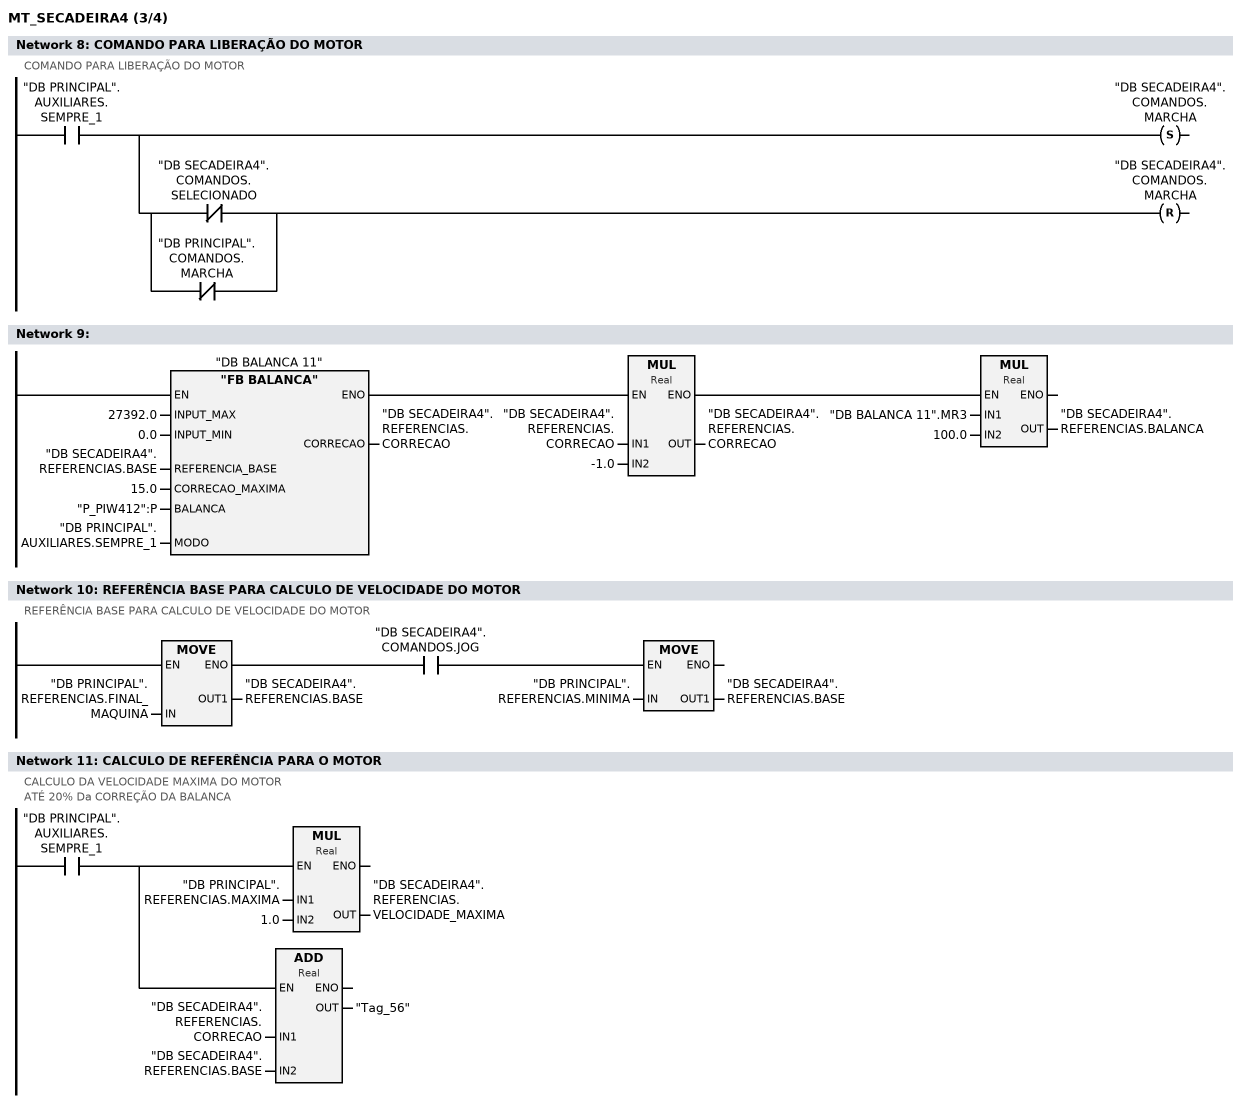
   RUNG wire#powerrail
      Contact( "DB PRINCIPAL".AUXILIARES.SEMPRE_1 )
      wire#w1
      S_Coil( "DB SECADEIRA4".COMANDOS.MARCHA )
   END_RUNG
   RUNG wire#w1
      I_Contact( "DB SECADEIRA4".COMANDOS.SELECIONADO )
      wire#w2
      R_Coil( "DB SECADEIRA4".COMANDOS.MARCHA )
   END_RUNG
   RUNG wire#w1
      I_Contact( "DB PRINCIPAL".COMANDOS.MARCHA )
   END_RUNG wire#w2
   // the same network as SCL:
   IF "DB PRINCIPAL".AUXILIARES.SEMPRE_1 THEN "DB SECADEIRA4".COMANDOS.MARCHA := TRUE; END_IF;
   IF "DB PRINCIPAL".AUXILIARES.SEMPRE_1 AND (NOT "DB SECADEIRA4".COMANDOS.SELECIONADO OR NOT "DB PRINCIPAL".COMANDOS.MARCHA) THEN
       "DB SECADEIRA4".COMANDOS.MARCHA := FALSE;
   END_IF;
END_REGION

REGION Network 9
   RUNG wire#powerrail
      "DB BALANCA 11"(INPUT_MAX := 27392.0, INPUT_MIN := 0.0, REFERENCIA_BASE := "DB SECADEIRA4".REFERENCIAS.BASE, CORRECAO_MAXIMA := 15.0, BALANCA := "P_PIW412":P, MODO := "DB PRINCIPAL".AUXILIARES.SEMPRE_1, CORRECAO => "DB SECADEIRA4".REFERENCIAS.CORRECAO)
      { S7_Templates := "SrcType := Real"; S7_GenerateENO := "TRUE" } Mul(in1 := "DB SECADEIRA4".REFERENCIAS.CORRECAO, in2 := -1.0, out => "DB SECADEIRA4".REFERENCIAS.CORRECAO)
      { S7_Templates := "SrcType := Real"; S7_GenerateENO := "TRUE" } Mul(in1 := "DB BALANCA 11".MR3, in2 := 100.0, out => "DB SECADEIRA4".REFERENCIAS.BALANCA)
   END_RUNG
   // the same network as SCL:
   // ENO of a box is taken as its EN; it also drops when the box reports an error
   "DB BALANCA 11"(INPUT_MAX := 27392.0,   // "FB BALANCA"
                   INPUT_MIN := 0.0,
                   REFERENCIA_BASE := "DB SECADEIRA4".REFERENCIAS.BASE,
                   CORRECAO_MAXIMA := 15.0,
                   BALANCA := "P_PIW412":P,
                   MODO := "DB PRINCIPAL".AUXILIARES.SEMPRE_1,
                   CORRECAO => "DB SECADEIRA4".REFERENCIAS.CORRECAO,
                   ENO => #_w1);
   IF #_w1 THEN
       "DB SECADEIRA4".REFERENCIAS.CORRECAO := "DB SECADEIRA4".REFERENCIAS.CORRECAO * (-1.0);
       "DB SECADEIRA4".REFERENCIAS.BALANCA := "DB BALANCA 11".MR3 * 100.0;
   END_IF;
END_REGION

REGION Network 10: REFERÊNCIA BASE PARA CALCULO DE VELOCIDADE DO MOTOR
   // REFERÊNCIA BASE PARA CALCULO DE VELOCIDADE DO MOTOR
   RUNG wire#powerrail
      { S7_GenerateENO := "TRUE" } Move(in := "DB PRINCIPAL".REFERENCIAS.FINAL_MAQUINA, out1 => "DB SECADEIRA4".REFERENCIAS.BASE)
      Contact( "DB SECADEIRA4".COMANDOS.JOG )
      { S7_GenerateENO := "TRUE" } Move(in := "DB PRINCIPAL".REFERENCIAS.MINIMA, out1 => "DB SECADEIRA4".REFERENCIAS.BASE)
   END_RUNG
   // the same network as SCL:
   // ENO of a box is taken as its EN; it also drops when the box reports an error
   "DB SECADEIRA4".REFERENCIAS.BASE := "DB PRINCIPAL".REFERENCIAS.FINAL_MAQUINA;
   IF "DB SECADEIRA4".COMANDOS.JOG THEN
       "DB SECADEIRA4".REFERENCIAS.BASE := "DB PRINCIPAL".REFERENCIAS.MINIMA;
   END_IF;
END_REGION

REGION Network 11: CALCULO DE REFERÊNCIA PARA O MOTOR
   // CALCULO DA VELOCIDADE MAXIMA DO MOTOR
   // ATÉ 20% Da CORREÇÃO DA BALANCA
   RUNG wire#powerrail
      Contact( "DB PRINCIPAL".AUXILIARES.SEMPRE_1 )
      wire#w1
      { S7_Templates := "SrcType := Real"; S7_GenerateENO := "TRUE" } Mul(in1 := "DB PRINCIPAL".REFERENCIAS.MAXIMA, in2 := 1.0, out => "DB SECADEIRA4".REFERENCIAS.VELOCIDADE_MAXIMA)
   END_RUNG
   RUNG wire#w1
      { S7_Templates := "SrcType := Real"; S7_GenerateENO := "TRUE" } Add(in1 := "DB SECADEIRA4".REFERENCIAS.CORRECAO, in2 := "DB SECADEIRA4".REFERENCIAS.BASE, out => "Tag_56")
   END_RUNG
   // the same network as SCL:
   IF "DB PRINCIPAL".AUXILIARES.SEMPRE_1 THEN
       "DB SECADEIRA4".REFERENCIAS.VELOCIDADE_MAXIMA := "DB PRINCIPAL".REFERENCIAS.MAXIMA * 1.0;
       "Tag_56" := "DB SECADEIRA4".REFERENCIAS.CORRECAO + "DB SECADEIRA4".REFERENCIAS.BASE;
   END_IF;
END_REGION

REGION Network 12: ACC/DEC DA REFERÊNCIA DO MOTOR
   // ACC/DEC DA REFERÊNCIA DO MOTOR
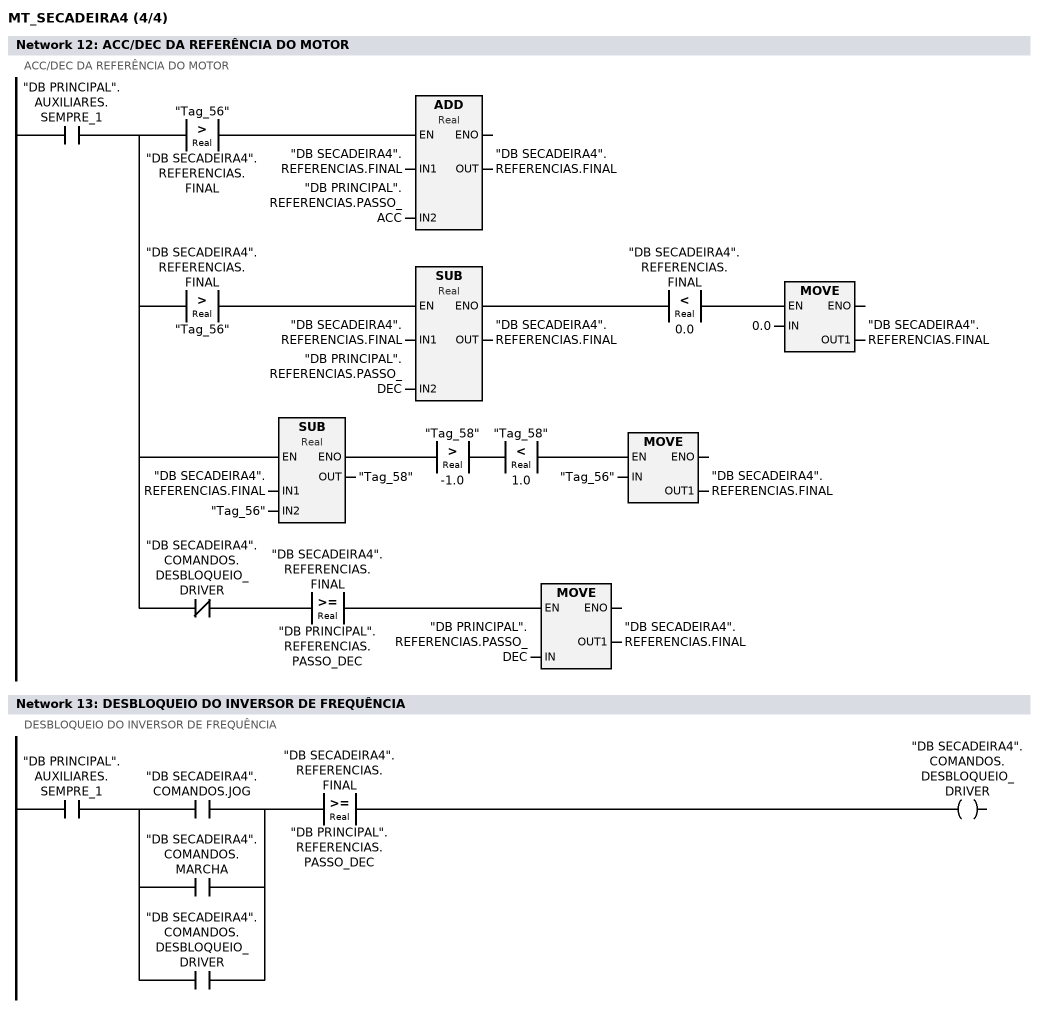
   RUNG wire#powerrail
      Contact( "DB PRINCIPAL".AUXILIARES.SEMPRE_1 )
      wire#w1
      { S7_Templates := "SrcType := Real" } GT_Contact(in1 := "Tag_56", in2 := "DB SECADEIRA4".REFERENCIAS.FINAL)
      { S7_Templates := "SrcType := Real"; S7_GenerateENO := "TRUE" } Add(in1 := "DB SECADEIRA4".REFERENCIAS.FINAL, in2 := "DB PRINCIPAL".REFERENCIAS.PASSO_ACC, out => "DB SECADEIRA4".REFERENCIAS.FINAL)
   END_RUNG
   RUNG wire#w1
      { S7_Templates := "SrcType := Real" } GT_Contact(in1 := "DB SECADEIRA4".REFERENCIAS.FINAL, in2 := "Tag_56")
      { S7_Templates := "SrcType := Real"; S7_GenerateENO := "TRUE" } Sub(in1 := "DB SECADEIRA4".REFERENCIAS.FINAL, in2 := "DB PRINCIPAL".REFERENCIAS.PASSO_DEC, out => "DB SECADEIRA4".REFERENCIAS.FINAL)
      { S7_Templates := "SrcType := Real" } LT_Contact(in1 := "DB SECADEIRA4".REFERENCIAS.FINAL, in2 := 0.0)
      { S7_GenerateENO := "TRUE" } Move(in := 0.0, out1 => "DB SECADEIRA4".REFERENCIAS.FINAL)
   END_RUNG
   RUNG wire#w1
      { S7_Templates := "SrcType := Real"; S7_GenerateENO := "TRUE" } Sub(in1 := "DB SECADEIRA4".REFERENCIAS.FINAL, in2 := "Tag_56", out => "Tag_58")
      { S7_Templates := "SrcType := Real" } GT_Contact(in1 := "Tag_58", in2 := -1.0)
      { S7_Templates := "SrcType := Real" } LT_Contact(in1 := "Tag_58", in2 := 1.0)
      { S7_GenerateENO := "TRUE" } Move(in := "Tag_56", out1 => "DB SECADEIRA4".REFERENCIAS.FINAL)
   END_RUNG
   RUNG wire#w1
      I_Contact( "DB SECADEIRA4".COMANDOS.DESBLOQUEIO_DRIVER )
      { S7_Templates := "SrcType := Real" } GE_Contact(in1 := "DB SECADEIRA4".REFERENCIAS.FINAL, in2 := "DB PRINCIPAL".REFERENCIAS.PASSO_DEC)
      { S7_GenerateENO := "TRUE" } Move(in := "DB PRINCIPAL".REFERENCIAS.PASSO_DEC, out1 => "DB SECADEIRA4".REFERENCIAS.FINAL)
   END_RUNG
   // the same network as SCL:
   // ENO of a box is taken as its EN; it also drops when the box reports an error
   IF "DB PRINCIPAL".AUXILIARES.SEMPRE_1 AND ("Tag_56" > "DB SECADEIRA4".REFERENCIAS.FINAL) THEN
       "DB SECADEIRA4".REFERENCIAS.FINAL := "DB SECADEIRA4".REFERENCIAS.FINAL + "DB PRINCIPAL".REFERENCIAS.PASSO_ACC;
   END_IF;
   #_w1 := "DB PRINCIPAL".AUXILIARES.SEMPRE_1 AND ("DB SECADEIRA4".REFERENCIAS.FINAL > "Tag_56");
   IF #_w1 THEN
       "DB SECADEIRA4".REFERENCIAS.FINAL := "DB SECADEIRA4".REFERENCIAS.FINAL - "DB PRINCIPAL".REFERENCIAS.PASSO_DEC;
   END_IF;
   IF #_w1 AND ("DB SECADEIRA4".REFERENCIAS.FINAL < 0.0) THEN
       "DB SECADEIRA4".REFERENCIAS.FINAL := 0.0;
   END_IF;
   IF "DB PRINCIPAL".AUXILIARES.SEMPRE_1 THEN
       "Tag_58" := "DB SECADEIRA4".REFERENCIAS.FINAL - "Tag_56";
   END_IF;
   IF "DB PRINCIPAL".AUXILIARES.SEMPRE_1 AND ("Tag_58" > (-1.0)) AND ("Tag_58" < 1.0) THEN
       "DB SECADEIRA4".REFERENCIAS.FINAL := "Tag_56";
   END_IF;
   IF "DB PRINCIPAL".AUXILIARES.SEMPRE_1 AND NOT "DB SECADEIRA4".COMANDOS.DESBLOQUEIO_DRIVER AND ("DB SECADEIRA4".REFERENCIAS.FINAL >= "DB PRINCIPAL".REFERENCIAS.PASSO_DEC) THEN
       "DB SECADEIRA4".REFERENCIAS.FINAL := "DB PRINCIPAL".REFERENCIAS.PASSO_DEC;
   END_IF;
END_REGION

REGION Network 13: DESBLOQUEIO DO INVERSOR DE FREQUÊNCIA
   // DESBLOQUEIO DO INVERSOR DE FREQUÊNCIA
   RUNG wire#powerrail
      Contact( "DB PRINCIPAL".AUXILIARES.SEMPRE_1 )
      wire#w1
      Contact( "DB SECADEIRA4".COMANDOS.JOG )
      wire#w2
      { S7_Templates := "SrcType := Real" } GE_Contact(in1 := "DB SECADEIRA4".REFERENCIAS.FINAL, in2 := "DB PRINCIPAL".REFERENCIAS.PASSO_DEC)
      Coil( "DB SECADEIRA4".COMANDOS.DESBLOQUEIO_DRIVER )
   END_RUNG
   RUNG wire#w1
      Contact( "DB SECADEIRA4".COMANDOS.MARCHA )
   END_RUNG wire#w2
   RUNG wire#w1
      Contact( "DB SECADEIRA4".COMANDOS.DESBLOQUEIO_DRIVER )
   END_RUNG wire#w2
   // the same network as SCL:
   "DB SECADEIRA4".COMANDOS.DESBLOQUEIO_DRIVER := "DB PRINCIPAL".AUXILIARES.SEMPRE_1 AND ("DB SECADEIRA4".COMANDOS.JOG OR "DB SECADEIRA4".COMANDOS.MARCHA OR "DB SECADEIRA4".COMANDOS.DESBLOQUEIO_DRIVER) AND ("DB SECADEIRA4".REFERENCIAS.FINAL >= "DB PRINCIPAL".REFERENCIAS.PASSO_DEC);
END_REGION

REGION Network 14 (STL): STATUS / CONTROLE - INVERSOR DE FREQUÊNCIA
   // DANFOSS FC300 PROFIBUS - TEX24626INV001
   // STATUS DO INVERSOR DE FREQUÊNCIA
         L     "Tag_42":P;
         T     "Tag_1";
         AN    "Tag_59";
         =     "DB SECADEIRA4".COMANDOS.STATUS_DRIVER;

   // CONTROLE DO INVERSOR DE FREQUÊNCIA
         L     1150;
         T     "Tag_1";
         A     "DB SECADEIRA4".COMANDOS.DESBLOQUEIO_DRIVER;
         =     "Tag_60";
         A     "T2";
         AN    "DB SECADEIRA4".COMANDOS.STATUS_DRIVER;
         =     "Tag_61";
         L     "Tag_1";
         T     "Tag_43":P;

   // REFERÊNCIA PARA O INVERSOR DE FREQUÊNCIA
         L     "DB SECADEIRA4".REFERENCIAS.FINAL;
         L     16384.0;
         *R;

         L     "DB SECADEIRA4".REFERENCIAS.VELOCIDADE_MAXIMA;
         /R;
         RND;
         T     "Tag_62";
         L     "Tag_62";
         T     "Tag_44":P;
END_REGION

REGION Network 15 (STL): INVERSOR RESERVA
         A     "DB PRINCIPAL".AUXILIARES.SEMPRE_1;
         =     %L24.0;
         A     %L24.0;
         A(;
         L     "DB PRINCIPAL".AUXILIARES1.INVERSOR_RESERVA1;
         L     15;
         ==I;
         );
         =     %L24.1;
         A     %L24.1;
         JNB   M00d;
         L     "DB SECADEIRA4".REFERENCIAS.FINAL;
         L     3.456;
         *R;
         T     #AUX_R;
         RND;
         T     "P_QW100":P;
   M00d: NOP   0;
         A     %L24.1;
         A     "I130";
         S     "DB PRINCIPAL".ALARME.INV_RESERVA1;
         A     %L24.1;
         A     "DB SECADEIRA4".COMANDOS.DESBLOQUEIO_DRIVER;
         S     "Q134";
         A     %L24.1;
         AN    "DB SECADEIRA4".COMANDOS.DESBLOQUEIO_DRIVER;
         R     "Q134";
         A     %L24.0;
         A(;
         L     "DB PRINCIPAL".AUXILIARES1.INVERSOR_RESERVA2;
         L     15;
         ==I;
         );
         =     %L24.1;
         A     %L24.1;
         JNB   M00e;
         L     "DB SECADEIRA4".REFERENCIAS.FINAL;
         L     3.456;
         *R;
         T     #AUX_R;
         RND;
         T     "P_QW102":P;
   M00e: NOP   0;
         A     %L24.1;
         A     "I132";
         S     "DB PRINCIPAL".ALARME.INV_RESERVA2;
         A     %L24.1;
         A     "DB SECADEIRA4".COMANDOS.DESBLOQUEIO_DRIVER;
         S     "Q135";
         A     %L24.1;
         AN    "DB SECADEIRA4".COMANDOS.DESBLOQUEIO_DRIVER;
         R     "Q135";
END_REGION
END_FUNCTION

FUNCTION "MT_PUXADOR_JOTA_SAIDA" : Void   // FC25, LAD
TITLE = MÓDULO DE CONTROLE DO PUXADOR DO JOTA DA SAIDA
{ S7_Optimized_Access := 'FALSE' }
AUTHOR : THALLES
FAMILY : TRAÇÃO
NAME : LINHA1
VERSION : 0.1
// DATA BLOCK DE CONTROLE // DB25
// Automation Pack Automação Indl. e Com. Ltda.
// Cliente: Texima S/A Ind. de Máquinas
// Cliente Final: Cia. Fiação e Tecidos Santo Antonio.
// Máquina: LINHA 1 DENIN - O.S.: 24.626
   VAR_TEMP
      AUX_R : Real;
   END_VAR
   VAR_TEMP   // added for the SCL form of the ladder/FBD networks
      _w1 : Bool;
   END_VAR
BEGIN

REGION Network 1: ALARMES
   // RESET DOS ALARMES
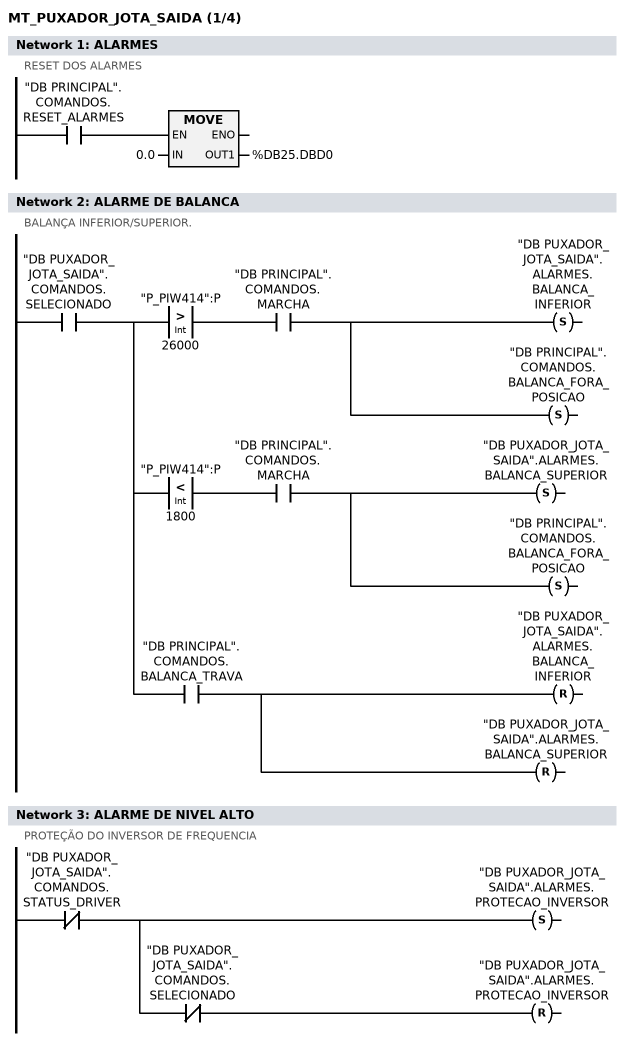
   RUNG wire#powerrail
      Contact( "DB PRINCIPAL".COMANDOS.RESET_ALARMES )
      { S7_GenerateENO := "TRUE" } Move(in := 0.0, out1 => %DB25.DBD0)
   END_RUNG
   // the same network as SCL:
   IF "DB PRINCIPAL".COMANDOS.RESET_ALARMES THEN %DB25.DBD0 := 0.0; END_IF;
END_REGION

REGION Network 2: ALARME DE BALANCA
   // BALANÇA INFERIOR/SUPERIOR.
   RUNG wire#powerrail
      Contact( "DB PUXADOR_JOTA_SAIDA".COMANDOS.SELECIONADO )
      wire#w1
      { S7_Templates := "SrcType := Int" } GT_Contact(in1 := "P_PIW414":P, in2 := 26000)
      Contact( "DB PRINCIPAL".COMANDOS.MARCHA )
      wire#w2
      S_Coil( "DB PUXADOR_JOTA_SAIDA".ALARMES.BALANCA_INFERIOR )
   END_RUNG
   RUNG wire#w2
      S_Coil( "DB PRINCIPAL".COMANDOS.BALANCA_FORA_POSICAO )
   END_RUNG
   RUNG wire#w1
      { S7_Templates := "SrcType := Int" } LT_Contact(in1 := "P_PIW414":P, in2 := 1800)
      Contact( "DB PRINCIPAL".COMANDOS.MARCHA )
      wire#w3
      S_Coil( "DB PUXADOR_JOTA_SAIDA".ALARMES.BALANCA_SUPERIOR )
   END_RUNG
   RUNG wire#w3
      S_Coil( "DB PRINCIPAL".COMANDOS.BALANCA_FORA_POSICAO )
   END_RUNG
   RUNG wire#w1
      Contact( "DB PRINCIPAL".COMANDOS.BALANCA_TRAVA )
      wire#w4
      R_Coil( "DB PUXADOR_JOTA_SAIDA".ALARMES.BALANCA_INFERIOR )
   END_RUNG
   RUNG wire#w4
      R_Coil( "DB PUXADOR_JOTA_SAIDA".ALARMES.BALANCA_SUPERIOR )
   END_RUNG
   // the same network as SCL:
   IF "DB PUXADOR_JOTA_SAIDA".COMANDOS.SELECIONADO AND ("P_PIW414":P > 26000) AND "DB PRINCIPAL".COMANDOS.MARCHA THEN
       "DB PUXADOR_JOTA_SAIDA".ALARMES.BALANCA_INFERIOR := TRUE;
       "DB PRINCIPAL".COMANDOS.BALANCA_FORA_POSICAO := TRUE;
   END_IF;
   IF "DB PUXADOR_JOTA_SAIDA".COMANDOS.SELECIONADO AND ("P_PIW414":P < 1800) AND "DB PRINCIPAL".COMANDOS.MARCHA THEN
       "DB PUXADOR_JOTA_SAIDA".ALARMES.BALANCA_SUPERIOR := TRUE;
       "DB PRINCIPAL".COMANDOS.BALANCA_FORA_POSICAO := TRUE;
   END_IF;
   IF "DB PUXADOR_JOTA_SAIDA".COMANDOS.SELECIONADO AND "DB PRINCIPAL".COMANDOS.BALANCA_TRAVA THEN
       "DB PUXADOR_JOTA_SAIDA".ALARMES.BALANCA_INFERIOR := FALSE;
       "DB PUXADOR_JOTA_SAIDA".ALARMES.BALANCA_SUPERIOR := FALSE;
   END_IF;
END_REGION

REGION Network 3: ALARME DE NIVEL ALTO
   // PROTEÇÃO DO INVERSOR DE FREQUENCIA
   RUNG wire#powerrail
      I_Contact( "DB PUXADOR_JOTA_SAIDA".COMANDOS.STATUS_DRIVER )
      wire#w1
      S_Coil( "DB PUXADOR_JOTA_SAIDA".ALARMES.PROTECAO_INVERSOR )
   END_RUNG
   RUNG wire#w1
      I_Contact( "DB PUXADOR_JOTA_SAIDA".COMANDOS.SELECIONADO )
      R_Coil( "DB PUXADOR_JOTA_SAIDA".ALARMES.PROTECAO_INVERSOR )
   END_RUNG
   // the same network as SCL:
   #_w1 := NOT "DB PUXADOR_JOTA_SAIDA".COMANDOS.STATUS_DRIVER;
   IF #_w1 THEN "DB PUXADOR_JOTA_SAIDA".ALARMES.PROTECAO_INVERSOR := TRUE; END_IF;
   IF #_w1 AND NOT "DB PUXADOR_JOTA_SAIDA".COMANDOS.SELECIONADO THEN
       "DB PUXADOR_JOTA_SAIDA".ALARMES.PROTECAO_INVERSOR := FALSE;
   END_IF;
END_REGION

REGION Network 4: ALARMES
   // ATIVAÇÃO DO BIT DE ALARME DE NIVEL ALTO
   // ATIVAÇÃO DO BIT DE ALARME DE NIVEL BAIXO
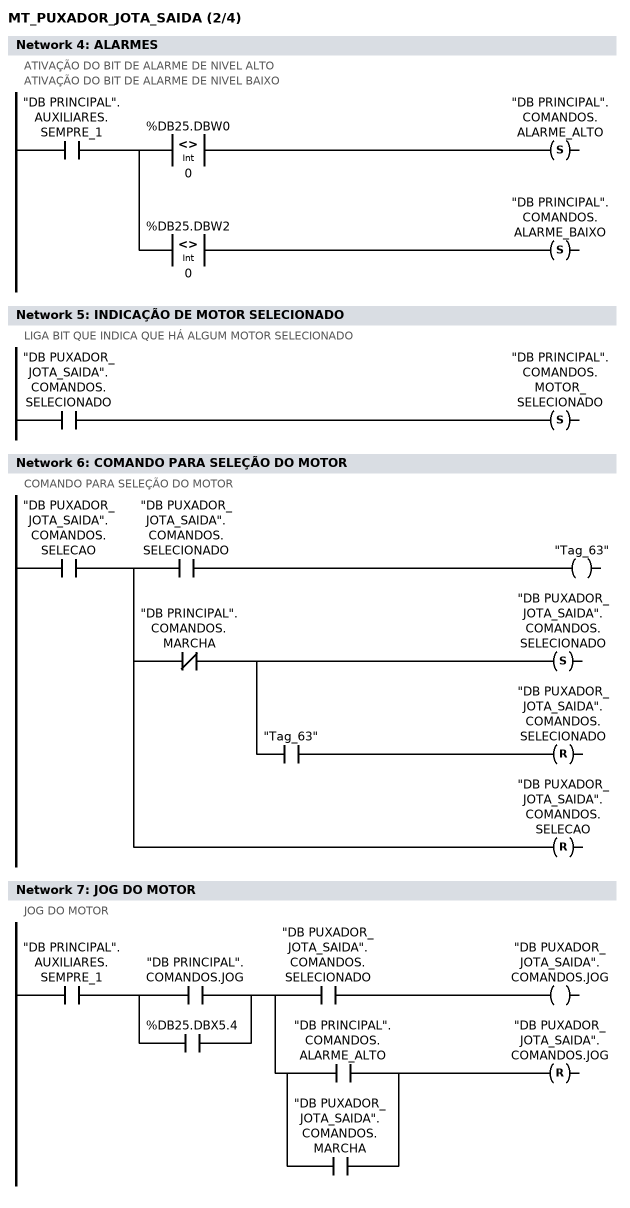
   RUNG wire#powerrail
      Contact( "DB PRINCIPAL".AUXILIARES.SEMPRE_1 )
      wire#w1
      { S7_Templates := "SrcType := Int" } NE_Contact(in1 := %DB25.DBW0, in2 := 0)
      S_Coil( "DB PRINCIPAL".COMANDOS.ALARME_ALTO )
   END_RUNG
   RUNG wire#w1
      { S7_Templates := "SrcType := Int" } NE_Contact(in1 := %DB25.DBW2, in2 := 0)
      S_Coil( "DB PRINCIPAL".COMANDOS.ALARME_BAIXO )
   END_RUNG
   // the same network as SCL:
   IF "DB PRINCIPAL".AUXILIARES.SEMPRE_1 AND (%DB25.DBW0 <> 0) THEN
       "DB PRINCIPAL".COMANDOS.ALARME_ALTO := TRUE;
   END_IF;
   IF "DB PRINCIPAL".AUXILIARES.SEMPRE_1 AND (%DB25.DBW2 <> 0) THEN
       "DB PRINCIPAL".COMANDOS.ALARME_BAIXO := TRUE;
   END_IF;
END_REGION

REGION Network 5: INDICAÇÃO DE MOTOR SELECIONADO
   // LIGA BIT QUE INDICA QUE HÁ ALGUM MOTOR SELECIONADO
   RUNG wire#powerrail
      Contact( "DB PUXADOR_JOTA_SAIDA".COMANDOS.SELECIONADO )
      S_Coil( "DB PRINCIPAL".COMANDOS.MOTOR_SELECIONADO )
   END_RUNG
   // the same network as SCL:
   IF "DB PUXADOR_JOTA_SAIDA".COMANDOS.SELECIONADO THEN
       "DB PRINCIPAL".COMANDOS.MOTOR_SELECIONADO := TRUE;
   END_IF;
END_REGION

REGION Network 6: COMANDO PARA SELEÇÃO DO MOTOR
   // COMANDO PARA SELEÇÃO DO MOTOR
   RUNG wire#powerrail
      Contact( "DB PUXADOR_JOTA_SAIDA".COMANDOS.SELECAO )
      wire#w1
      Contact( "DB PUXADOR_JOTA_SAIDA".COMANDOS.SELECIONADO )
      Coil( "Tag_63" )
   END_RUNG
   RUNG wire#w1
      I_Contact( "DB PRINCIPAL".COMANDOS.MARCHA )
      wire#w2
      S_Coil( "DB PUXADOR_JOTA_SAIDA".COMANDOS.SELECIONADO )
   END_RUNG
   RUNG wire#w2
      Contact( "Tag_63" )
      R_Coil( "DB PUXADOR_JOTA_SAIDA".COMANDOS.SELECIONADO )
   END_RUNG
   RUNG wire#w1
      R_Coil( "DB PUXADOR_JOTA_SAIDA".COMANDOS.SELECAO )
   END_RUNG
   // the same network as SCL:
   "Tag_63" := "DB PUXADOR_JOTA_SAIDA".COMANDOS.SELECAO AND "DB PUXADOR_JOTA_SAIDA".COMANDOS.SELECIONADO;
   #_w1 := "DB PUXADOR_JOTA_SAIDA".COMANDOS.SELECAO AND NOT "DB PRINCIPAL".COMANDOS.MARCHA;
   IF #_w1 THEN "DB PUXADOR_JOTA_SAIDA".COMANDOS.SELECIONADO := TRUE; END_IF;
   IF #_w1 AND "Tag_63" THEN "DB PUXADOR_JOTA_SAIDA".COMANDOS.SELECIONADO := FALSE; END_IF;
   IF "DB PUXADOR_JOTA_SAIDA".COMANDOS.SELECAO THEN
       "DB PUXADOR_JOTA_SAIDA".COMANDOS.SELECAO := FALSE;
   END_IF;
END_REGION

REGION Network 7: JOG DO MOTOR
   // JOG DO MOTOR
   RUNG wire#powerrail
      Contact( "DB PRINCIPAL".AUXILIARES.SEMPRE_1 )
      wire#w1
      Contact( "DB PRINCIPAL".COMANDOS.JOG )
      wire#w2
      Contact( "DB PUXADOR_JOTA_SAIDA".COMANDOS.SELECIONADO )
      Coil( "DB PUXADOR_JOTA_SAIDA".COMANDOS.JOG )
   END_RUNG
   RUNG wire#w1
      Contact( %DB25.DBX5.4 )
   END_RUNG wire#w2
   RUNG wire#w2
      Contact( "DB PRINCIPAL".COMANDOS.ALARME_ALTO )
      wire#w3
      R_Coil( "DB PUXADOR_JOTA_SAIDA".COMANDOS.JOG )
   END_RUNG
   RUNG wire#w2
      Contact( "DB PUXADOR_JOTA_SAIDA".COMANDOS.MARCHA )
   END_RUNG wire#w3
   // the same network as SCL:
   #_w1 := "DB PRINCIPAL".AUXILIARES.SEMPRE_1 AND ("DB PRINCIPAL".COMANDOS.JOG OR %DB25.DBX5.4);
   "DB PUXADOR_JOTA_SAIDA".COMANDOS.JOG := #_w1 AND "DB PUXADOR_JOTA_SAIDA".COMANDOS.SELECIONADO;
   IF #_w1 AND ("DB PRINCIPAL".COMANDOS.ALARME_ALTO OR "DB PUXADOR_JOTA_SAIDA".COMANDOS.MARCHA) THEN
       "DB PUXADOR_JOTA_SAIDA".COMANDOS.JOG := FALSE;
   END_IF;
END_REGION

REGION Network 8: COMANDO PARA LIBERAÇÃO DO MOTOR
   // COMANDO PARA LIBERAÇÃO DO MOTOR
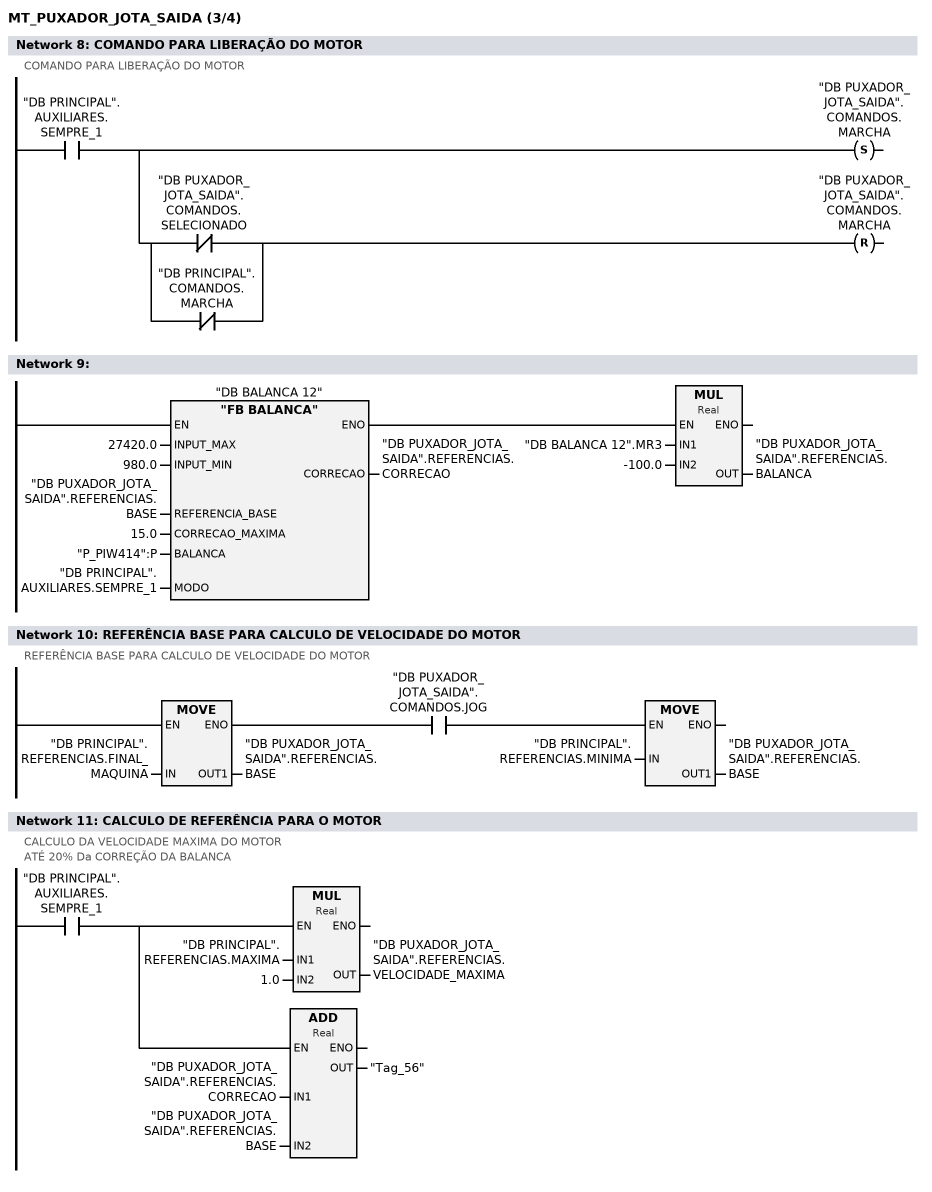
   RUNG wire#powerrail
      Contact( "DB PRINCIPAL".AUXILIARES.SEMPRE_1 )
      wire#w1
      S_Coil( "DB PUXADOR_JOTA_SAIDA".COMANDOS.MARCHA )
   END_RUNG
   RUNG wire#w1
      I_Contact( "DB PUXADOR_JOTA_SAIDA".COMANDOS.SELECIONADO )
      wire#w2
      R_Coil( "DB PUXADOR_JOTA_SAIDA".COMANDOS.MARCHA )
   END_RUNG
   RUNG wire#w1
      I_Contact( "DB PRINCIPAL".COMANDOS.MARCHA )
   END_RUNG wire#w2
   // the same network as SCL:
   IF "DB PRINCIPAL".AUXILIARES.SEMPRE_1 THEN "DB PUXADOR_JOTA_SAIDA".COMANDOS.MARCHA := TRUE; END_IF;
   IF "DB PRINCIPAL".AUXILIARES.SEMPRE_1 AND (NOT "DB PUXADOR_JOTA_SAIDA".COMANDOS.SELECIONADO OR NOT "DB PRINCIPAL".COMANDOS.MARCHA) THEN
       "DB PUXADOR_JOTA_SAIDA".COMANDOS.MARCHA := FALSE;
   END_IF;
END_REGION

REGION Network 9
   RUNG wire#powerrail
      "DB BALANCA 12"(INPUT_MAX := 27420.0, INPUT_MIN := 980.0, REFERENCIA_BASE := "DB PUXADOR_JOTA_SAIDA".REFERENCIAS.BASE, CORRECAO_MAXIMA := 15.0, BALANCA := "P_PIW414":P, MODO := "DB PRINCIPAL".AUXILIARES.SEMPRE_1, CORRECAO => "DB PUXADOR_JOTA_SAIDA".REFERENCIAS.CORRECAO)
      { S7_Templates := "SrcType := Real"; S7_GenerateENO := "TRUE" } Mul(in1 := "DB BALANCA 12".MR3, in2 := -100.0, out => "DB PUXADOR_JOTA_SAIDA".REFERENCIAS.BALANCA)
   END_RUNG
   // the same network as SCL:
   "DB BALANCA 12"(INPUT_MAX := 27420.0,   // "FB BALANCA"
                   INPUT_MIN := 980.0,
                   REFERENCIA_BASE := "DB PUXADOR_JOTA_SAIDA".REFERENCIAS.BASE,
                   CORRECAO_MAXIMA := 15.0,
                   BALANCA := "P_PIW414":P,
                   MODO := "DB PRINCIPAL".AUXILIARES.SEMPRE_1,
                   CORRECAO => "DB PUXADOR_JOTA_SAIDA".REFERENCIAS.CORRECAO,
                   ENO => #_w1);
   IF #_w1 THEN "DB PUXADOR_JOTA_SAIDA".REFERENCIAS.BALANCA := "DB BALANCA 12".MR3 * (-100.0); END_IF;
END_REGION

REGION Network 10: REFERÊNCIA BASE PARA CALCULO DE VELOCIDADE DO MOTOR
   // REFERÊNCIA BASE PARA CALCULO DE VELOCIDADE DO MOTOR
   RUNG wire#powerrail
      { S7_GenerateENO := "TRUE" } Move(in := "DB PRINCIPAL".REFERENCIAS.FINAL_MAQUINA, out1 => "DB PUXADOR_JOTA_SAIDA".REFERENCIAS.BASE)
      Contact( "DB PUXADOR_JOTA_SAIDA".COMANDOS.JOG )
      { S7_GenerateENO := "TRUE" } Move(in := "DB PRINCIPAL".REFERENCIAS.MINIMA, out1 => "DB PUXADOR_JOTA_SAIDA".REFERENCIAS.BASE)
   END_RUNG
   // the same network as SCL:
   // ENO of a box is taken as its EN; it also drops when the box reports an error
   "DB PUXADOR_JOTA_SAIDA".REFERENCIAS.BASE := "DB PRINCIPAL".REFERENCIAS.FINAL_MAQUINA;
   IF "DB PUXADOR_JOTA_SAIDA".COMANDOS.JOG THEN
       "DB PUXADOR_JOTA_SAIDA".REFERENCIAS.BASE := "DB PRINCIPAL".REFERENCIAS.MINIMA;
   END_IF;
END_REGION

REGION Network 11: CALCULO DE REFERÊNCIA PARA O MOTOR
   // CALCULO DA VELOCIDADE MAXIMA DO MOTOR
   // ATÉ 20% Da CORREÇÃO DA BALANCA
   RUNG wire#powerrail
      Contact( "DB PRINCIPAL".AUXILIARES.SEMPRE_1 )
      wire#w1
      { S7_Templates := "SrcType := Real"; S7_GenerateENO := "TRUE" } Mul(in1 := "DB PRINCIPAL".REFERENCIAS.MAXIMA, in2 := 1.0, out => "DB PUXADOR_JOTA_SAIDA".REFERENCIAS.VELOCIDADE_MAXIMA)
   END_RUNG
   RUNG wire#w1
      { S7_Templates := "SrcType := Real"; S7_GenerateENO := "TRUE" } Add(in1 := "DB PUXADOR_JOTA_SAIDA".REFERENCIAS.CORRECAO, in2 := "DB PUXADOR_JOTA_SAIDA".REFERENCIAS.BASE, out => "Tag_56")
   END_RUNG
   // the same network as SCL:
   IF "DB PRINCIPAL".AUXILIARES.SEMPRE_1 THEN
       "DB PUXADOR_JOTA_SAIDA".REFERENCIAS.VELOCIDADE_MAXIMA := "DB PRINCIPAL".REFERENCIAS.MAXIMA * 1.0;
       "Tag_56" := "DB PUXADOR_JOTA_SAIDA".REFERENCIAS.CORRECAO + "DB PUXADOR_JOTA_SAIDA".REFERENCIAS.BASE;
   END_IF;
END_REGION

REGION Network 12: ACC/DEC DA REFERÊNCIA DO MOTOR
   // ACC/DEC DA REFERÊNCIA DO MOTOR
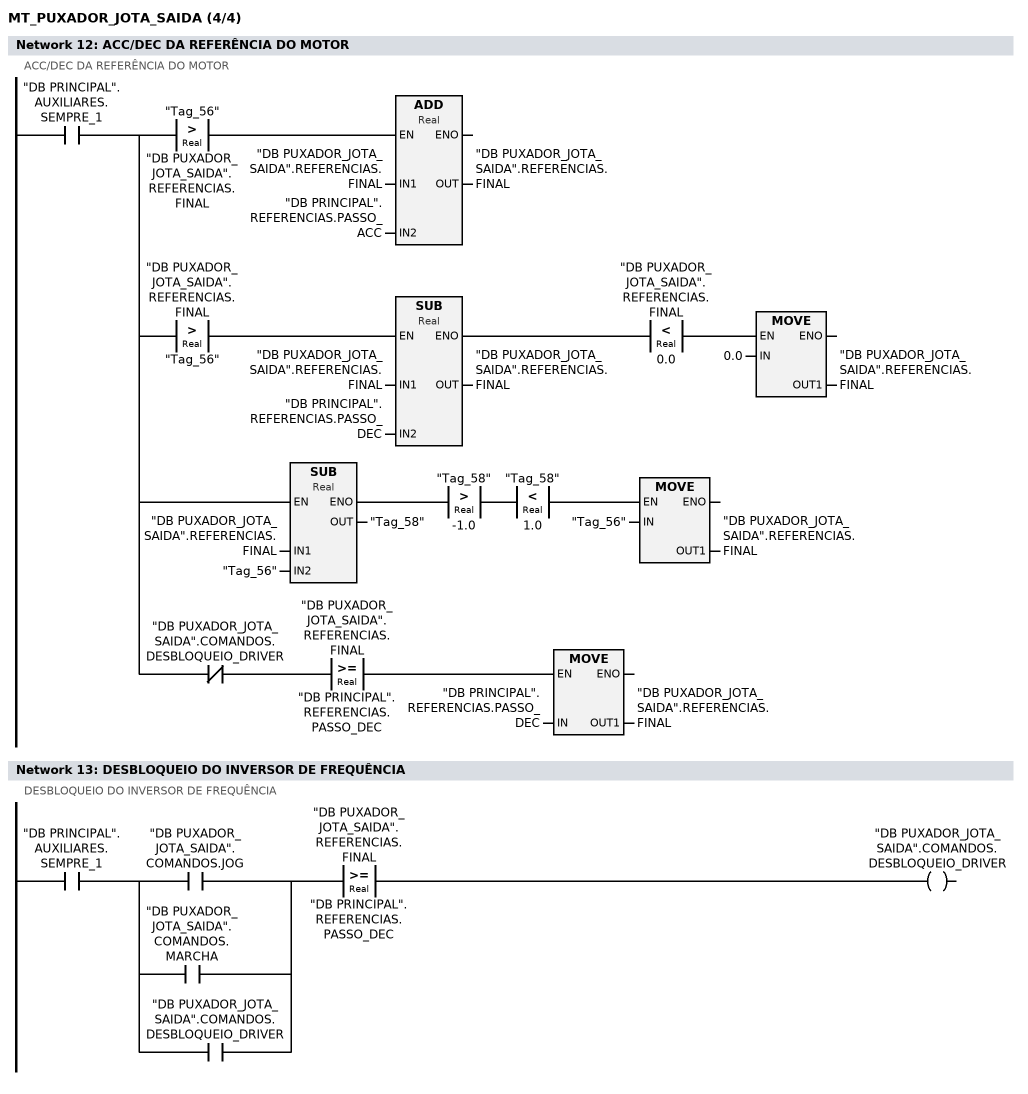
   RUNG wire#powerrail
      Contact( "DB PRINCIPAL".AUXILIARES.SEMPRE_1 )
      wire#w1
      { S7_Templates := "SrcType := Real" } GT_Contact(in1 := "Tag_56", in2 := "DB PUXADOR_JOTA_SAIDA".REFERENCIAS.FINAL)
      { S7_Templates := "SrcType := Real"; S7_GenerateENO := "TRUE" } Add(in1 := "DB PUXADOR_JOTA_SAIDA".REFERENCIAS.FINAL, in2 := "DB PRINCIPAL".REFERENCIAS.PASSO_ACC, out => "DB PUXADOR_JOTA_SAIDA".REFERENCIAS.FINAL)
   END_RUNG
   RUNG wire#w1
      { S7_Templates := "SrcType := Real" } GT_Contact(in1 := "DB PUXADOR_JOTA_SAIDA".REFERENCIAS.FINAL, in2 := "Tag_56")
      { S7_Templates := "SrcType := Real"; S7_GenerateENO := "TRUE" } Sub(in1 := "DB PUXADOR_JOTA_SAIDA".REFERENCIAS.FINAL, in2 := "DB PRINCIPAL".REFERENCIAS.PASSO_DEC, out => "DB PUXADOR_JOTA_SAIDA".REFERENCIAS.FINAL)
      { S7_Templates := "SrcType := Real" } LT_Contact(in1 := "DB PUXADOR_JOTA_SAIDA".REFERENCIAS.FINAL, in2 := 0.0)
      { S7_GenerateENO := "TRUE" } Move(in := 0.0, out1 => "DB PUXADOR_JOTA_SAIDA".REFERENCIAS.FINAL)
   END_RUNG
   RUNG wire#w1
      { S7_Templates := "SrcType := Real"; S7_GenerateENO := "TRUE" } Sub(in1 := "DB PUXADOR_JOTA_SAIDA".REFERENCIAS.FINAL, in2 := "Tag_56", out => "Tag_58")
      { S7_Templates := "SrcType := Real" } GT_Contact(in1 := "Tag_58", in2 := -1.0)
      { S7_Templates := "SrcType := Real" } LT_Contact(in1 := "Tag_58", in2 := 1.0)
      { S7_GenerateENO := "TRUE" } Move(in := "Tag_56", out1 => "DB PUXADOR_JOTA_SAIDA".REFERENCIAS.FINAL)
   END_RUNG
   RUNG wire#w1
      I_Contact( "DB PUXADOR_JOTA_SAIDA".COMANDOS.DESBLOQUEIO_DRIVER )
      { S7_Templates := "SrcType := Real" } GE_Contact(in1 := "DB PUXADOR_JOTA_SAIDA".REFERENCIAS.FINAL, in2 := "DB PRINCIPAL".REFERENCIAS.PASSO_DEC)
      { S7_GenerateENO := "TRUE" } Move(in := "DB PRINCIPAL".REFERENCIAS.PASSO_DEC, out1 => "DB PUXADOR_JOTA_SAIDA".REFERENCIAS.FINAL)
   END_RUNG
   // the same network as SCL:
   // ENO of a box is taken as its EN; it also drops when the box reports an error
   IF "DB PRINCIPAL".AUXILIARES.SEMPRE_1 AND ("Tag_56" > "DB PUXADOR_JOTA_SAIDA".REFERENCIAS.FINAL) THEN
       "DB PUXADOR_JOTA_SAIDA".REFERENCIAS.FINAL := "DB PUXADOR_JOTA_SAIDA".REFERENCIAS.FINAL + "DB PRINCIPAL".REFERENCIAS.PASSO_ACC;
   END_IF;
   #_w1 := "DB PRINCIPAL".AUXILIARES.SEMPRE_1 AND ("DB PUXADOR_JOTA_SAIDA".REFERENCIAS.FINAL > "Tag_56");
   IF #_w1 THEN
       "DB PUXADOR_JOTA_SAIDA".REFERENCIAS.FINAL := "DB PUXADOR_JOTA_SAIDA".REFERENCIAS.FINAL - "DB PRINCIPAL".REFERENCIAS.PASSO_DEC;
   END_IF;
   IF #_w1 AND ("DB PUXADOR_JOTA_SAIDA".REFERENCIAS.FINAL < 0.0) THEN
       "DB PUXADOR_JOTA_SAIDA".REFERENCIAS.FINAL := 0.0;
   END_IF;
   IF "DB PRINCIPAL".AUXILIARES.SEMPRE_1 THEN
       "Tag_58" := "DB PUXADOR_JOTA_SAIDA".REFERENCIAS.FINAL - "Tag_56";
   END_IF;
   IF "DB PRINCIPAL".AUXILIARES.SEMPRE_1 AND ("Tag_58" > (-1.0)) AND ("Tag_58" < 1.0) THEN
       "DB PUXADOR_JOTA_SAIDA".REFERENCIAS.FINAL := "Tag_56";
   END_IF;
   IF "DB PRINCIPAL".AUXILIARES.SEMPRE_1 AND NOT "DB PUXADOR_JOTA_SAIDA".COMANDOS.DESBLOQUEIO_DRIVER AND ("DB PUXADOR_JOTA_SAIDA".REFERENCIAS.FINAL >= "DB PRINCIPAL".REFERENCIAS.PASSO_DEC) THEN
       "DB PUXADOR_JOTA_SAIDA".REFERENCIAS.FINAL := "DB PRINCIPAL".REFERENCIAS.PASSO_DEC;
   END_IF;
END_REGION

REGION Network 13: DESBLOQUEIO DO INVERSOR DE FREQUÊNCIA
   // DESBLOQUEIO DO INVERSOR DE FREQUÊNCIA
   RUNG wire#powerrail
      Contact( "DB PRINCIPAL".AUXILIARES.SEMPRE_1 )
      wire#w1
      Contact( "DB PUXADOR_JOTA_SAIDA".COMANDOS.JOG )
      wire#w2
      { S7_Templates := "SrcType := Real" } GE_Contact(in1 := "DB PUXADOR_JOTA_SAIDA".REFERENCIAS.FINAL, in2 := "DB PRINCIPAL".REFERENCIAS.PASSO_DEC)
      Coil( "DB PUXADOR_JOTA_SAIDA".COMANDOS.DESBLOQUEIO_DRIVER )
   END_RUNG
   RUNG wire#w1
      Contact( "DB PUXADOR_JOTA_SAIDA".COMANDOS.MARCHA )
   END_RUNG wire#w2
   RUNG wire#w1
      Contact( "DB PUXADOR_JOTA_SAIDA".COMANDOS.DESBLOQUEIO_DRIVER )
   END_RUNG wire#w2
   // the same network as SCL:
   "DB PUXADOR_JOTA_SAIDA".COMANDOS.DESBLOQUEIO_DRIVER := "DB PRINCIPAL".AUXILIARES.SEMPRE_1 AND ("DB PUXADOR_JOTA_SAIDA".COMANDOS.JOG OR "DB PUXADOR_JOTA_SAIDA".COMANDOS.MARCHA OR "DB PUXADOR_JOTA_SAIDA".COMANDOS.DESBLOQUEIO_DRIVER) AND ("DB PUXADOR_JOTA_SAIDA".REFERENCIAS.FINAL >= "DB PRINCIPAL".REFERENCIAS.PASSO_DEC);
END_REGION

REGION Network 14 (STL): STATUS / CONTROLE - INVERSOR DE FREQUÊNCIA
   // DANFOSS FC300 PROFIBUS - TEX24626INV001
   // STATUS DO INVERSOR DE FREQUÊNCIA
         L     "Tag_45":P;
         T     "Tag_1";
         AN    "Tag_59";
         =     "DB PUXADOR_JOTA_SAIDA".COMANDOS.STATUS_DRIVER;

   // CONTROLE DO INVERSOR DE FREQUÊNCIA
         L     1150;
         T     "Tag_1";
         A     "DB PUXADOR_JOTA_SAIDA".COMANDOS.DESBLOQUEIO_DRIVER;
         =     "Tag_60";
         A     "T2";
         AN    "DB PUXADOR_JOTA_SAIDA".COMANDOS.STATUS_DRIVER;
         =     "Tag_61";
         L     "Tag_1";
         T     "Tag_46":P;

   // REFERÊNCIA PARA O INVERSOR DE FREQUÊNCIA
         L     "DB PUXADOR_JOTA_SAIDA".REFERENCIAS.FINAL;
         L     16384.0;
         *R;

         L     "DB PUXADOR_JOTA_SAIDA".REFERENCIAS.VELOCIDADE_MAXIMA;
         /R;
         RND;
         T     "Tag_62";
         L     "Tag_62";
         T     "Tag_47":P;
END_REGION

REGION Network 15 (STL): INVERSOR RESERVA
         A     "DB PRINCIPAL".AUXILIARES.SEMPRE_1;
         =     %L24.0;
         A     %L24.0;
         A(;
         L     "DB PRINCIPAL".AUXILIARES1.INVERSOR_RESERVA1;
         L     16;
         ==I;
         );
         =     %L24.1;
         A     %L24.1;
         JNB   M00c;
         L     "DB PUXADOR_JOTA_SAIDA".REFERENCIAS.FINAL;
         L     3.456;
         *R;
         T     #AUX_R;
         RND;
         T     "P_QW100":P;
   M00c: NOP   0;
         A     %L24.1;
         A     "I130";
         S     "DB PRINCIPAL".ALARME.INV_RESERVA1;
         A     %L24.1;
         A     "DB PUXADOR_JOTA_SAIDA".COMANDOS.DESBLOQUEIO_DRIVER;
         S     "Q134";
         A     %L24.1;
         AN    "DB PUXADOR_JOTA_SAIDA".COMANDOS.DESBLOQUEIO_DRIVER;
         R     "Q134";
         A     %L24.0;
         A(;
         L     "DB PRINCIPAL".AUXILIARES1.INVERSOR_RESERVA2;
         L     16;
         ==I;
         );
         =     %L24.1;
         A     %L24.1;
         JNB   M00d;
         L     "DB PUXADOR_JOTA_SAIDA".REFERENCIAS.FINAL;
         L     3.456;
         *R;
         T     #AUX_R;
         RND;
         T     "P_QW102":P;
   M00d: NOP   0;
         A     %L24.1;
         A     "I132";
         S     "DB PRINCIPAL".ALARME.INV_RESERVA2;
         A     %L24.1;
         A     "DB PUXADOR_JOTA_SAIDA".COMANDOS.DESBLOQUEIO_DRIVER;
         S     "Q135";
         A     %L24.1;
         AN    "DB PUXADOR_JOTA_SAIDA".COMANDOS.DESBLOQUEIO_DRIVER;
         R     "Q135";
END_REGION
END_FUNCTION

FUNCTION "MT_ENROLADOR_GIGANTE" : Void   // FC26, LAD
TITLE = MÓDULO DE CONTROLE DO ENROLADOR GIGANTE
{ S7_Optimized_Access := 'FALSE' }
AUTHOR : THALLES
FAMILY : TRAÇÃO
NAME : LINHA1
VERSION : 0.1
// DATA BLOCK DE CONTROLE // DB26
// Automation Pack Automação Indl. e Com. Ltda.
// Cliente: Texima S/A Ind. de Máquinas
// Cliente Final: Cia. Fiação e Tecidos Santo Antonio.
// Máquina: LINHA 1 DENIN - O.S.: 24.626
   VAR_TEMP
      AUX_R : Real;
   END_VAR
   VAR_TEMP   // added for the SCL form of the ladder/FBD networks
      _w1 : Bool;
      _w2 : Bool;
      _w3 : Bool;
      _w4 : Bool;
      _w5 : Bool;
      _w6 : Bool;
   END_VAR
BEGIN

REGION Network 1: ALARMES
   // RESET DOS ALARMES
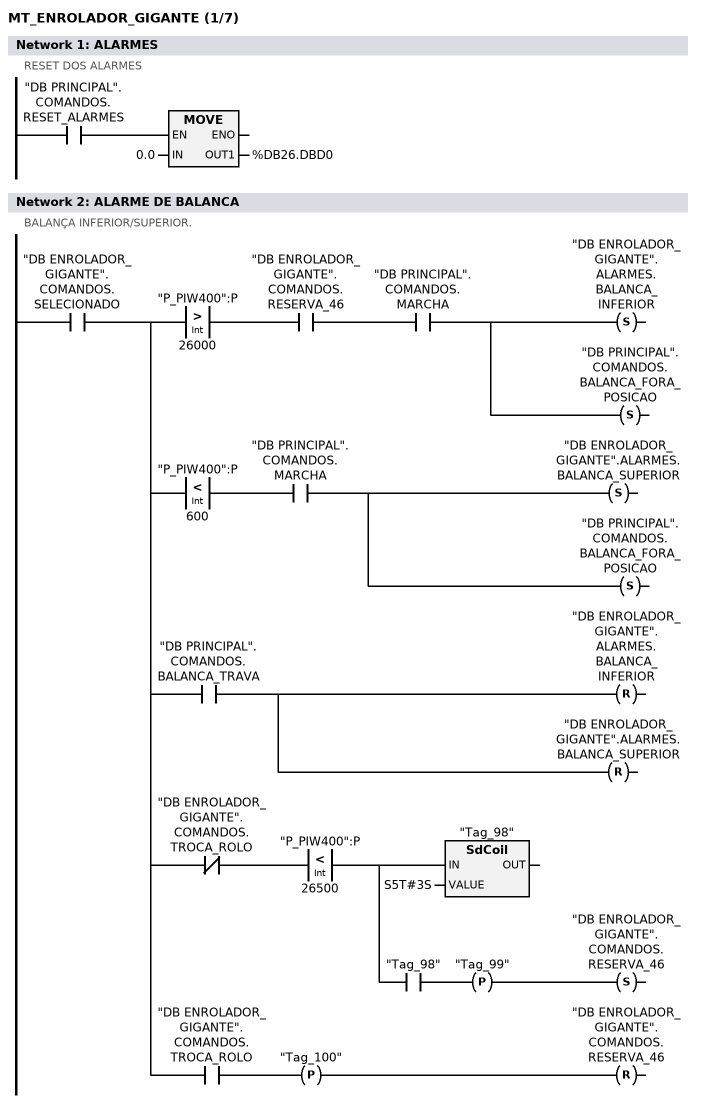
   RUNG wire#powerrail
      Contact( "DB PRINCIPAL".COMANDOS.RESET_ALARMES )
      { S7_GenerateENO := "TRUE" } Move(in := 0.0, out1 => %DB26.DBD0)
   END_RUNG
   // the same network as SCL:
   IF "DB PRINCIPAL".COMANDOS.RESET_ALARMES THEN %DB26.DBD0 := 0.0; END_IF;
END_REGION

REGION Network 2: ALARME DE BALANCA
   // BALANÇA INFERIOR/SUPERIOR.
   // no SCL statement known for SdCoil: written as a call
   IF "DB ENROLADOR_GIGANTE".COMANDOS.SELECIONADO AND ("P_PIW400":P > 26000) AND "DB ENROLADOR_GIGANTE".COMANDOS.RESERVA_46 AND "DB PRINCIPAL".COMANDOS.MARCHA THEN
       "DB ENROLADOR_GIGANTE".ALARMES.BALANCA_INFERIOR := TRUE;
       "DB PRINCIPAL".COMANDOS.BALANCA_FORA_POSICAO := TRUE;
   END_IF;
   IF "DB ENROLADOR_GIGANTE".COMANDOS.SELECIONADO AND ("P_PIW400":P < 600) AND "DB PRINCIPAL".COMANDOS.MARCHA THEN
       "DB ENROLADOR_GIGANTE".ALARMES.BALANCA_SUPERIOR := TRUE;
       "DB PRINCIPAL".COMANDOS.BALANCA_FORA_POSICAO := TRUE;
   END_IF;
   IF "DB ENROLADOR_GIGANTE".COMANDOS.SELECIONADO AND "DB PRINCIPAL".COMANDOS.BALANCA_TRAVA THEN
       "DB ENROLADOR_GIGANTE".ALARMES.BALANCA_INFERIOR := FALSE;
       "DB ENROLADOR_GIGANTE".ALARMES.BALANCA_SUPERIOR := FALSE;
   END_IF;
   #_w1 := "DB ENROLADOR_GIGANTE".COMANDOS.SELECIONADO AND NOT "DB ENROLADOR_GIGANTE".COMANDOS.TROCA_ROLO AND ("P_PIW400":P < 26500);
   #_w2 := "DB ENROLADOR_GIGANTE".COMANDOS.SELECIONADO;
   SdCoil(in := #_w1, value := S5T#3S, operand := "Tag_98");
   #_w3 := #_w1 AND "Tag_98";
   #_w4 := #_w3 AND NOT "Tag_99";   // rising edge
   "Tag_99" := #_w3;
   IF #_w4 THEN "DB ENROLADOR_GIGANTE".COMANDOS.RESERVA_46 := TRUE; END_IF;
   #_w5 := #_w2 AND "DB ENROLADOR_GIGANTE".COMANDOS.TROCA_ROLO;
   #_w6 := #_w5 AND NOT "Tag_100";   // rising edge
   "Tag_100" := #_w5;
   IF #_w6 THEN "DB ENROLADOR_GIGANTE".COMANDOS.RESERVA_46 := FALSE; END_IF;
END_REGION

REGION Network 3: ALARME DE NIVEL ALTO
   // PROTEÇÃO DO INVERSOR DE FREQUENCIA
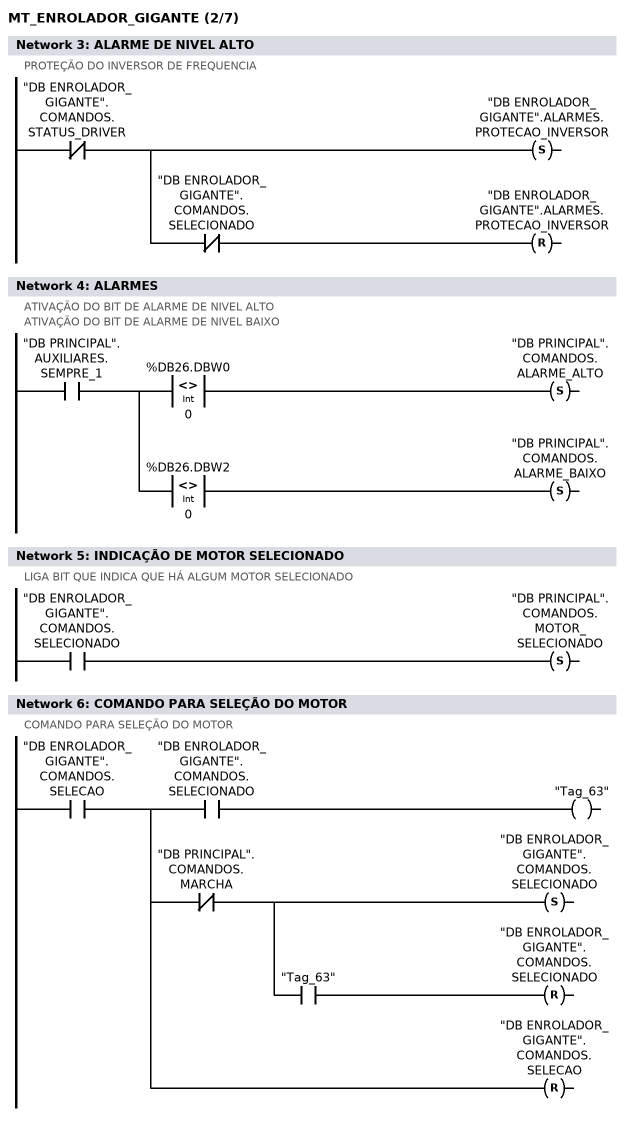
   RUNG wire#powerrail
      I_Contact( "DB ENROLADOR_GIGANTE".COMANDOS.STATUS_DRIVER )
      wire#w1
      S_Coil( "DB ENROLADOR_GIGANTE".ALARMES.PROTECAO_INVERSOR )
   END_RUNG
   RUNG wire#w1
      I_Contact( "DB ENROLADOR_GIGANTE".COMANDOS.SELECIONADO )
      R_Coil( "DB ENROLADOR_GIGANTE".ALARMES.PROTECAO_INVERSOR )
   END_RUNG
   // the same network as SCL:
   #_w1 := NOT "DB ENROLADOR_GIGANTE".COMANDOS.STATUS_DRIVER;
   IF #_w1 THEN "DB ENROLADOR_GIGANTE".ALARMES.PROTECAO_INVERSOR := TRUE; END_IF;
   IF #_w1 AND NOT "DB ENROLADOR_GIGANTE".COMANDOS.SELECIONADO THEN
       "DB ENROLADOR_GIGANTE".ALARMES.PROTECAO_INVERSOR := FALSE;
   END_IF;
END_REGION

REGION Network 4: ALARMES
   // ATIVAÇÃO DO BIT DE ALARME DE NIVEL ALTO
   // ATIVAÇÃO DO BIT DE ALARME DE NIVEL BAIXO
   RUNG wire#powerrail
      Contact( "DB PRINCIPAL".AUXILIARES.SEMPRE_1 )
      wire#w1
      { S7_Templates := "SrcType := Int" } NE_Contact(in1 := %DB26.DBW0, in2 := 0)
      S_Coil( "DB PRINCIPAL".COMANDOS.ALARME_ALTO )
   END_RUNG
   RUNG wire#w1
      { S7_Templates := "SrcType := Int" } NE_Contact(in1 := %DB26.DBW2, in2 := 0)
      S_Coil( "DB PRINCIPAL".COMANDOS.ALARME_BAIXO )
   END_RUNG
   // the same network as SCL:
   IF "DB PRINCIPAL".AUXILIARES.SEMPRE_1 AND (%DB26.DBW0 <> 0) THEN
       "DB PRINCIPAL".COMANDOS.ALARME_ALTO := TRUE;
   END_IF;
   IF "DB PRINCIPAL".AUXILIARES.SEMPRE_1 AND (%DB26.DBW2 <> 0) THEN
       "DB PRINCIPAL".COMANDOS.ALARME_BAIXO := TRUE;
   END_IF;
END_REGION

REGION Network 5: INDICAÇÃO DE MOTOR SELECIONADO
   // LIGA BIT QUE INDICA QUE HÁ ALGUM MOTOR SELECIONADO
   RUNG wire#powerrail
      Contact( "DB ENROLADOR_GIGANTE".COMANDOS.SELECIONADO )
      S_Coil( "DB PRINCIPAL".COMANDOS.MOTOR_SELECIONADO )
   END_RUNG
   // the same network as SCL:
   IF "DB ENROLADOR_GIGANTE".COMANDOS.SELECIONADO THEN
       "DB PRINCIPAL".COMANDOS.MOTOR_SELECIONADO := TRUE;
   END_IF;
END_REGION

REGION Network 6: COMANDO PARA SELEÇÃO DO MOTOR
   // COMANDO PARA SELEÇÃO DO MOTOR
   RUNG wire#powerrail
      Contact( "DB ENROLADOR_GIGANTE".COMANDOS.SELECAO )
      wire#w1
      Contact( "DB ENROLADOR_GIGANTE".COMANDOS.SELECIONADO )
      Coil( "Tag_63" )
   END_RUNG
   RUNG wire#w1
      I_Contact( "DB PRINCIPAL".COMANDOS.MARCHA )
      wire#w2
      S_Coil( "DB ENROLADOR_GIGANTE".COMANDOS.SELECIONADO )
   END_RUNG
   RUNG wire#w2
      Contact( "Tag_63" )
      R_Coil( "DB ENROLADOR_GIGANTE".COMANDOS.SELECIONADO )
   END_RUNG
   RUNG wire#w1
      R_Coil( "DB ENROLADOR_GIGANTE".COMANDOS.SELECAO )
   END_RUNG
   // the same network as SCL:
   "Tag_63" := "DB ENROLADOR_GIGANTE".COMANDOS.SELECAO AND "DB ENROLADOR_GIGANTE".COMANDOS.SELECIONADO;
   #_w1 := "DB ENROLADOR_GIGANTE".COMANDOS.SELECAO AND NOT "DB PRINCIPAL".COMANDOS.MARCHA;
   IF #_w1 THEN "DB ENROLADOR_GIGANTE".COMANDOS.SELECIONADO := TRUE; END_IF;
   IF #_w1 AND "Tag_63" THEN "DB ENROLADOR_GIGANTE".COMANDOS.SELECIONADO := FALSE; END_IF;
   IF "DB ENROLADOR_GIGANTE".COMANDOS.SELECAO THEN "DB ENROLADOR_GIGANTE".COMANDOS.SELECAO := FALSE; END_IF;
END_REGION

REGION Network 7: JOG DO MOTOR
   // JOG DO MOTOR
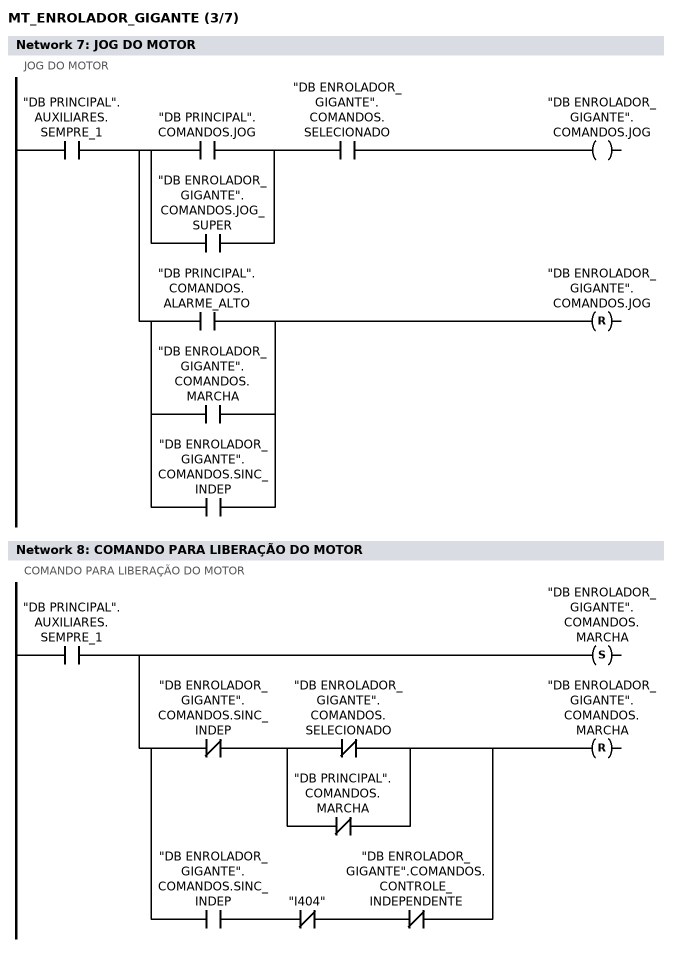
   RUNG wire#powerrail
      Contact( "DB PRINCIPAL".AUXILIARES.SEMPRE_1 )
      wire#w1
      Contact( "DB PRINCIPAL".COMANDOS.JOG )
      wire#w2
      Contact( "DB ENROLADOR_GIGANTE".COMANDOS.SELECIONADO )
      Coil( "DB ENROLADOR_GIGANTE".COMANDOS.JOG )
   END_RUNG
   RUNG wire#w1
      Contact( "DB ENROLADOR_GIGANTE".COMANDOS.JOG_SUPER )
   END_RUNG wire#w2
   RUNG wire#w1
      Contact( "DB PRINCIPAL".COMANDOS.ALARME_ALTO )
      wire#w3
      R_Coil( "DB ENROLADOR_GIGANTE".COMANDOS.JOG )
   END_RUNG
   RUNG wire#w1
      Contact( "DB ENROLADOR_GIGANTE".COMANDOS.MARCHA )
   END_RUNG wire#w3
   RUNG wire#w1
      Contact( "DB ENROLADOR_GIGANTE".COMANDOS.SINC_INDEP )
   END_RUNG wire#w3
   // the same network as SCL:
   "DB ENROLADOR_GIGANTE".COMANDOS.JOG := "DB PRINCIPAL".AUXILIARES.SEMPRE_1 AND ("DB PRINCIPAL".COMANDOS.JOG OR "DB ENROLADOR_GIGANTE".COMANDOS.JOG_SUPER) AND "DB ENROLADOR_GIGANTE".COMANDOS.SELECIONADO;
   IF "DB PRINCIPAL".AUXILIARES.SEMPRE_1 AND ("DB PRINCIPAL".COMANDOS.ALARME_ALTO OR "DB ENROLADOR_GIGANTE".COMANDOS.MARCHA OR "DB ENROLADOR_GIGANTE".COMANDOS.SINC_INDEP) THEN
       "DB ENROLADOR_GIGANTE".COMANDOS.JOG := FALSE;
   END_IF;
END_REGION

REGION Network 8: COMANDO PARA LIBERAÇÃO DO MOTOR
   // COMANDO PARA LIBERAÇÃO DO MOTOR
   RUNG wire#powerrail
      Contact( "DB PRINCIPAL".AUXILIARES.SEMPRE_1 )
      wire#w1
      S_Coil( "DB ENROLADOR_GIGANTE".COMANDOS.MARCHA )
   END_RUNG
   RUNG wire#w1
      I_Contact( "DB ENROLADOR_GIGANTE".COMANDOS.SINC_INDEP )
      wire#w2
      I_Contact( "DB ENROLADOR_GIGANTE".COMANDOS.SELECIONADO )
      wire#w3
      R_Coil( "DB ENROLADOR_GIGANTE".COMANDOS.MARCHA )
   END_RUNG
   RUNG wire#w2
      I_Contact( "DB PRINCIPAL".COMANDOS.MARCHA )
   END_RUNG wire#w3
   RUNG wire#w1
      Contact( "DB ENROLADOR_GIGANTE".COMANDOS.SINC_INDEP )
      I_Contact( "I404" )
      I_Contact( "DB ENROLADOR_GIGANTE".COMANDOS.CONTROLE_INDEPENDENTE )
   END_RUNG wire#w3
   // the same network as SCL:
   IF "DB PRINCIPAL".AUXILIARES.SEMPRE_1 THEN "DB ENROLADOR_GIGANTE".COMANDOS.MARCHA := TRUE; END_IF;
   IF "DB PRINCIPAL".AUXILIARES.SEMPRE_1 AND ((NOT "DB ENROLADOR_GIGANTE".COMANDOS.SINC_INDEP AND (NOT "DB ENROLADOR_GIGANTE".COMANDOS.SELECIONADO OR NOT "DB PRINCIPAL".COMANDOS.MARCHA)) OR ("DB ENROLADOR_GIGANTE".COMANDOS.SINC_INDEP AND NOT "I404" AND NOT "DB ENROLADOR_GIGANTE".COMANDOS.CONTROLE_INDEPENDENTE)) THEN
       "DB ENROLADOR_GIGANTE".COMANDOS.MARCHA := FALSE;
   END_IF;
END_REGION

REGION Network 9: MODO TROCA ROLO
   // LÓGICA QUE CONTROLA O MODO TROCA ROLO.
   // O MODO TROCA ROLO É RESETADO QUANDO A MAQUINA PARA
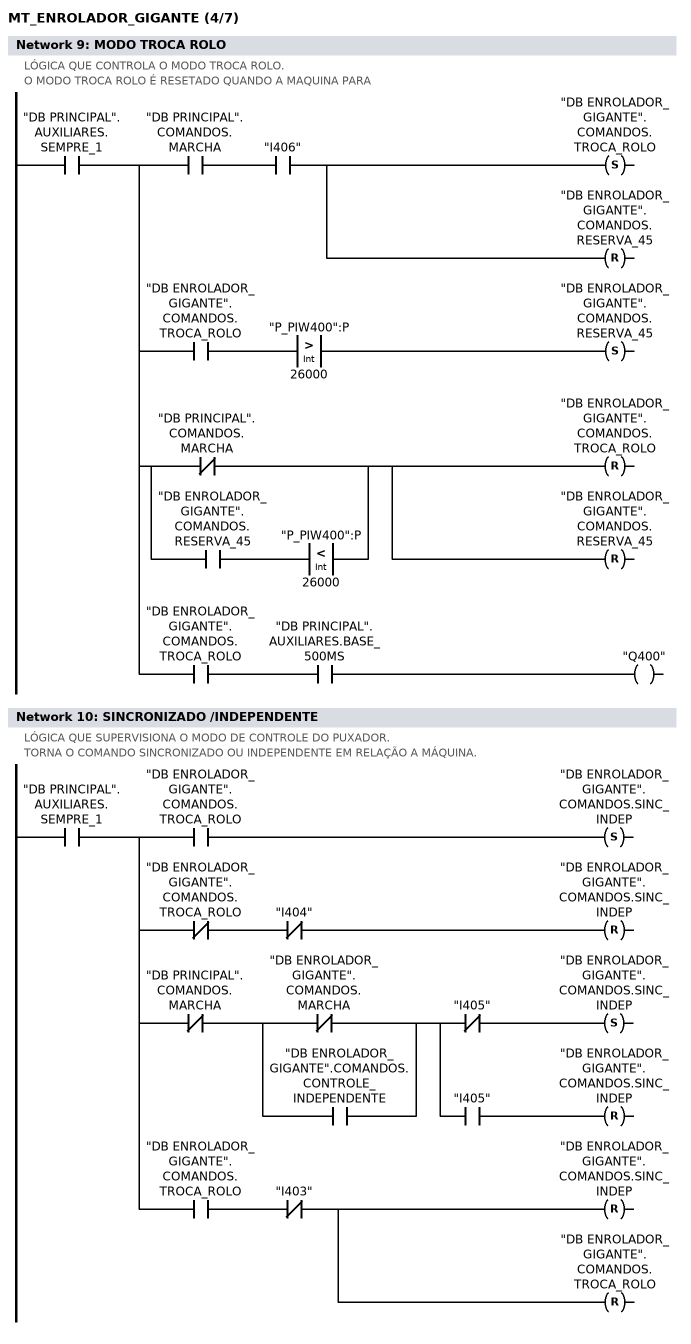
   IF "DB PRINCIPAL".AUXILIARES.SEMPRE_1 AND "DB PRINCIPAL".COMANDOS.MARCHA AND "I406" THEN
       "DB ENROLADOR_GIGANTE".COMANDOS.TROCA_ROLO := TRUE;
       "DB ENROLADOR_GIGANTE".COMANDOS.RESERVA_45 := FALSE;
   END_IF;
   IF "DB PRINCIPAL".AUXILIARES.SEMPRE_1 AND "DB ENROLADOR_GIGANTE".COMANDOS.TROCA_ROLO AND ("P_PIW400":P > 26000) THEN
       "DB ENROLADOR_GIGANTE".COMANDOS.RESERVA_45 := TRUE;
   END_IF;
   IF "DB PRINCIPAL".AUXILIARES.SEMPRE_1 AND (("DB ENROLADOR_GIGANTE".COMANDOS.RESERVA_45 AND ("P_PIW400":P < 26000)) OR NOT "DB PRINCIPAL".COMANDOS.MARCHA) THEN
       "DB ENROLADOR_GIGANTE".COMANDOS.TROCA_ROLO := FALSE;
       "DB ENROLADOR_GIGANTE".COMANDOS.RESERVA_45 := FALSE;
   END_IF;
   "Q400" := "DB PRINCIPAL".AUXILIARES.SEMPRE_1 AND "DB ENROLADOR_GIGANTE".COMANDOS.TROCA_ROLO AND "DB PRINCIPAL".AUXILIARES.BASE_500MS;
END_REGION

REGION Network 10: SINCRONIZADO /INDEPENDENTE
   // LÓGICA QUE SUPERVISIONA O MODO DE CONTROLE DO PUXADOR.
   // TORNA O COMANDO SINCRONIZADO OU INDEPENDENTE EM RELAÇÃO A MÁQUINA.
   RUNG wire#powerrail
      Contact( "DB PRINCIPAL".AUXILIARES.SEMPRE_1 )
      wire#w1
      Contact( "DB ENROLADOR_GIGANTE".COMANDOS.TROCA_ROLO )
      S_Coil( "DB ENROLADOR_GIGANTE".COMANDOS.SINC_INDEP )
   END_RUNG
   RUNG wire#w1
      I_Contact( "DB ENROLADOR_GIGANTE".COMANDOS.TROCA_ROLO )
      I_Contact( "I404" )
      R_Coil( "DB ENROLADOR_GIGANTE".COMANDOS.SINC_INDEP )
   END_RUNG
   RUNG wire#w1
      I_Contact( "DB PRINCIPAL".COMANDOS.MARCHA )
      wire#w2
      I_Contact( "DB ENROLADOR_GIGANTE".COMANDOS.MARCHA )
      wire#w3
      I_Contact( "I405" )
      S_Coil( "DB ENROLADOR_GIGANTE".COMANDOS.SINC_INDEP )
   END_RUNG
   RUNG wire#w2
      Contact( "DB ENROLADOR_GIGANTE".COMANDOS.CONTROLE_INDEPENDENTE )
   END_RUNG wire#w3
   RUNG wire#w3
      Contact( "I405" )
      R_Coil( "DB ENROLADOR_GIGANTE".COMANDOS.SINC_INDEP )
   END_RUNG
   RUNG wire#w1
      Contact( "DB ENROLADOR_GIGANTE".COMANDOS.TROCA_ROLO )
      I_Contact( "I403" )
      wire#w4
      R_Coil( "DB ENROLADOR_GIGANTE".COMANDOS.SINC_INDEP )
   END_RUNG
   RUNG wire#w4
      R_Coil( "DB ENROLADOR_GIGANTE".COMANDOS.TROCA_ROLO )
   END_RUNG
   // the same network as SCL:
   IF "DB PRINCIPAL".AUXILIARES.SEMPRE_1 AND "DB ENROLADOR_GIGANTE".COMANDOS.TROCA_ROLO THEN
       "DB ENROLADOR_GIGANTE".COMANDOS.SINC_INDEP := TRUE;
   END_IF;
   IF "DB PRINCIPAL".AUXILIARES.SEMPRE_1 AND NOT "DB ENROLADOR_GIGANTE".COMANDOS.TROCA_ROLO AND NOT "I404" THEN
       "DB ENROLADOR_GIGANTE".COMANDOS.SINC_INDEP := FALSE;
   END_IF;
   #_w1 := "DB PRINCIPAL".AUXILIARES.SEMPRE_1 AND NOT "DB PRINCIPAL".COMANDOS.MARCHA AND (NOT "DB ENROLADOR_GIGANTE".COMANDOS.MARCHA OR "DB ENROLADOR_GIGANTE".COMANDOS.CONTROLE_INDEPENDENTE);
   IF #_w1 AND NOT "I405" THEN "DB ENROLADOR_GIGANTE".COMANDOS.SINC_INDEP := TRUE; END_IF;
   IF #_w1 AND "I405" THEN "DB ENROLADOR_GIGANTE".COMANDOS.SINC_INDEP := FALSE; END_IF;
   IF "DB PRINCIPAL".AUXILIARES.SEMPRE_1 AND "DB ENROLADOR_GIGANTE".COMANDOS.TROCA_ROLO AND NOT "I403" THEN
       "DB ENROLADOR_GIGANTE".COMANDOS.SINC_INDEP := FALSE;
       "DB ENROLADOR_GIGANTE".COMANDOS.TROCA_ROLO := FALSE;
   END_IF;
END_REGION

REGION Network 11: COMANDO INDEPENDENTE
   // LÓGICA DE LIGA / DESLIGA O ENROLADOR GIGANTE EM MODO INDEPENDENTE.
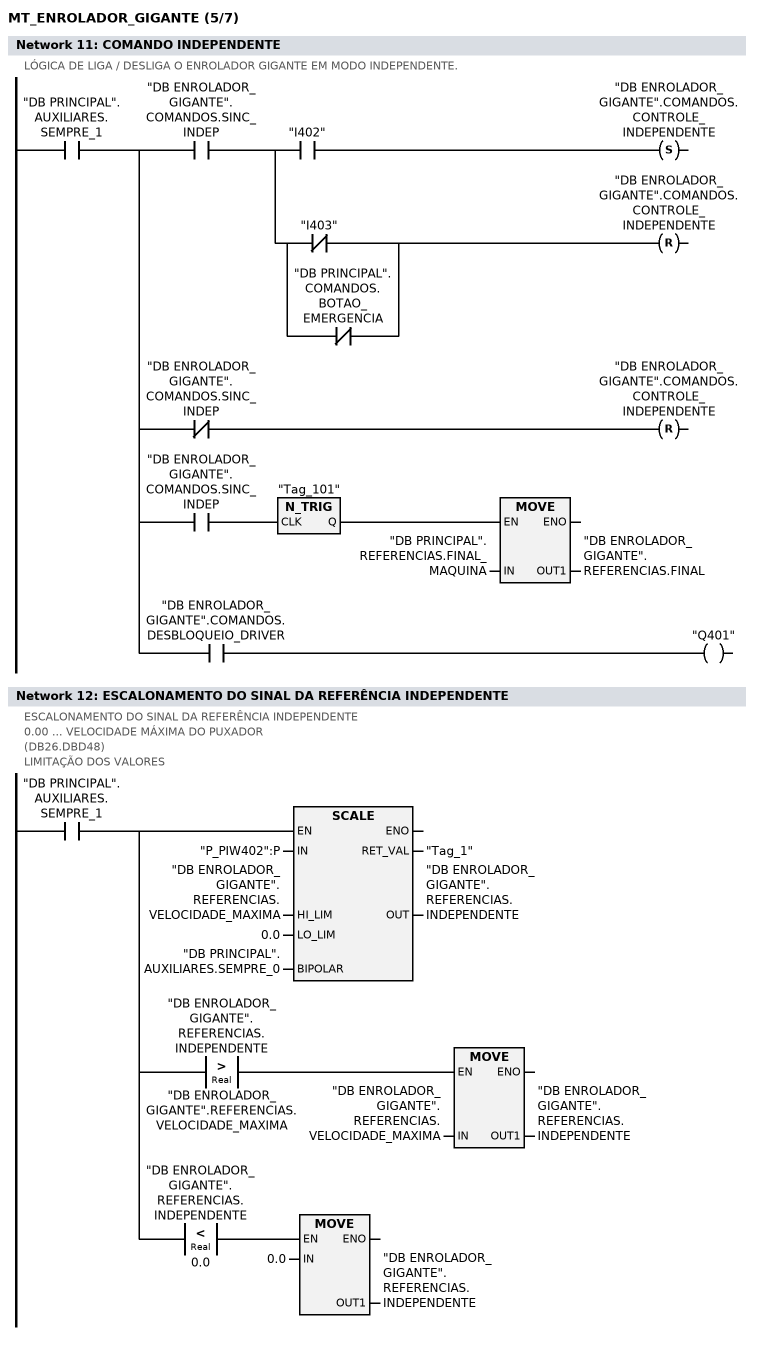
   RUNG wire#powerrail
      Contact( "DB PRINCIPAL".AUXILIARES.SEMPRE_1 )
      wire#w1
      Contact( "DB ENROLADOR_GIGANTE".COMANDOS.SINC_INDEP )
      wire#w2
      Contact( "I402" )
      S_Coil( "DB ENROLADOR_GIGANTE".COMANDOS.CONTROLE_INDEPENDENTE )
   END_RUNG
   RUNG wire#w2
      I_Contact( "I403" )
      wire#w3
      R_Coil( "DB ENROLADOR_GIGANTE".COMANDOS.CONTROLE_INDEPENDENTE )
   END_RUNG
   RUNG wire#w2
      I_Contact( "DB PRINCIPAL".COMANDOS.BOTAO_EMERGENCIA )
   END_RUNG wire#w3
   RUNG wire#w1
      I_Contact( "DB ENROLADOR_GIGANTE".COMANDOS.SINC_INDEP )
      R_Coil( "DB ENROLADOR_GIGANTE".COMANDOS.CONTROLE_INDEPENDENTE )
   END_RUNG
   RUNG wire#w1
      Contact( "DB ENROLADOR_GIGANTE".COMANDOS.SINC_INDEP )
      N_Trig( "Tag_101" )
      { S7_GenerateENO := "TRUE" } Move(in := "DB PRINCIPAL".REFERENCIAS.FINAL_MAQUINA, out1 => "DB ENROLADOR_GIGANTE".REFERENCIAS.FINAL)
   END_RUNG
   RUNG wire#w1
      Contact( "DB ENROLADOR_GIGANTE".COMANDOS.DESBLOQUEIO_DRIVER )
      Coil( "Q401" )
   END_RUNG
   // the same network as SCL:
   #_w1 := "DB PRINCIPAL".AUXILIARES.SEMPRE_1 AND "DB ENROLADOR_GIGANTE".COMANDOS.SINC_INDEP;
   IF #_w1 AND "I402" THEN "DB ENROLADOR_GIGANTE".COMANDOS.CONTROLE_INDEPENDENTE := TRUE; END_IF;
   IF #_w1 AND (NOT "I403" OR NOT "DB PRINCIPAL".COMANDOS.BOTAO_EMERGENCIA) THEN
       "DB ENROLADOR_GIGANTE".COMANDOS.CONTROLE_INDEPENDENTE := FALSE;
   END_IF;
   IF "DB PRINCIPAL".AUXILIARES.SEMPRE_1 AND NOT "DB ENROLADOR_GIGANTE".COMANDOS.SINC_INDEP THEN
       "DB ENROLADOR_GIGANTE".COMANDOS.CONTROLE_INDEPENDENTE := FALSE;
   END_IF;
   #_w2 := "DB PRINCIPAL".AUXILIARES.SEMPRE_1 AND "DB ENROLADOR_GIGANTE".COMANDOS.SINC_INDEP;
   #_w3 := NOT #_w2 AND "Tag_101";   // falling edge
   "Tag_101" := #_w2;
   IF #_w3 THEN "DB ENROLADOR_GIGANTE".REFERENCIAS.FINAL := "DB PRINCIPAL".REFERENCIAS.FINAL_MAQUINA; END_IF;
   "Q401" := "DB PRINCIPAL".AUXILIARES.SEMPRE_1 AND "DB ENROLADOR_GIGANTE".COMANDOS.DESBLOQUEIO_DRIVER;
END_REGION

REGION Network 12: ESCALONAMENTO DO SINAL DA REFERÊNCIA INDEPENDENTE
   // ESCALONAMENTO DO SINAL DA REFERÊNCIA INDEPENDENTE
   // 0.00 ... VELOCIDADE MÁXIMA DO PUXADOR 
   // (DB26.DBD48)
   // LIMITAÇÃO DOS VALORES
   #_w1 := "DB PRINCIPAL".AUXILIARES.SEMPRE_1;
   IF #_w1 THEN
       "Tag_1" := SCALE(IN := "P_PIW402":P,
                        HI_LIM := "DB ENROLADOR_GIGANTE".REFERENCIAS.VELOCIDADE_MAXIMA,
                        LO_LIM := 0.0,
                        BIPOLAR := "DB PRINCIPAL".AUXILIARES.SEMPRE_0,
                        OUT => "DB ENROLADOR_GIGANTE".REFERENCIAS.INDEPENDENTE);
   END_IF;
   IF #_w1 AND ("DB ENROLADOR_GIGANTE".REFERENCIAS.INDEPENDENTE > "DB ENROLADOR_GIGANTE".REFERENCIAS.VELOCIDADE_MAXIMA) THEN
       "DB ENROLADOR_GIGANTE".REFERENCIAS.INDEPENDENTE := "DB ENROLADOR_GIGANTE".REFERENCIAS.VELOCIDADE_MAXIMA;
   END_IF;
   IF #_w1 AND ("DB ENROLADOR_GIGANTE".REFERENCIAS.INDEPENDENTE < 0.0) THEN
       "DB ENROLADOR_GIGANTE".REFERENCIAS.INDEPENDENTE := 0.0;
   END_IF;
END_REGION

REGION Network 13
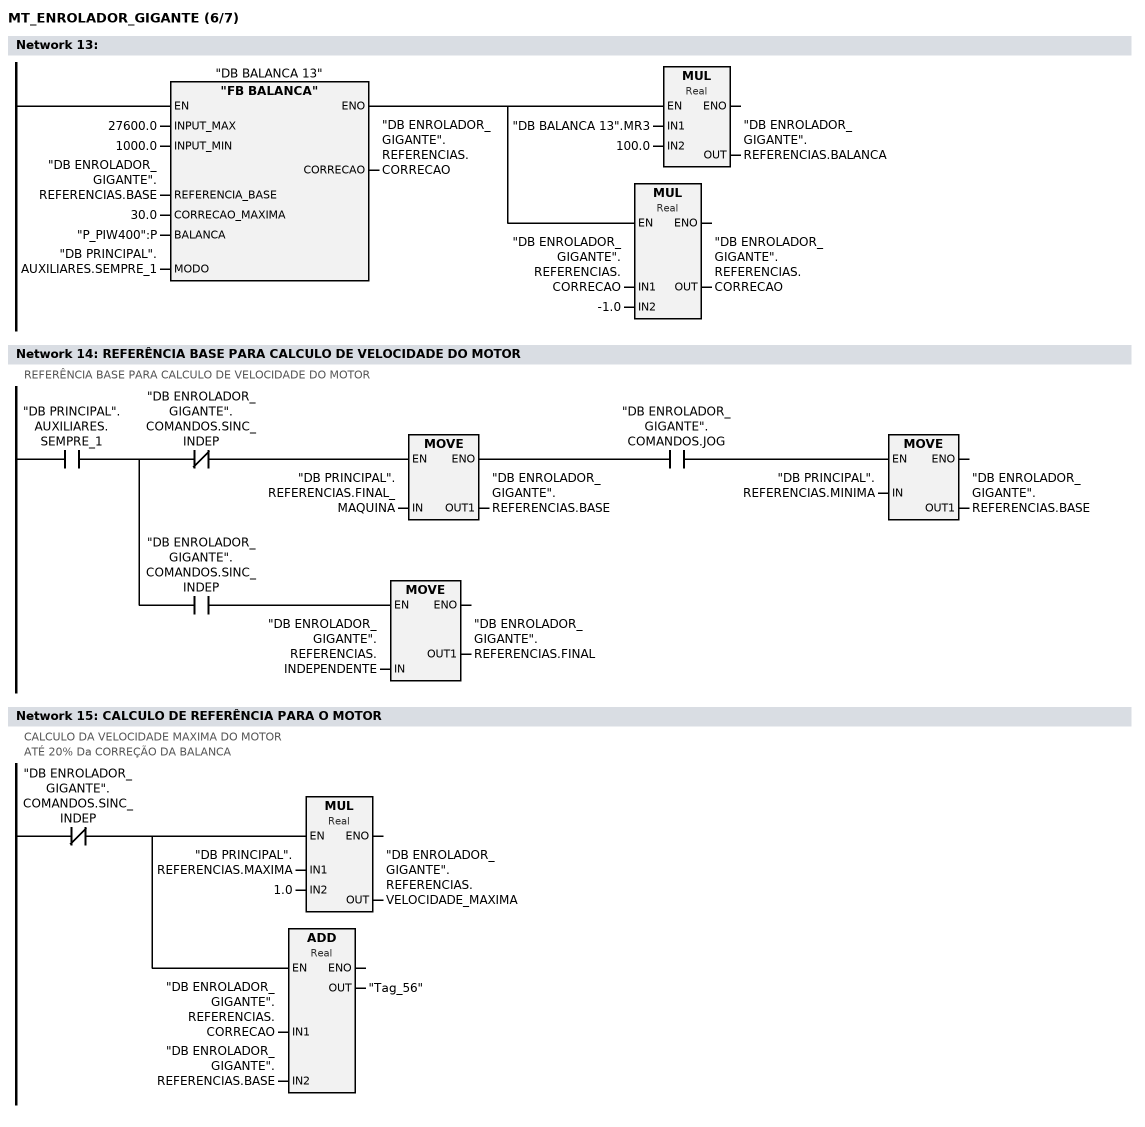
   RUNG wire#powerrail
      "DB BALANCA 13"(INPUT_MAX := 27600.0, INPUT_MIN := 1000.0, REFERENCIA_BASE := "DB ENROLADOR_GIGANTE".REFERENCIAS.BASE, CORRECAO_MAXIMA := 30.0, BALANCA := "P_PIW400":P, MODO := "DB PRINCIPAL".AUXILIARES.SEMPRE_1, CORRECAO => "DB ENROLADOR_GIGANTE".REFERENCIAS.CORRECAO)
      wire#w1
      { S7_Templates := "SrcType := Real"; S7_GenerateENO := "TRUE" } Mul(in1 := "DB BALANCA 13".MR3, in2 := 100.0, out => "DB ENROLADOR_GIGANTE".REFERENCIAS.BALANCA)
   END_RUNG
   RUNG wire#w1
      { S7_Templates := "SrcType := Real"; S7_GenerateENO := "TRUE" } Mul(in1 := "DB ENROLADOR_GIGANTE".REFERENCIAS.CORRECAO, in2 := -1.0, out => "DB ENROLADOR_GIGANTE".REFERENCIAS.CORRECAO)
   END_RUNG
   // the same network as SCL:
   "DB BALANCA 13"(INPUT_MAX := 27600.0,   // "FB BALANCA"
                   INPUT_MIN := 1000.0,
                   REFERENCIA_BASE := "DB ENROLADOR_GIGANTE".REFERENCIAS.BASE,
                   CORRECAO_MAXIMA := 30.0,
                   BALANCA := "P_PIW400":P,
                   MODO := "DB PRINCIPAL".AUXILIARES.SEMPRE_1,
                   CORRECAO => "DB ENROLADOR_GIGANTE".REFERENCIAS.CORRECAO,
                   ENO => #_w1);
   IF #_w1 THEN
       "DB ENROLADOR_GIGANTE".REFERENCIAS.BALANCA := "DB BALANCA 13".MR3 * 100.0;
       "DB ENROLADOR_GIGANTE".REFERENCIAS.CORRECAO := "DB ENROLADOR_GIGANTE".REFERENCIAS.CORRECAO * (-1.0);
   END_IF;
END_REGION

REGION Network 14: REFERÊNCIA BASE PARA CALCULO DE VELOCIDADE DO MOTOR
   // REFERÊNCIA BASE PARA CALCULO DE VELOCIDADE DO MOTOR
   RUNG wire#powerrail
      Contact( "DB PRINCIPAL".AUXILIARES.SEMPRE_1 )
      wire#w1
      I_Contact( "DB ENROLADOR_GIGANTE".COMANDOS.SINC_INDEP )
      { S7_GenerateENO := "TRUE" } Move(in := "DB PRINCIPAL".REFERENCIAS.FINAL_MAQUINA, out1 => "DB ENROLADOR_GIGANTE".REFERENCIAS.BASE)
      Contact( "DB ENROLADOR_GIGANTE".COMANDOS.JOG )
      { S7_GenerateENO := "TRUE" } Move(in := "DB PRINCIPAL".REFERENCIAS.MINIMA, out1 => "DB ENROLADOR_GIGANTE".REFERENCIAS.BASE)
   END_RUNG
   RUNG wire#w1
      Contact( "DB ENROLADOR_GIGANTE".COMANDOS.SINC_INDEP )
      { S7_GenerateENO := "TRUE" } Move(in := "DB ENROLADOR_GIGANTE".REFERENCIAS.INDEPENDENTE, out1 => "DB ENROLADOR_GIGANTE".REFERENCIAS.FINAL)
   END_RUNG
   // the same network as SCL:
   // ENO of a box is taken as its EN; it also drops when the box reports an error
   #_w1 := "DB PRINCIPAL".AUXILIARES.SEMPRE_1 AND NOT "DB ENROLADOR_GIGANTE".COMANDOS.SINC_INDEP;
   IF #_w1 THEN "DB ENROLADOR_GIGANTE".REFERENCIAS.BASE := "DB PRINCIPAL".REFERENCIAS.FINAL_MAQUINA; END_IF;
   IF #_w1 AND "DB ENROLADOR_GIGANTE".COMANDOS.JOG THEN
       "DB ENROLADOR_GIGANTE".REFERENCIAS.BASE := "DB PRINCIPAL".REFERENCIAS.MINIMA;
   END_IF;
   IF "DB PRINCIPAL".AUXILIARES.SEMPRE_1 AND "DB ENROLADOR_GIGANTE".COMANDOS.SINC_INDEP THEN
       "DB ENROLADOR_GIGANTE".REFERENCIAS.FINAL := "DB ENROLADOR_GIGANTE".REFERENCIAS.INDEPENDENTE;
   END_IF;
END_REGION

REGION Network 15: CALCULO DE REFERÊNCIA PARA O MOTOR
   // CALCULO DA VELOCIDADE MAXIMA DO MOTOR
   // ATÉ 20% Da CORREÇÃO DA BALANCA
   RUNG wire#powerrail
      I_Contact( "DB ENROLADOR_GIGANTE".COMANDOS.SINC_INDEP )
      wire#w1
      { S7_Templates := "SrcType := Real"; S7_GenerateENO := "TRUE" } Mul(in1 := "DB PRINCIPAL".REFERENCIAS.MAXIMA, in2 := 1.0, out => "DB ENROLADOR_GIGANTE".REFERENCIAS.VELOCIDADE_MAXIMA)
   END_RUNG
   RUNG wire#w1
      { S7_Templates := "SrcType := Real"; S7_GenerateENO := "TRUE" } Add(in1 := "DB ENROLADOR_GIGANTE".REFERENCIAS.CORRECAO, in2 := "DB ENROLADOR_GIGANTE".REFERENCIAS.BASE, out => "Tag_56")
   END_RUNG
   // the same network as SCL:
   IF NOT "DB ENROLADOR_GIGANTE".COMANDOS.SINC_INDEP THEN
       "DB ENROLADOR_GIGANTE".REFERENCIAS.VELOCIDADE_MAXIMA := "DB PRINCIPAL".REFERENCIAS.MAXIMA * 1.0;
       "Tag_56" := "DB ENROLADOR_GIGANTE".REFERENCIAS.CORRECAO + "DB ENROLADOR_GIGANTE".REFERENCIAS.BASE;
   END_IF;
END_REGION

REGION Network 16: ACC/DEC DA REFERÊNCIA DO MOTOR
   // ACC/DEC DA REFERÊNCIA DO MOTOR
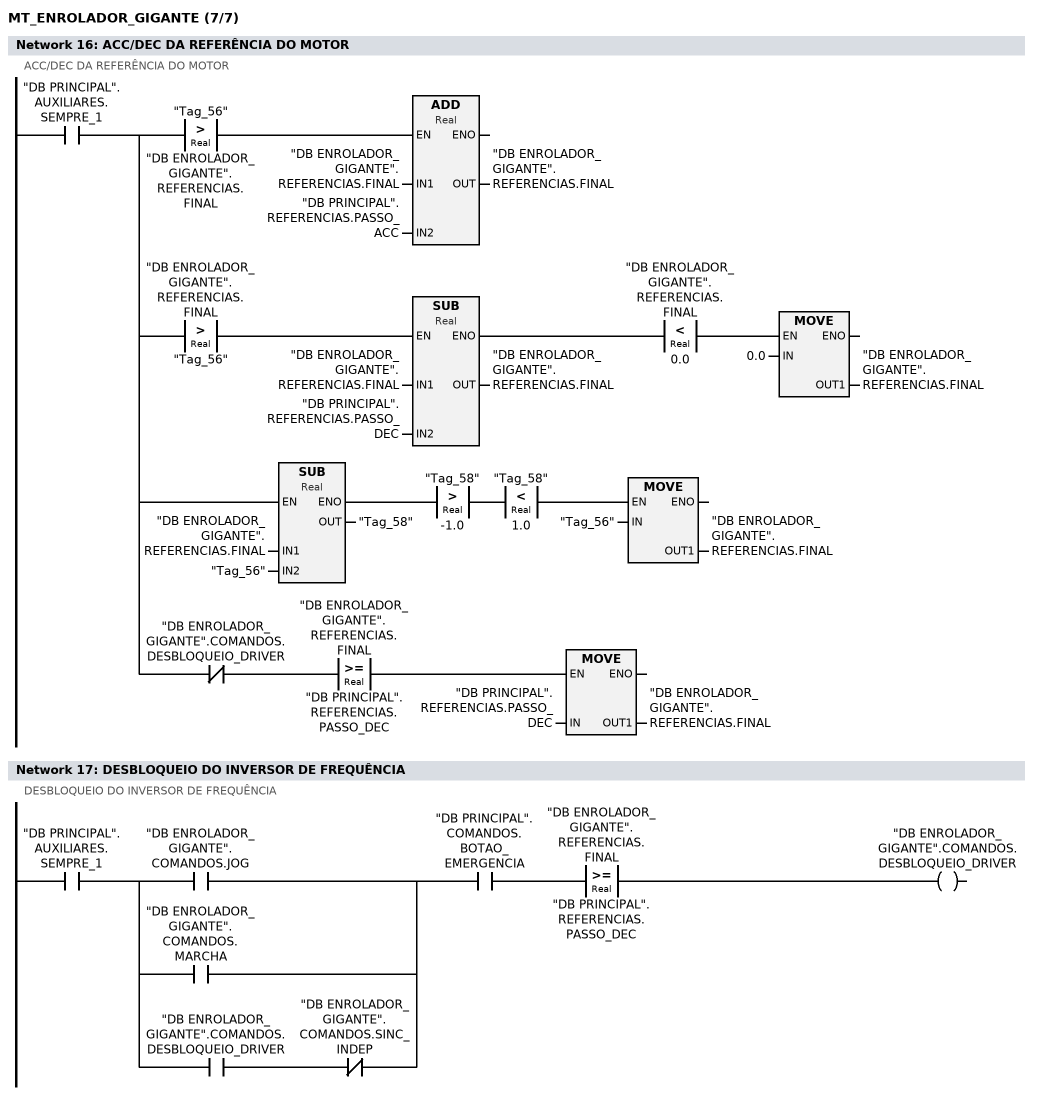
   RUNG wire#powerrail
      Contact( "DB PRINCIPAL".AUXILIARES.SEMPRE_1 )
      wire#w1
      { S7_Templates := "SrcType := Real" } GT_Contact(in1 := "Tag_56", in2 := "DB ENROLADOR_GIGANTE".REFERENCIAS.FINAL)
      { S7_Templates := "SrcType := Real"; S7_GenerateENO := "TRUE" } Add(in1 := "DB ENROLADOR_GIGANTE".REFERENCIAS.FINAL, in2 := "DB PRINCIPAL".REFERENCIAS.PASSO_ACC, out => "DB ENROLADOR_GIGANTE".REFERENCIAS.FINAL)
   END_RUNG
   RUNG wire#w1
      { S7_Templates := "SrcType := Real" } GT_Contact(in1 := "DB ENROLADOR_GIGANTE".REFERENCIAS.FINAL, in2 := "Tag_56")
      { S7_Templates := "SrcType := Real"; S7_GenerateENO := "TRUE" } Sub(in1 := "DB ENROLADOR_GIGANTE".REFERENCIAS.FINAL, in2 := "DB PRINCIPAL".REFERENCIAS.PASSO_DEC, out => "DB ENROLADOR_GIGANTE".REFERENCIAS.FINAL)
      { S7_Templates := "SrcType := Real" } LT_Contact(in1 := "DB ENROLADOR_GIGANTE".REFERENCIAS.FINAL, in2 := 0.0)
      { S7_GenerateENO := "TRUE" } Move(in := 0.0, out1 => "DB ENROLADOR_GIGANTE".REFERENCIAS.FINAL)
   END_RUNG
   RUNG wire#w1
      { S7_Templates := "SrcType := Real"; S7_GenerateENO := "TRUE" } Sub(in1 := "DB ENROLADOR_GIGANTE".REFERENCIAS.FINAL, in2 := "Tag_56", out => "Tag_58")
      { S7_Templates := "SrcType := Real" } GT_Contact(in1 := "Tag_58", in2 := -1.0)
      { S7_Templates := "SrcType := Real" } LT_Contact(in1 := "Tag_58", in2 := 1.0)
      { S7_GenerateENO := "TRUE" } Move(in := "Tag_56", out1 => "DB ENROLADOR_GIGANTE".REFERENCIAS.FINAL)
   END_RUNG
   RUNG wire#w1
      I_Contact( "DB ENROLADOR_GIGANTE".COMANDOS.DESBLOQUEIO_DRIVER )
      { S7_Templates := "SrcType := Real" } GE_Contact(in1 := "DB ENROLADOR_GIGANTE".REFERENCIAS.FINAL, in2 := "DB PRINCIPAL".REFERENCIAS.PASSO_DEC)
      { S7_GenerateENO := "TRUE" } Move(in := "DB PRINCIPAL".REFERENCIAS.PASSO_DEC, out1 => "DB ENROLADOR_GIGANTE".REFERENCIAS.FINAL)
   END_RUNG
   // the same network as SCL:
   // ENO of a box is taken as its EN; it also drops when the box reports an error
   IF "DB PRINCIPAL".AUXILIARES.SEMPRE_1 AND ("Tag_56" > "DB ENROLADOR_GIGANTE".REFERENCIAS.FINAL) THEN
       "DB ENROLADOR_GIGANTE".REFERENCIAS.FINAL := "DB ENROLADOR_GIGANTE".REFERENCIAS.FINAL + "DB PRINCIPAL".REFERENCIAS.PASSO_ACC;
   END_IF;
   #_w1 := "DB PRINCIPAL".AUXILIARES.SEMPRE_1 AND ("DB ENROLADOR_GIGANTE".REFERENCIAS.FINAL > "Tag_56");
   IF #_w1 THEN
       "DB ENROLADOR_GIGANTE".REFERENCIAS.FINAL := "DB ENROLADOR_GIGANTE".REFERENCIAS.FINAL - "DB PRINCIPAL".REFERENCIAS.PASSO_DEC;
   END_IF;
   IF #_w1 AND ("DB ENROLADOR_GIGANTE".REFERENCIAS.FINAL < 0.0) THEN
       "DB ENROLADOR_GIGANTE".REFERENCIAS.FINAL := 0.0;
   END_IF;
   IF "DB PRINCIPAL".AUXILIARES.SEMPRE_1 THEN
       "Tag_58" := "DB ENROLADOR_GIGANTE".REFERENCIAS.FINAL - "Tag_56";
   END_IF;
   IF "DB PRINCIPAL".AUXILIARES.SEMPRE_1 AND ("Tag_58" > (-1.0)) AND ("Tag_58" < 1.0) THEN
       "DB ENROLADOR_GIGANTE".REFERENCIAS.FINAL := "Tag_56";
   END_IF;
   IF "DB PRINCIPAL".AUXILIARES.SEMPRE_1 AND NOT "DB ENROLADOR_GIGANTE".COMANDOS.DESBLOQUEIO_DRIVER AND ("DB ENROLADOR_GIGANTE".REFERENCIAS.FINAL >= "DB PRINCIPAL".REFERENCIAS.PASSO_DEC) THEN
       "DB ENROLADOR_GIGANTE".REFERENCIAS.FINAL := "DB PRINCIPAL".REFERENCIAS.PASSO_DEC;
   END_IF;
END_REGION

REGION Network 17: DESBLOQUEIO DO INVERSOR DE FREQUÊNCIA
   // DESBLOQUEIO DO INVERSOR DE FREQUÊNCIA
   RUNG wire#powerrail
      Contact( "DB PRINCIPAL".AUXILIARES.SEMPRE_1 )
      wire#w1
      Contact( "DB ENROLADOR_GIGANTE".COMANDOS.JOG )
      wire#w2
      Contact( "DB PRINCIPAL".COMANDOS.BOTAO_EMERGENCIA )
      { S7_Templates := "SrcType := Real" } GE_Contact(in1 := "DB ENROLADOR_GIGANTE".REFERENCIAS.FINAL, in2 := "DB PRINCIPAL".REFERENCIAS.PASSO_DEC)
      Coil( "DB ENROLADOR_GIGANTE".COMANDOS.DESBLOQUEIO_DRIVER )
   END_RUNG
   RUNG wire#w1
      Contact( "DB ENROLADOR_GIGANTE".COMANDOS.MARCHA )
   END_RUNG wire#w2
   RUNG wire#w1
      Contact( "DB ENROLADOR_GIGANTE".COMANDOS.DESBLOQUEIO_DRIVER )
      I_Contact( "DB ENROLADOR_GIGANTE".COMANDOS.SINC_INDEP )
   END_RUNG wire#w2
   // the same network as SCL:
   "DB ENROLADOR_GIGANTE".COMANDOS.DESBLOQUEIO_DRIVER := "DB PRINCIPAL".AUXILIARES.SEMPRE_1 AND ("DB ENROLADOR_GIGANTE".COMANDOS.JOG OR "DB ENROLADOR_GIGANTE".COMANDOS.MARCHA OR ("DB ENROLADOR_GIGANTE".COMANDOS.DESBLOQUEIO_DRIVER AND NOT "DB ENROLADOR_GIGANTE".COMANDOS.SINC_INDEP)) AND "DB PRINCIPAL".COMANDOS.BOTAO_EMERGENCIA AND ("DB ENROLADOR_GIGANTE".REFERENCIAS.FINAL >= "DB PRINCIPAL".REFERENCIAS.PASSO_DEC);
END_REGION

REGION Network 18 (STL): STATUS / CONTROLE - INVERSOR DE FREQUÊNCIA
   // DANFOSS FC300 PROFIBUS - TEX24626INV001
   // STATUS DO INVERSOR DE FREQUÊNCIA
         L     "Tag_48":P;
         T     "Tag_1";
         AN    "Tag_59";
         =     "DB ENROLADOR_GIGANTE".COMANDOS.STATUS_DRIVER;

   // CONTROLE DO INVERSOR DE FREQUÊNCIA
         L     1150;
         T     "Tag_1";
         A     "DB ENROLADOR_GIGANTE".COMANDOS.DESBLOQUEIO_DRIVER;
         =     "Tag_60";
         A     "T2";
         AN    "DB ENROLADOR_GIGANTE".COMANDOS.STATUS_DRIVER;
         =     "Tag_61";
         L     "Tag_1";
         T     "Tag_49":P;

   // REFERÊNCIA PARA O INVERSOR DE FREQUÊNCIA
         L     "DB ENROLADOR_GIGANTE".REFERENCIAS.FINAL;
         L     16384.0;
         *R;

         L     "DB ENROLADOR_GIGANTE".REFERENCIAS.VELOCIDADE_MAXIMA;
         /R;
         RND;
         T     "Tag_62";
         L     "Tag_62";
         T     "Tag_50":P;
END_REGION

REGION Network 19 (STL): INVERSOR RESERVA
         A     "DB PRINCIPAL".AUXILIARES.SEMPRE_1;
         =     %L24.0;
         A     %L24.0;
         A(;
         L     "DB PRINCIPAL".AUXILIARES1.INVERSOR_RESERVA1;
         L     17;
         ==I;
         );
         =     %L24.1;
         A     %L24.1;
         JNB   M002;
         L     "DB ENROLADOR_GIGANTE".REFERENCIAS.FINAL;
         L     3.456;
         *R;
         T     #AUX_R;
         RND;
         T     "P_QW100":P;
   M002: NOP   0;
         A     %L24.1;
         A     "I130";
         S     "DB PRINCIPAL".ALARME.INV_RESERVA1;
         A     %L24.1;
         A     "DB ENROLADOR_GIGANTE".COMANDOS.DESBLOQUEIO_DRIVER;
         S     "Q134";
         A     %L24.1;
         AN    "DB ENROLADOR_GIGANTE".COMANDOS.DESBLOQUEIO_DRIVER;
         R     "Q134";
         A     %L24.0;
         A(;
         L     "DB PRINCIPAL".AUXILIARES1.INVERSOR_RESERVA2;
         L     17;
         ==I;
         );
         =     %L24.1;
         A     %L24.1;
         JNB   M001;
         L     "DB ENROLADOR_GIGANTE".REFERENCIAS.FINAL;
         L     3.456;
         *R;
         T     #AUX_R;
         RND;
         T     "P_QW102":P;
   M001: NOP   0;
         A     %L24.1;
         A     "I132";
         S     "DB PRINCIPAL".ALARME.INV_RESERVA2;
         A     %L24.1;
         A     "DB ENROLADOR_GIGANTE".COMANDOS.DESBLOQUEIO_DRIVER;
         S     "Q135";
         A     %L24.1;
         AN    "DB ENROLADOR_GIGANTE".COMANDOS.DESBLOQUEIO_DRIVER;
         R     "Q135";
END_REGION
END_FUNCTION

FUNCTION "INTEGRAÇÃO LINHA" : Void   // FC100, LAD
TITLE = MÓDULO DE CONTROLE DA INTERLIGAÇÃO DA LINHA COM A SANFORIZADEIRA
{ S7_Optimized_Access := 'FALSE' }
AUTHOR : ANDERSON
FAMILY : OS:24626
NAME : SANFOR
VERSION : 0.1
// DATA BLOCK DE CONTROLE // DB100
// Automation Pack Automação Indl. e Com. Ltda.
// Cliente: Texima S/A Ind. de Máquinas
// Cliente Final: Cia. Fiação e Tecidos Santo Antonio.
// Máquina: Sanforizadeira da Linha Integrada 1 - O.S.: 24.626
BEGIN

REGION Network 1 (STL): VARIÁVEIS TRANSMITIDAS COMUNS AS MÁQUINAS
   // ALOCAÇÃO DAS VARIÁVEIS QUE SERAM TRANSMITIDAS NA DB DE TRANSMIÇÃO
         A     "DB PRINCIPAL".COMANDOS.BOTAO_LIGA;
         =     "DB VALORES TRANSMITIDOS".VARIAVEIS_COMPARTILHADAS.DIGITAIS.LIGA_MAQUINA;
         A     "DB PRINCIPAL".COMANDOS.BOTAO_DESLIGA;
         =     "DB VALORES TRANSMITIDOS".VARIAVEIS_COMPARTILHADAS.DIGITAIS.DESLIGA_MAQUINA;
         A     "DB PRINCIPAL".COMANDOS.BOTAO_EMERGENCIA;
         =     "DB VALORES TRANSMITIDOS".VARIAVEIS_COMPARTILHADAS.DIGITAIS.EMERGENCIA_GERAL;
         A     "DB PRINCIPAL".COMANDOS.BOTAO_JOG;
         =     "DB VALORES TRANSMITIDOS".VARIAVEIS_COMPARTILHADAS.DIGITAIS.JOG_GERAL;
         A     "I306";
         =     "DB VALORES TRANSMITIDOS".VARIAVEIS_COMPARTILHADAS.DIGITAIS.TRAVA_BALANCA;
         A     "I307";
         =     "DB VALORES TRANSMITIDOS".VARIAVEIS_COMPARTILHADAS.DIGITAIS.DESTRAVA_ALARME;
         A     "I323";
         =     "DB VALORES TRANSMITIDOS".VARIAVEIS_COMPARTILHADAS.DIGITAIS.PRESSOSTATO_MAQUINA;
         A     "DB PRINCIPAL".COMANDOS.ALARME_ALTO;
         =     "DB VALORES TRANSMITIDOS".VARIAVEIS_COMPARTILHADAS.DIGITAIS.ALARME_ALTO;
         A     "DB PRINCIPAL".COMANDOS.ALARME_BAIXO;
         =     "DB VALORES TRANSMITIDOS".VARIAVEIS_COMPARTILHADAS.DIGITAIS.ALARME_BAIXO;
         A     "DB PRINCIPAL".COMANDOS.BALANCA_FORA_POSICAO;
         =     "DB VALORES TRANSMITIDOS".VARIAVEIS_COMPARTILHADAS.DIGITAIS.BALANCA_FORA_POSICAO;
         A     "DB PRINCIPAL".COMANDOS.MARCHA;
         =     "DB VALORES TRANSMITIDOS".VARIAVEIS_COMPARTILHADAS.DIGITAIS.MARCHA;
         A     "DB PRINCIPAL".COMANDOS.AUX_MARCHA;
         =     "DB VALORES TRANSMITIDOS".VARIAVEIS_COMPARTILHADAS.DIGITAIS.AUX_MARCHA;
         A     "DB PRINCIPAL".COMANDOS.MOTOR_SELECIONADO;
         =     "DB VALORES TRANSMITIDOS".VARIAVEIS_COMPARTILHADAS.DIGITAIS.MOTOR_SELECIONADO;
END_REGION

REGION Network 2 (STL): VARIAVEIS TRANSMITIDAS DA LINHA PARA A SANFOR
   // ALOCAÇÃO DAS VARIÁVEIS QUE SERAM TRANSMITIDAS NA DB DE TRANSMIÇÃO
         L     "DB PRINCIPAL".REFERENCIAS.BASE;
         T     "DB VALORES TRANSMITIDOS".VARIAVEIS_LINHA.ANALOGICAS.REFERENCIA_BASE_LINHA;
         L     "P_PIW400":P;
         T     "DB VALORES TRANSMITIDOS".VARIAVEIS_LINHA.ANALOGICAS.POSICAO_REAL_BALANCA;
END_REGION
END_FUNCTION

ORGANIZATION_BLOCK "PRINCIPAL"   // OB1, LAD
TITLE = MÓDULO PRINCIPAL
{ S7_Optimized_Access := 'FALSE' }
AUTHOR : THALLES
FAMILY : MÁQUINA
NAME : LINHA1
VERSION : 0.1
// DATA BLOCK DE CONTROLE // DB1
// Automation Pack Automação Indl. e Com. Ltda.
// Cliente: Texima S/A Ind. de Máquinas
// Cliente Final: Cia. Fiação e Tecidos Santo Antonio.
// Máquina: LINHA 1 DENIN - O.S.: 24.626
   VAR_TEMP
      OB1_EV_CLASS : Byte;   // Bits 0-3 = 1 (Coming event), Bits 4-7 = 1 (Event class 1)
      OB1_SCAN_1 : Byte;   // 1 (Cold restart scan 1 of OB 1), 3 (Scan 2-n of OB 1)
      OB1_PRIORITY : Byte;   // Priority of OB Execution
      OB1_OB_NUMBR : Byte;   // 1 (Organization block 1, OB1)
      OB1_RESERVED_1 : Byte;   // Reserved for system
      OB1_RESERVED_2 : Byte;   // Reserved for system
      OB1_PREV_CYCLE : Int;   // Cycle time of previous OB1 scan (milliseconds)
      OB1_MIN_CYCLE : Int;   // Minimum cycle time of OB1 (milliseconds)
      OB1_MAX_CYCLE : Int;   // Maximum cycle time of OB1 (milliseconds)
      OB1_DATE_TIME : Date_And_Time;   // Date and time OB1 started
      AUX_R : Real;
   END_VAR
   VAR_TEMP   // added for the SCL form of the ladder/FBD networks
      _w1 : Bool;
      _s5time1 : S5Time;
      _w2 : Bool;
      _w3 : Bool;
      _w4 : Bool;
   END_VAR
BEGIN

REGION Network 1: CHAMA LOGICA DE LEITURA DOS VALORES DA INTEGRAÇÃO DA REDE
   // CONEXÃO MERGE PROFINET ENTRE AS CPU'S LINHA E SANFORIZADEIRA ONDE A 
   // SANFORIZADEIRA CONTROLA A COMUNICAÇÃO E A LINHA CONTROLA AS VARIAVEIS (EXEMPLO 
   // VELOCIDADE DO CONJUNTO)
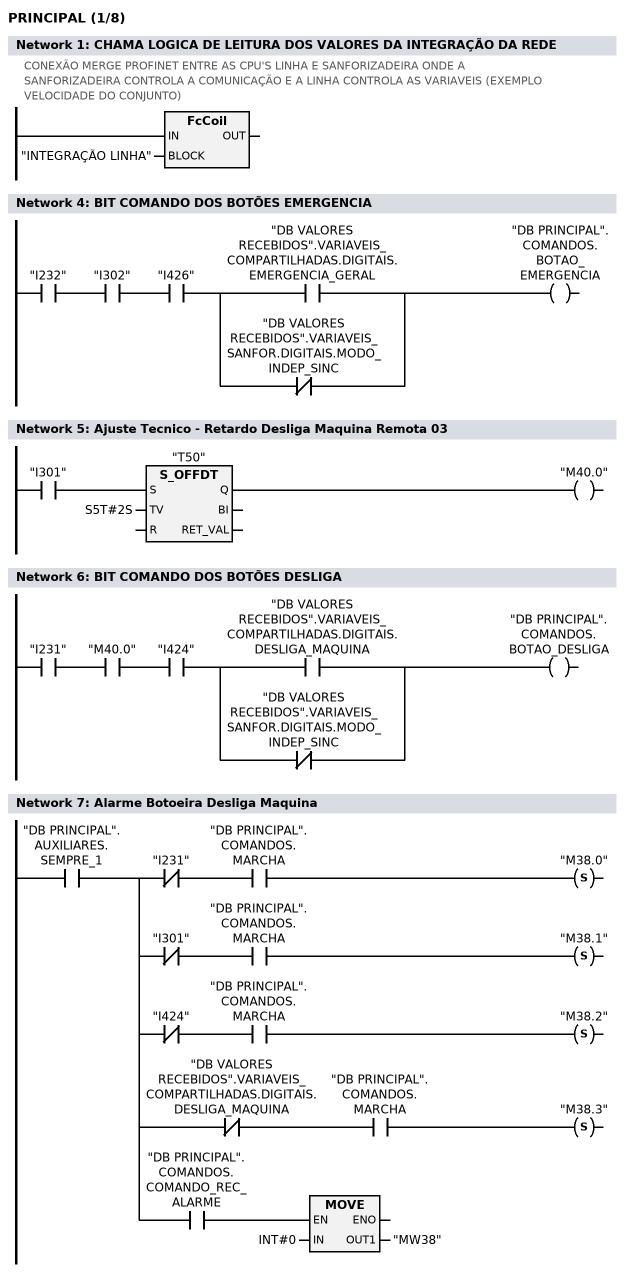
   // no SCL statement known for FcCoil: written as a call
   FcCoil(block := "INTEGRAÇÃO LINHA", in := TRUE);
END_REGION

REGION Network 2 (STL): BIT´S DE USO GERAL
   // BIT SEMPRE DESLIGADO
   // BIT SEMPRE LIGADO
         CLR;
         =     "DB PRINCIPAL".AUXILIARES.SEMPRE_0;
         SET;
         =     "DB PRINCIPAL".AUXILIARES.SEMPRE_1;
         NOP   0;
END_REGION

REGION Network 3 (STL): BIT´S DE USO GERAL
   // MUDA DE ESTADO A CADA SCAN
   // MUDA DE ESTADO À CADA  50ms - PERIODO 100MS
   // MUDA DE ESTADO A CADA 250ms - PERIODO 500MS
   // MUDA DE ESTADO A CADA 500ms - PERIODO 1S
         AN    "DB PRINCIPAL".AUXILIARES.BASE_1_SCAN;
         =     "DB PRINCIPAL".AUXILIARES.BASE_1_SCAN;
         A     "Tag_102";
         =     "DB PRINCIPAL".AUXILIARES.BASE_100MS;
         A     "Tag_103";
         =     "DB PRINCIPAL".AUXILIARES.BASE_500MS;
         A     "Tag_104";
         =     "DB PRINCIPAL".AUXILIARES.BASE_1S;
         NOP   0;
END_REGION

REGION Network 4: BIT COMANDO DOS BOTÕES EMERGENCIA
   RUNG wire#powerrail
      Contact( "I232" )
      Contact( "I302" )
      Contact( "I426" )
      wire#w1
      Contact( "DB VALORES RECEBIDOS".VARIAVEIS_COMPARTILHADAS.DIGITAIS.EMERGENCIA_GERAL )
      wire#w2
      Coil( "DB PRINCIPAL".COMANDOS.BOTAO_EMERGENCIA )
   END_RUNG
   RUNG wire#w1
      I_Contact( "DB VALORES RECEBIDOS".VARIAVEIS_SANFOR.DIGITAIS.MODO_INDEP_SINC )
   END_RUNG wire#w2
   // the same network as SCL:
   "DB PRINCIPAL".COMANDOS.BOTAO_EMERGENCIA := "I232" AND "I302" AND "I426" AND ("DB VALORES RECEBIDOS".VARIAVEIS_COMPARTILHADAS.DIGITAIS.EMERGENCIA_GERAL OR NOT "DB VALORES RECEBIDOS".VARIAVEIS_SANFOR.DIGITAIS.MODO_INDEP_SINC);
END_REGION

REGION Network 5: Ajuste Tecnico - Retardo Desliga Maquina Remota 03
   RUNG wire#powerrail
      Contact( "I301" )
      S_OFFDT(T_NO := "T50", TV := S5T#2S, R :=, BI =>, RET_VAL =>)
      Coil( "M40.0" )
   END_RUNG
   // the same network as SCL:
   #_s5time1 := S_OFFDT(T_NO := "T50", TV := S5T#2S, S := "I301", Q => #_w1);
   "M40.0" := #_w1;
END_REGION

REGION Network 6: BIT COMANDO DOS BOTÕES DESLIGA
   RUNG wire#powerrail
      Contact( "I231" )
      Contact( "M40.0" )
      Contact( "I424" )
      wire#w1
      Contact( "DB VALORES RECEBIDOS".VARIAVEIS_COMPARTILHADAS.DIGITAIS.DESLIGA_MAQUINA )
      wire#w2
      Coil( "DB PRINCIPAL".COMANDOS.BOTAO_DESLIGA )
   END_RUNG
   RUNG wire#w1
      I_Contact( "DB VALORES RECEBIDOS".VARIAVEIS_SANFOR.DIGITAIS.MODO_INDEP_SINC )
   END_RUNG wire#w2
   // the same network as SCL:
   "DB PRINCIPAL".COMANDOS.BOTAO_DESLIGA := "I231" AND "M40.0" AND "I424" AND ("DB VALORES RECEBIDOS".VARIAVEIS_COMPARTILHADAS.DIGITAIS.DESLIGA_MAQUINA OR NOT "DB VALORES RECEBIDOS".VARIAVEIS_SANFOR.DIGITAIS.MODO_INDEP_SINC);
END_REGION

REGION Network 7: Alarme Botoeira Desliga Maquina
   RUNG wire#powerrail
      Contact( "DB PRINCIPAL".AUXILIARES.SEMPRE_1 )
      wire#w1
      I_Contact( "I231" )
      Contact( "DB PRINCIPAL".COMANDOS.MARCHA )
      S_Coil( "M38.0" )
   END_RUNG
   RUNG wire#w1
      I_Contact( "I301" )
      Contact( "DB PRINCIPAL".COMANDOS.MARCHA )
      S_Coil( "M38.1" )
   END_RUNG
   RUNG wire#w1
      I_Contact( "I424" )
      Contact( "DB PRINCIPAL".COMANDOS.MARCHA )
      S_Coil( "M38.2" )
   END_RUNG
   RUNG wire#w1
      I_Contact( "DB VALORES RECEBIDOS".VARIAVEIS_COMPARTILHADAS.DIGITAIS.DESLIGA_MAQUINA )
      Contact( "DB PRINCIPAL".COMANDOS.MARCHA )
      S_Coil( "M38.3" )
   END_RUNG
   RUNG wire#w1
      Contact( "DB PRINCIPAL".COMANDOS.COMANDO_REC_ALARME )
      { S7_GenerateENO := "TRUE" } Move(in := INT#0, out1 => "MW38")
   END_RUNG
   // the same network as SCL:
   IF "DB PRINCIPAL".AUXILIARES.SEMPRE_1 AND NOT "I231" AND "DB PRINCIPAL".COMANDOS.MARCHA THEN
       "M38.0" := TRUE;
   END_IF;
   IF "DB PRINCIPAL".AUXILIARES.SEMPRE_1 AND NOT "I301" AND "DB PRINCIPAL".COMANDOS.MARCHA THEN
       "M38.1" := TRUE;
   END_IF;
   IF "DB PRINCIPAL".AUXILIARES.SEMPRE_1 AND NOT "I424" AND "DB PRINCIPAL".COMANDOS.MARCHA THEN
       "M38.2" := TRUE;
   END_IF;
   IF "DB PRINCIPAL".AUXILIARES.SEMPRE_1 AND NOT "DB VALORES RECEBIDOS".VARIAVEIS_COMPARTILHADAS.DIGITAIS.DESLIGA_MAQUINA AND "DB PRINCIPAL".COMANDOS.MARCHA THEN
       "M38.3" := TRUE;
   END_IF;
   IF "DB PRINCIPAL".AUXILIARES.SEMPRE_1 AND "DB PRINCIPAL".COMANDOS.COMANDO_REC_ALARME THEN
       "MW38" := INT#0;
   END_IF;
END_REGION

REGION Network 8: BIT COMANDO DOS BOTÕES JOG
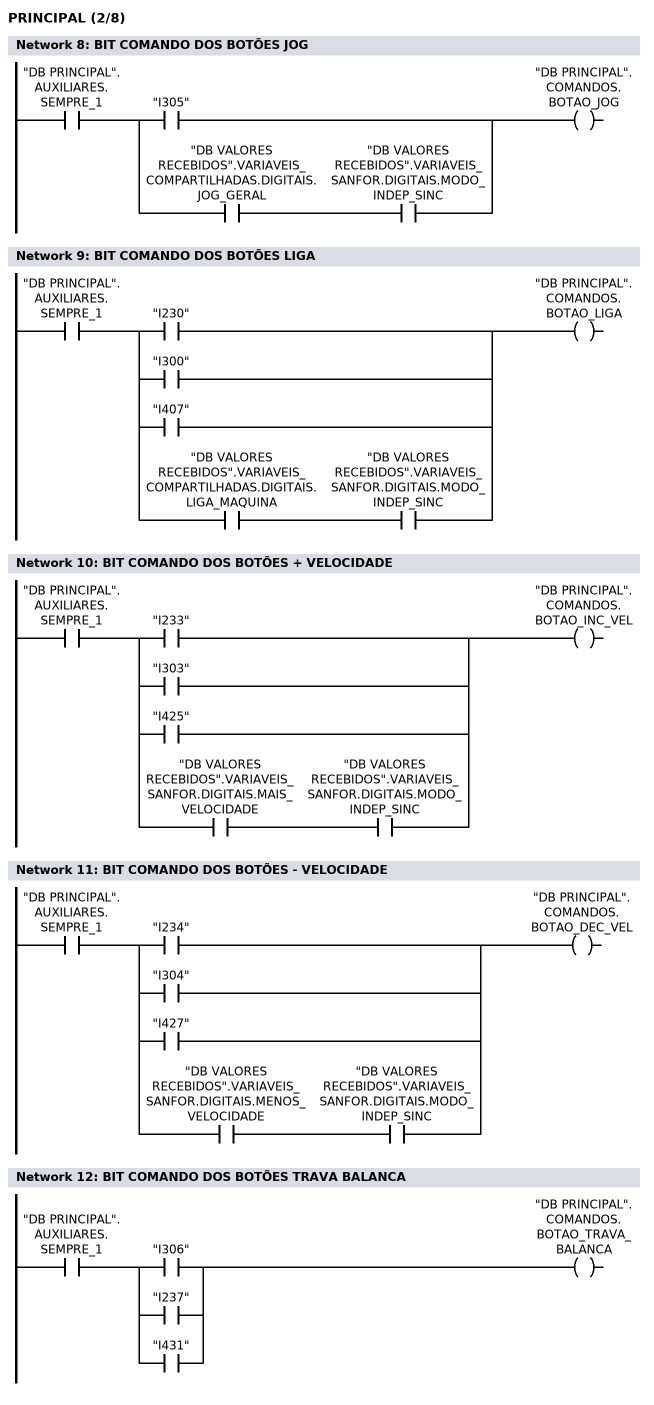
   RUNG wire#powerrail
      Contact( "DB PRINCIPAL".AUXILIARES.SEMPRE_1 )
      wire#w1
      Contact( "I305" )
      wire#w2
      Coil( "DB PRINCIPAL".COMANDOS.BOTAO_JOG )
   END_RUNG
   RUNG wire#w1
      Contact( "DB VALORES RECEBIDOS".VARIAVEIS_COMPARTILHADAS.DIGITAIS.JOG_GERAL )
      Contact( "DB VALORES RECEBIDOS".VARIAVEIS_SANFOR.DIGITAIS.MODO_INDEP_SINC )
   END_RUNG wire#w2
   // the same network as SCL:
   "DB PRINCIPAL".COMANDOS.BOTAO_JOG := "DB PRINCIPAL".AUXILIARES.SEMPRE_1 AND ("I305" OR ("DB VALORES RECEBIDOS".VARIAVEIS_COMPARTILHADAS.DIGITAIS.JOG_GERAL AND "DB VALORES RECEBIDOS".VARIAVEIS_SANFOR.DIGITAIS.MODO_INDEP_SINC));
END_REGION

REGION Network 9: BIT COMANDO DOS BOTÕES LIGA
   RUNG wire#powerrail
      Contact( "DB PRINCIPAL".AUXILIARES.SEMPRE_1 )
      wire#w1
      Contact( "I230" )
      wire#w2
      Coil( "DB PRINCIPAL".COMANDOS.BOTAO_LIGA )
   END_RUNG
   RUNG wire#w1
      Contact( "I300" )
   END_RUNG wire#w2
   RUNG wire#w1
      Contact( "I407" )
   END_RUNG wire#w2
   RUNG wire#w1
      Contact( "DB VALORES RECEBIDOS".VARIAVEIS_COMPARTILHADAS.DIGITAIS.LIGA_MAQUINA )
      Contact( "DB VALORES RECEBIDOS".VARIAVEIS_SANFOR.DIGITAIS.MODO_INDEP_SINC )
   END_RUNG wire#w2
   // the same network as SCL:
   "DB PRINCIPAL".COMANDOS.BOTAO_LIGA := "DB PRINCIPAL".AUXILIARES.SEMPRE_1 AND ("I230" OR "I300" OR "I407" OR ("DB VALORES RECEBIDOS".VARIAVEIS_COMPARTILHADAS.DIGITAIS.LIGA_MAQUINA AND "DB VALORES RECEBIDOS".VARIAVEIS_SANFOR.DIGITAIS.MODO_INDEP_SINC));
END_REGION

REGION Network 10: BIT COMANDO DOS BOTÕES + VELOCIDADE
   RUNG wire#powerrail
      Contact( "DB PRINCIPAL".AUXILIARES.SEMPRE_1 )
      wire#w1
      Contact( "I233" )
      wire#w2
      Coil( "DB PRINCIPAL".COMANDOS.BOTAO_INC_VEL )
   END_RUNG
   RUNG wire#w1
      Contact( "I303" )
   END_RUNG wire#w2
   RUNG wire#w1
      Contact( "I425" )
   END_RUNG wire#w2
   RUNG wire#w1
      Contact( "DB VALORES RECEBIDOS".VARIAVEIS_SANFOR.DIGITAIS.MAIS_VELOCIDADE )
      Contact( "DB VALORES RECEBIDOS".VARIAVEIS_SANFOR.DIGITAIS.MODO_INDEP_SINC )
   END_RUNG wire#w2
   // the same network as SCL:
   "DB PRINCIPAL".COMANDOS.BOTAO_INC_VEL := "DB PRINCIPAL".AUXILIARES.SEMPRE_1 AND ("I233" OR "I303" OR "I425" OR ("DB VALORES RECEBIDOS".VARIAVEIS_SANFOR.DIGITAIS.MAIS_VELOCIDADE AND "DB VALORES RECEBIDOS".VARIAVEIS_SANFOR.DIGITAIS.MODO_INDEP_SINC));
END_REGION

REGION Network 11: BIT COMANDO DOS BOTÕES - VELOCIDADE
   RUNG wire#powerrail
      Contact( "DB PRINCIPAL".AUXILIARES.SEMPRE_1 )
      wire#w1
      Contact( "I234" )
      wire#w2
      Coil( "DB PRINCIPAL".COMANDOS.BOTAO_DEC_VEL )
   END_RUNG
   RUNG wire#w1
      Contact( "I304" )
   END_RUNG wire#w2
   RUNG wire#w1
      Contact( "I427" )
   END_RUNG wire#w2
   RUNG wire#w1
      Contact( "DB VALORES RECEBIDOS".VARIAVEIS_SANFOR.DIGITAIS.MENOS_VELOCIDADE )
      Contact( "DB VALORES RECEBIDOS".VARIAVEIS_SANFOR.DIGITAIS.MODO_INDEP_SINC )
   END_RUNG wire#w2
   // the same network as SCL:
   "DB PRINCIPAL".COMANDOS.BOTAO_DEC_VEL := "DB PRINCIPAL".AUXILIARES.SEMPRE_1 AND ("I234" OR "I304" OR "I427" OR ("DB VALORES RECEBIDOS".VARIAVEIS_SANFOR.DIGITAIS.MENOS_VELOCIDADE AND "DB VALORES RECEBIDOS".VARIAVEIS_SANFOR.DIGITAIS.MODO_INDEP_SINC));
END_REGION

REGION Network 12: BIT COMANDO DOS BOTÕES TRAVA BALANCA
   RUNG wire#powerrail
      Contact( "DB PRINCIPAL".AUXILIARES.SEMPRE_1 )
      wire#w1
      Contact( "I306" )
      wire#w2
      Coil( "DB PRINCIPAL".COMANDOS.BOTAO_TRAVA_BALANCA )
   END_RUNG
   RUNG wire#w1
      Contact( "I237" )
   END_RUNG wire#w2
   RUNG wire#w1
      Contact( "I431" )
   END_RUNG wire#w2
   // the same network as SCL:
   "DB PRINCIPAL".COMANDOS.BOTAO_TRAVA_BALANCA := "DB PRINCIPAL".AUXILIARES.SEMPRE_1 AND ("I306" OR "I237" OR "I431");
END_REGION

REGION Network 13: BIT COMANDO DOS BOTÕES SIRENE
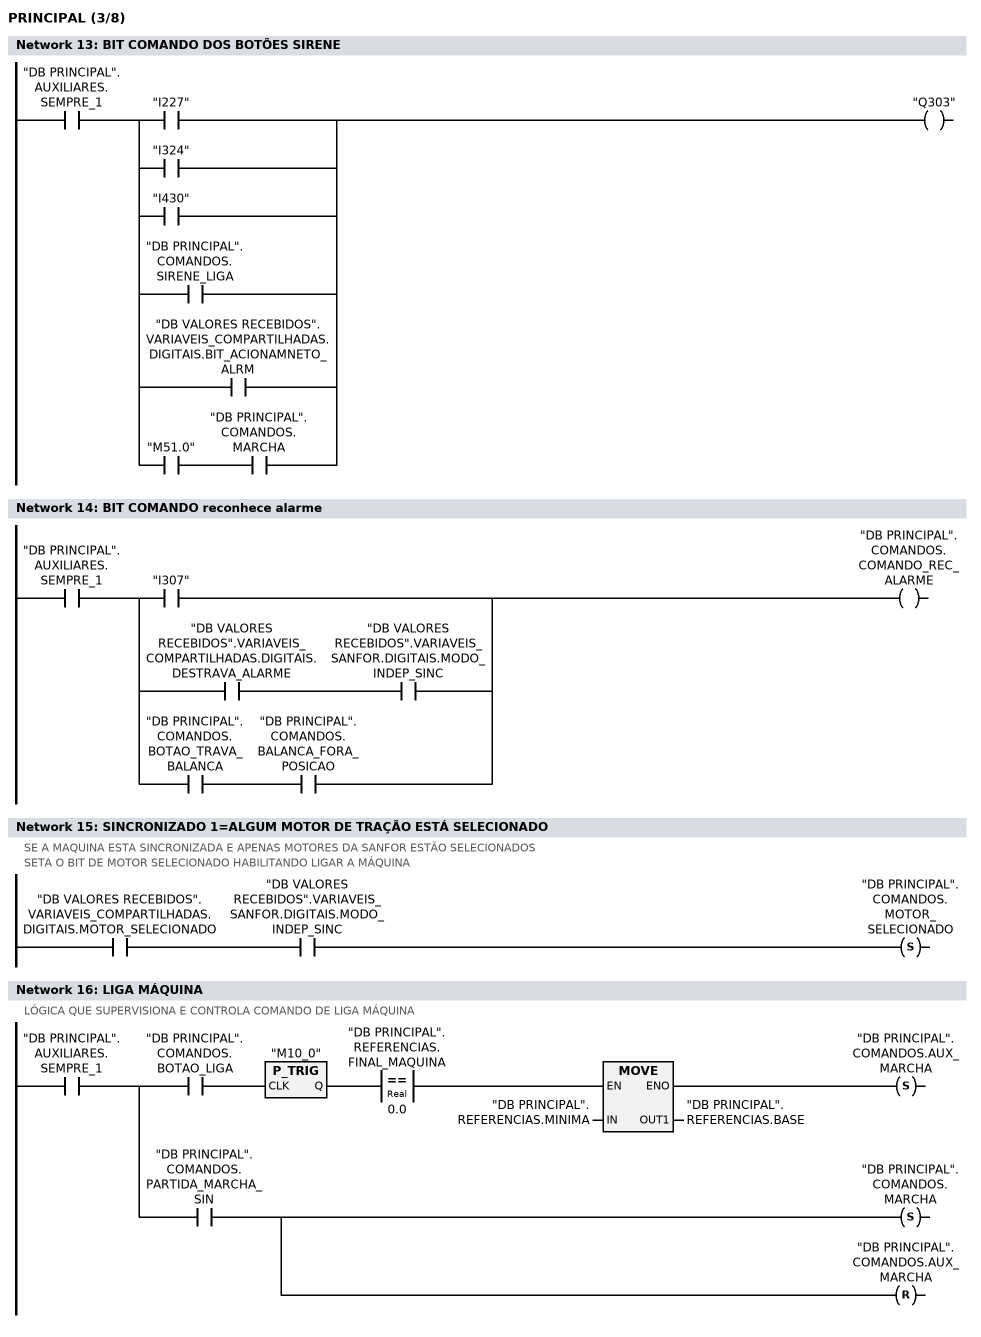
   RUNG wire#powerrail
      Contact( "DB PRINCIPAL".AUXILIARES.SEMPRE_1 )
      wire#w1
      Contact( "I227" )
      wire#w2
      Coil( "Q303" )
   END_RUNG
   RUNG wire#w1
      Contact( "I324" )
   END_RUNG wire#w2
   RUNG wire#w1
      Contact( "I430" )
   END_RUNG wire#w2
   RUNG wire#w1
      Contact( "DB PRINCIPAL".COMANDOS.SIRENE_LIGA )
   END_RUNG wire#w2
   RUNG wire#w1
      Contact( "DB VALORES RECEBIDOS".VARIAVEIS_COMPARTILHADAS.DIGITAIS.BIT_ACIONAMNETO_ALRM )
   END_RUNG wire#w2
   RUNG wire#w1
      Contact( "M51.0" )
      Contact( "DB PRINCIPAL".COMANDOS.MARCHA )
   END_RUNG wire#w2
   // the same network as SCL:
   "Q303" := "DB PRINCIPAL".AUXILIARES.SEMPRE_1 AND ("I227" OR "I324" OR "I430" OR "DB PRINCIPAL".COMANDOS.SIRENE_LIGA OR "DB VALORES RECEBIDOS".VARIAVEIS_COMPARTILHADAS.DIGITAIS.BIT_ACIONAMNETO_ALRM OR ("M51.0" AND "DB PRINCIPAL".COMANDOS.MARCHA));
END_REGION

REGION Network 14: BIT COMANDO reconhece alarme
   RUNG wire#powerrail
      Contact( "DB PRINCIPAL".AUXILIARES.SEMPRE_1 )
      wire#w1
      Contact( "I307" )
      wire#w2
      Coil( "DB PRINCIPAL".COMANDOS.COMANDO_REC_ALARME )
   END_RUNG
   RUNG wire#w1
      Contact( "DB VALORES RECEBIDOS".VARIAVEIS_COMPARTILHADAS.DIGITAIS.DESTRAVA_ALARME )
      Contact( "DB VALORES RECEBIDOS".VARIAVEIS_SANFOR.DIGITAIS.MODO_INDEP_SINC )
   END_RUNG wire#w2
   RUNG wire#w1
      Contact( "DB PRINCIPAL".COMANDOS.BOTAO_TRAVA_BALANCA )
      Contact( "DB PRINCIPAL".COMANDOS.BALANCA_FORA_POSICAO )
   END_RUNG wire#w2
   // the same network as SCL:
   "DB PRINCIPAL".COMANDOS.COMANDO_REC_ALARME := "DB PRINCIPAL".AUXILIARES.SEMPRE_1 AND ("I307" OR ("DB VALORES RECEBIDOS".VARIAVEIS_COMPARTILHADAS.DIGITAIS.DESTRAVA_ALARME AND "DB VALORES RECEBIDOS".VARIAVEIS_SANFOR.DIGITAIS.MODO_INDEP_SINC) OR ("DB PRINCIPAL".COMANDOS.BOTAO_TRAVA_BALANCA AND "DB PRINCIPAL".COMANDOS.BALANCA_FORA_POSICAO));
END_REGION

REGION Network 15: SINCRONIZADO 1=ALGUM MOTOR DE TRAÇÃO ESTÁ SELECIONADO
   // SE A MAQUINA ESTA SINCRONIZADA E APENAS MOTORES DA SANFOR ESTÃO SELECIONADOS 
   // SETA O BIT DE MOTOR SELECIONADO HABILITANDO LIGAR A MÁQUINA
   RUNG wire#powerrail
      Contact( "DB VALORES RECEBIDOS".VARIAVEIS_COMPARTILHADAS.DIGITAIS.MOTOR_SELECIONADO )
      Contact( "DB VALORES RECEBIDOS".VARIAVEIS_SANFOR.DIGITAIS.MODO_INDEP_SINC )
      S_Coil( "DB PRINCIPAL".COMANDOS.MOTOR_SELECIONADO )
   END_RUNG
   // the same network as SCL:
   IF "DB VALORES RECEBIDOS".VARIAVEIS_COMPARTILHADAS.DIGITAIS.MOTOR_SELECIONADO AND "DB VALORES RECEBIDOS".VARIAVEIS_SANFOR.DIGITAIS.MODO_INDEP_SINC THEN
       "DB PRINCIPAL".COMANDOS.MOTOR_SELECIONADO := TRUE;
   END_IF;
END_REGION

REGION Network 16: LIGA MÁQUINA
   // LÓGICA QUE SUPERVISIONA E CONTROLA COMANDO DE LIGA MÁQUINA
   RUNG wire#powerrail
      Contact( "DB PRINCIPAL".AUXILIARES.SEMPRE_1 )
      wire#w1
      Contact( "DB PRINCIPAL".COMANDOS.BOTAO_LIGA )
      P_Trig( "M10_0" )
      { S7_Templates := "SrcType := Real" } EQ_Contact(in1 := "DB PRINCIPAL".REFERENCIAS.FINAL_MAQUINA, in2 := 0.0)
      { S7_GenerateENO := "TRUE" } Move(in := "DB PRINCIPAL".REFERENCIAS.MINIMA, out1 => "DB PRINCIPAL".REFERENCIAS.BASE)
      S_Coil( "DB PRINCIPAL".COMANDOS.AUX_MARCHA )
   END_RUNG
   RUNG wire#w1
      Contact( "DB PRINCIPAL".COMANDOS.PARTIDA_MARCHA_SIN )
      wire#w2
      S_Coil( "DB PRINCIPAL".COMANDOS.MARCHA )
   END_RUNG
   RUNG wire#w2
      R_Coil( "DB PRINCIPAL".COMANDOS.AUX_MARCHA )
   END_RUNG
   // the same network as SCL:
   // ENO of a box is taken as its EN; it also drops when the box reports an error
   #_w1 := "DB PRINCIPAL".AUXILIARES.SEMPRE_1 AND "DB PRINCIPAL".COMANDOS.BOTAO_LIGA;
   #_w2 := #_w1 AND NOT "M10_0";   // rising edge
   "M10_0" := #_w1;
   IF #_w2 AND ("DB PRINCIPAL".REFERENCIAS.FINAL_MAQUINA = 0.0) THEN
       "DB PRINCIPAL".REFERENCIAS.BASE := "DB PRINCIPAL".REFERENCIAS.MINIMA;
       "DB PRINCIPAL".COMANDOS.AUX_MARCHA := TRUE;
   END_IF;
   IF "DB PRINCIPAL".AUXILIARES.SEMPRE_1 AND "DB PRINCIPAL".COMANDOS.PARTIDA_MARCHA_SIN THEN
       "DB PRINCIPAL".COMANDOS.MARCHA := TRUE;
       "DB PRINCIPAL".COMANDOS.AUX_MARCHA := FALSE;
   END_IF;
END_REGION

REGION Network 17
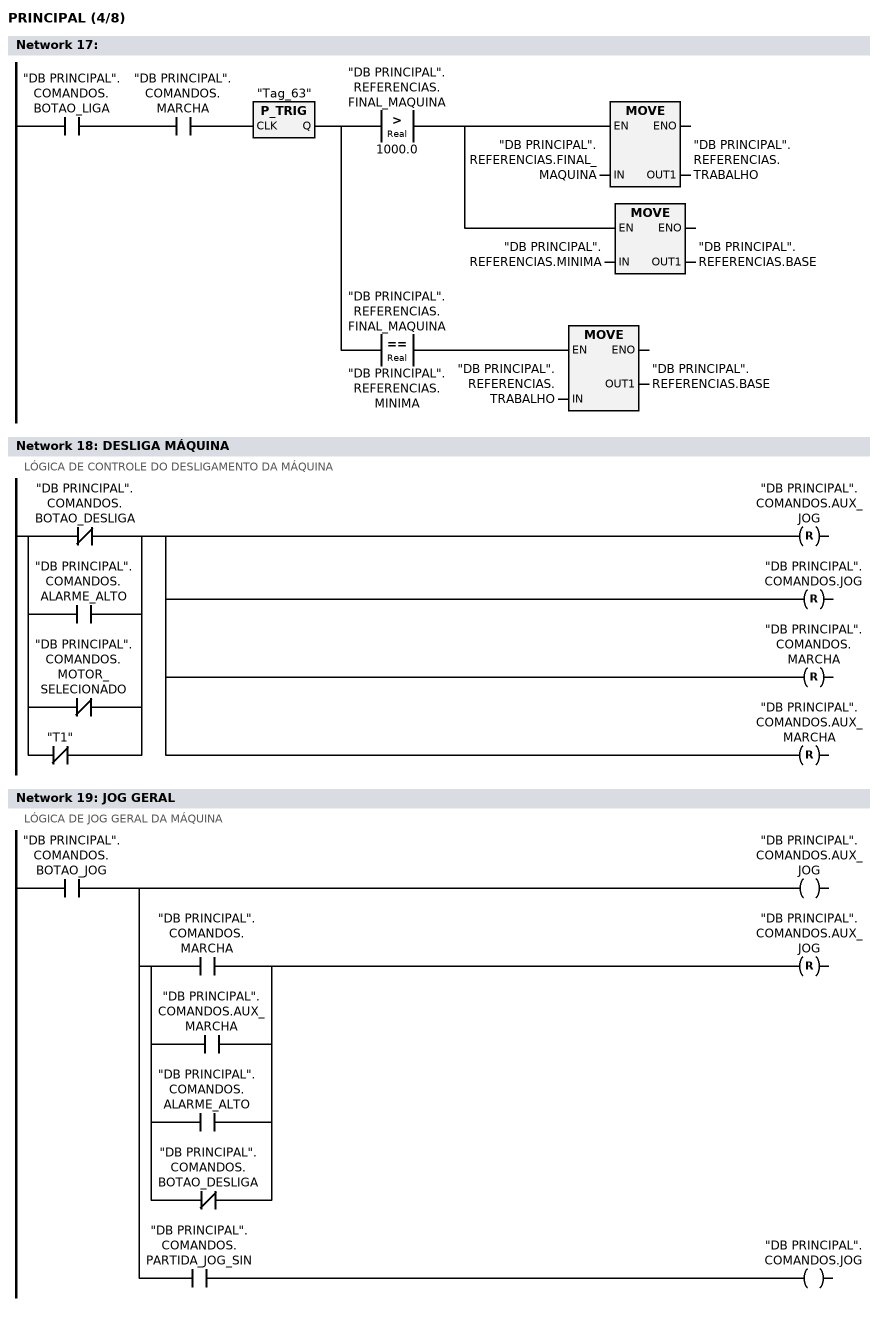
   RUNG wire#powerrail
      Contact( "DB PRINCIPAL".COMANDOS.BOTAO_LIGA )
      Contact( "DB PRINCIPAL".COMANDOS.MARCHA )
      P_Trig( "Tag_63" )
      wire#w1
      { S7_Templates := "SrcType := Real" } GT_Contact(in1 := "DB PRINCIPAL".REFERENCIAS.FINAL_MAQUINA, in2 := 1000.0)
      wire#w2
      { S7_GenerateENO := "TRUE" } Move(in := "DB PRINCIPAL".REFERENCIAS.FINAL_MAQUINA, out1 => "DB PRINCIPAL".REFERENCIAS.TRABALHO)
   END_RUNG
   RUNG wire#w2
      { S7_GenerateENO := "TRUE" } Move(in := "DB PRINCIPAL".REFERENCIAS.MINIMA, out1 => "DB PRINCIPAL".REFERENCIAS.BASE)
   END_RUNG
   RUNG wire#w1
      { S7_Templates := "SrcType := Real" } EQ_Contact(in1 := "DB PRINCIPAL".REFERENCIAS.FINAL_MAQUINA, in2 := "DB PRINCIPAL".REFERENCIAS.MINIMA)
      { S7_GenerateENO := "TRUE" } Move(in := "DB PRINCIPAL".REFERENCIAS.TRABALHO, out1 => "DB PRINCIPAL".REFERENCIAS.BASE)
   END_RUNG
   // the same network as SCL:
   #_w1 := "DB PRINCIPAL".COMANDOS.BOTAO_LIGA AND "DB PRINCIPAL".COMANDOS.MARCHA;
   #_w2 := #_w1 AND NOT "Tag_63";   // rising edge
   "Tag_63" := #_w1;
   IF #_w2 AND ("DB PRINCIPAL".REFERENCIAS.FINAL_MAQUINA > 1000.0) THEN
       "DB PRINCIPAL".REFERENCIAS.TRABALHO := "DB PRINCIPAL".REFERENCIAS.FINAL_MAQUINA;
       "DB PRINCIPAL".REFERENCIAS.BASE := "DB PRINCIPAL".REFERENCIAS.MINIMA;
   END_IF;
   IF #_w2 AND ("DB PRINCIPAL".REFERENCIAS.FINAL_MAQUINA = "DB PRINCIPAL".REFERENCIAS.MINIMA) THEN
       "DB PRINCIPAL".REFERENCIAS.BASE := "DB PRINCIPAL".REFERENCIAS.TRABALHO;
   END_IF;
END_REGION

REGION Network 18: DESLIGA MÁQUINA
   // LÓGICA DE CONTROLE DO DESLIGAMENTO DA MÁQUINA
   RUNG wire#powerrail
      I_Contact( "DB PRINCIPAL".COMANDOS.BOTAO_DESLIGA )
      wire#w1
      R_Coil( "DB PRINCIPAL".COMANDOS.AUX_JOG )
   END_RUNG
   RUNG wire#powerrail
      Contact( "DB PRINCIPAL".COMANDOS.ALARME_ALTO )
   END_RUNG wire#w1
   RUNG wire#powerrail
      I_Contact( "DB PRINCIPAL".COMANDOS.MOTOR_SELECIONADO )
   END_RUNG wire#w1
   RUNG wire#powerrail
      I_Contact( "T1" )
   END_RUNG wire#w1
   RUNG wire#w1
      R_Coil( "DB PRINCIPAL".COMANDOS.JOG )
   END_RUNG
   RUNG wire#w1
      R_Coil( "DB PRINCIPAL".COMANDOS.MARCHA )
   END_RUNG
   RUNG wire#w1
      R_Coil( "DB PRINCIPAL".COMANDOS.AUX_MARCHA )
   END_RUNG
   // the same network as SCL:
   IF NOT "DB PRINCIPAL".COMANDOS.BOTAO_DESLIGA OR "DB PRINCIPAL".COMANDOS.ALARME_ALTO OR NOT "DB PRINCIPAL".COMANDOS.MOTOR_SELECIONADO OR NOT "T1" THEN
       "DB PRINCIPAL".COMANDOS.AUX_JOG := FALSE;
       "DB PRINCIPAL".COMANDOS.JOG := FALSE;
       "DB PRINCIPAL".COMANDOS.MARCHA := FALSE;
       "DB PRINCIPAL".COMANDOS.AUX_MARCHA := FALSE;
   END_IF;
END_REGION

REGION Network 19: JOG GERAL
   // LÓGICA DE JOG GERAL DA MÁQUINA
   RUNG wire#powerrail
      Contact( "DB PRINCIPAL".COMANDOS.BOTAO_JOG )
      wire#w1
      Coil( "DB PRINCIPAL".COMANDOS.AUX_JOG )
   END_RUNG
   RUNG wire#w1
      Contact( "DB PRINCIPAL".COMANDOS.MARCHA )
      wire#w2
      R_Coil( "DB PRINCIPAL".COMANDOS.AUX_JOG )
   END_RUNG
   RUNG wire#w1
      Contact( "DB PRINCIPAL".COMANDOS.AUX_MARCHA )
   END_RUNG wire#w2
   RUNG wire#w1
      Contact( "DB PRINCIPAL".COMANDOS.ALARME_ALTO )
   END_RUNG wire#w2
   RUNG wire#w1
      I_Contact( "DB PRINCIPAL".COMANDOS.BOTAO_DESLIGA )
   END_RUNG wire#w2
   RUNG wire#w1
      Contact( "DB PRINCIPAL".COMANDOS.PARTIDA_JOG_SIN )
      Coil( "DB PRINCIPAL".COMANDOS.JOG )
   END_RUNG
   // the same network as SCL:
   "DB PRINCIPAL".COMANDOS.AUX_JOG := "DB PRINCIPAL".COMANDOS.BOTAO_JOG;
   IF "DB PRINCIPAL".COMANDOS.BOTAO_JOG AND ("DB PRINCIPAL".COMANDOS.MARCHA OR "DB PRINCIPAL".COMANDOS.AUX_MARCHA OR "DB PRINCIPAL".COMANDOS.ALARME_ALTO OR NOT "DB PRINCIPAL".COMANDOS.BOTAO_DESLIGA) THEN
       "DB PRINCIPAL".COMANDOS.AUX_JOG := FALSE;
   END_IF;
   "DB PRINCIPAL".COMANDOS.JOG := "DB PRINCIPAL".COMANDOS.BOTAO_JOG AND "DB PRINCIPAL".COMANDOS.PARTIDA_JOG_SIN;
END_REGION

REGION Network 20: SINALIZAÇÃO
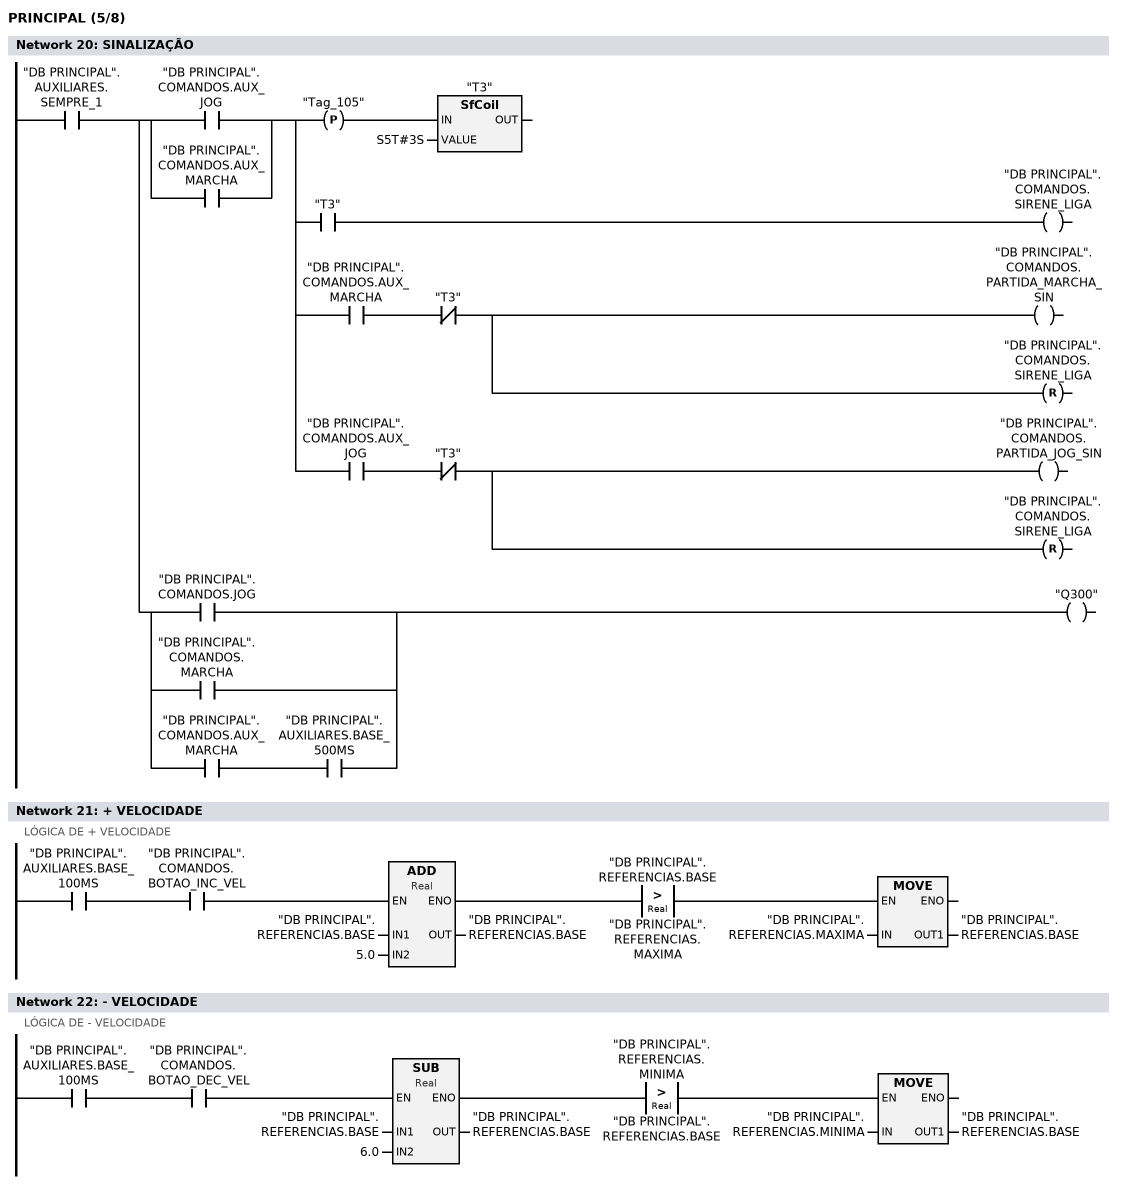
   // no SCL statement known for SfCoil: written as a call
   #_w1 := "DB PRINCIPAL".AUXILIARES.SEMPRE_1 AND ("DB PRINCIPAL".COMANDOS.AUX_JOG OR "DB PRINCIPAL".COMANDOS.AUX_MARCHA);
   #_w2 := #_w1 AND NOT "Tag_105";   // rising edge
   "Tag_105" := #_w1;
   #_w3 := "DB PRINCIPAL".AUXILIARES.SEMPRE_1;
   SfCoil(value := S5T#3S, in := #_w2, operand := "T3");
   "DB PRINCIPAL".COMANDOS.SIRENE_LIGA := #_w1 AND "T3";
   "DB PRINCIPAL".COMANDOS.PARTIDA_MARCHA_SIN := #_w1 AND "DB PRINCIPAL".COMANDOS.AUX_MARCHA AND NOT "T3";
   IF "DB PRINCIPAL".COMANDOS.PARTIDA_MARCHA_SIN THEN "DB PRINCIPAL".COMANDOS.SIRENE_LIGA := FALSE; END_IF;
   "DB PRINCIPAL".COMANDOS.PARTIDA_JOG_SIN := #_w1 AND "DB PRINCIPAL".COMANDOS.AUX_JOG AND NOT "T3";
   IF "DB PRINCIPAL".COMANDOS.PARTIDA_JOG_SIN THEN "DB PRINCIPAL".COMANDOS.SIRENE_LIGA := FALSE; END_IF;
   "Q300" := #_w3 AND ("DB PRINCIPAL".COMANDOS.JOG OR "DB PRINCIPAL".COMANDOS.MARCHA OR ("DB PRINCIPAL".COMANDOS.AUX_MARCHA AND "DB PRINCIPAL".AUXILIARES.BASE_500MS));
END_REGION

REGION Network 21: + VELOCIDADE
   // LÓGICA DE + VELOCIDADE
   RUNG wire#powerrail
      Contact( "DB PRINCIPAL".AUXILIARES.BASE_100MS )
      Contact( "DB PRINCIPAL".COMANDOS.BOTAO_INC_VEL )
      { S7_Templates := "SrcType := Real"; S7_GenerateENO := "TRUE" } Add(in1 := "DB PRINCIPAL".REFERENCIAS.BASE, in2 := 5.0, out => "DB PRINCIPAL".REFERENCIAS.BASE)
      { S7_Templates := "SrcType := Real" } GT_Contact(in1 := "DB PRINCIPAL".REFERENCIAS.BASE, in2 := "DB PRINCIPAL".REFERENCIAS.MAXIMA)
      { S7_GenerateENO := "TRUE" } Move(in := "DB PRINCIPAL".REFERENCIAS.MAXIMA, out1 => "DB PRINCIPAL".REFERENCIAS.BASE)
   END_RUNG
   // the same network as SCL:
   // ENO of a box is taken as its EN; it also drops when the box reports an error
   #_w1 := "DB PRINCIPAL".AUXILIARES.BASE_100MS AND "DB PRINCIPAL".COMANDOS.BOTAO_INC_VEL;
   IF #_w1 THEN "DB PRINCIPAL".REFERENCIAS.BASE := "DB PRINCIPAL".REFERENCIAS.BASE + 5.0; END_IF;
   IF #_w1 AND ("DB PRINCIPAL".REFERENCIAS.BASE > "DB PRINCIPAL".REFERENCIAS.MAXIMA) THEN
       "DB PRINCIPAL".REFERENCIAS.BASE := "DB PRINCIPAL".REFERENCIAS.MAXIMA;
   END_IF;
END_REGION

REGION Network 22: - VELOCIDADE
   // LÓGICA DE - VELOCIDADE
   RUNG wire#powerrail
      Contact( "DB PRINCIPAL".AUXILIARES.BASE_100MS )
      Contact( "DB PRINCIPAL".COMANDOS.BOTAO_DEC_VEL )
      { S7_Templates := "SrcType := Real"; S7_GenerateENO := "TRUE" } Sub(in1 := "DB PRINCIPAL".REFERENCIAS.BASE, in2 := 6.0, out => "DB PRINCIPAL".REFERENCIAS.BASE)
      { S7_Templates := "SrcType := Real" } GT_Contact(in1 := "DB PRINCIPAL".REFERENCIAS.MINIMA, in2 := "DB PRINCIPAL".REFERENCIAS.BASE)
      { S7_GenerateENO := "TRUE" } Move(in := "DB PRINCIPAL".REFERENCIAS.MINIMA, out1 => "DB PRINCIPAL".REFERENCIAS.BASE)
   END_RUNG
   // the same network as SCL:
   // ENO of a box is taken as its EN; it also drops when the box reports an error
   #_w1 := "DB PRINCIPAL".AUXILIARES.BASE_100MS AND "DB PRINCIPAL".COMANDOS.BOTAO_DEC_VEL;
   IF #_w1 THEN "DB PRINCIPAL".REFERENCIAS.BASE := "DB PRINCIPAL".REFERENCIAS.BASE - 6.0; END_IF;
   IF #_w1 AND ("DB PRINCIPAL".REFERENCIAS.MINIMA > "DB PRINCIPAL".REFERENCIAS.BASE) THEN
       "DB PRINCIPAL".REFERENCIAS.BASE := "DB PRINCIPAL".REFERENCIAS.MINIMA;
   END_IF;
END_REGION

REGION Network 23 (STL): ACC/DEC DA REFERENCIA DE VELOCIDADE
   // ACC/DEC DA REFERENCIA DE VELOCIDADE
   // LIMITAÇÃO DOS VALORES MAXIMOS E MINIMOS ATINGIDOS
         A     "DB PRINCIPAL".COMANDOS.MARCHA;
         =     %L24.0;
         A     %L24.0;
         A(;
         L     "DB PRINCIPAL".REFERENCIAS.BASE;
         L     "DB PRINCIPAL".REFERENCIAS.FINAL_MAQUINA;
         >R;
         );
         A     "DB PRINCIPAL".AUXILIARES.BASE_100MS;
         JNB   _00a;
         L     "DB PRINCIPAL".REFERENCIAS.FINAL_MAQUINA;
         L     "DB PRINCIPAL".REFERENCIAS.PASSO_ACC;
         +R;
         T     "DB PRINCIPAL".REFERENCIAS.FINAL_MAQUINA;
   _00a: NOP   0;
         A     %L24.0;
         A(;
         L     "DB PRINCIPAL".REFERENCIAS.FINAL_MAQUINA;
         L     "DB PRINCIPAL".REFERENCIAS.BASE;
         >R;
         );
         A     "DB PRINCIPAL".AUXILIARES.BASE_100MS;
         JNB   _00b;
         L     "DB PRINCIPAL".REFERENCIAS.FINAL_MAQUINA;
         L     "DB PRINCIPAL".REFERENCIAS.PASSO_DEC;
         -R;
         T     "DB PRINCIPAL".REFERENCIAS.FINAL_MAQUINA;
   _00b: NOP   0;
         A(;
         A     %L24.0;
         JNB   _00c;
         L     "DB PRINCIPAL".REFERENCIAS.FINAL_MAQUINA;
         L     "DB PRINCIPAL".REFERENCIAS.BASE;
         -R;
         T     "Tag_58";
         AN    OV;
         SAVE;
         CLR;
   _00c: A     BR;
         );
         A(;
         L     "Tag_58";
         L     -1.0;
         >R;
         );
         A(;
         L     "Tag_58";
         L     1.0;
         <R;
         );
         JNB   _00d;
         L     "DB PRINCIPAL".REFERENCIAS.BASE;
         T     "DB PRINCIPAL".REFERENCIAS.FINAL_MAQUINA;
   _00d: NOP   0;
         A     %L24.0;
         A(;
         L     "DB PRINCIPAL".REFERENCIAS.FINAL_MAQUINA;
         L     0.0;
         <R;
         );
         JNB   _00e;
         L     0.0;
         T     "DB PRINCIPAL".REFERENCIAS.FINAL_MAQUINA;
   _00e: NOP   0;
         A     %L24.0;
         A(;
         L     "DB PRINCIPAL".REFERENCIAS.FINAL_MAQUINA;
         L     "DB PRINCIPAL".REFERENCIAS.MAXIMA;
         >R;
         );
         JNB   _00f;
         L     "DB PRINCIPAL".REFERENCIAS.MAXIMA;
         T     "DB PRINCIPAL".REFERENCIAS.FINAL_MAQUINA;
   _00f: NOP   0;
END_REGION

REGION Network 24: TRAVA BALANCIM
   // LÓGICA DE CONTROLE E SINALIZAÇÃO DE TRAVA BALANCIM
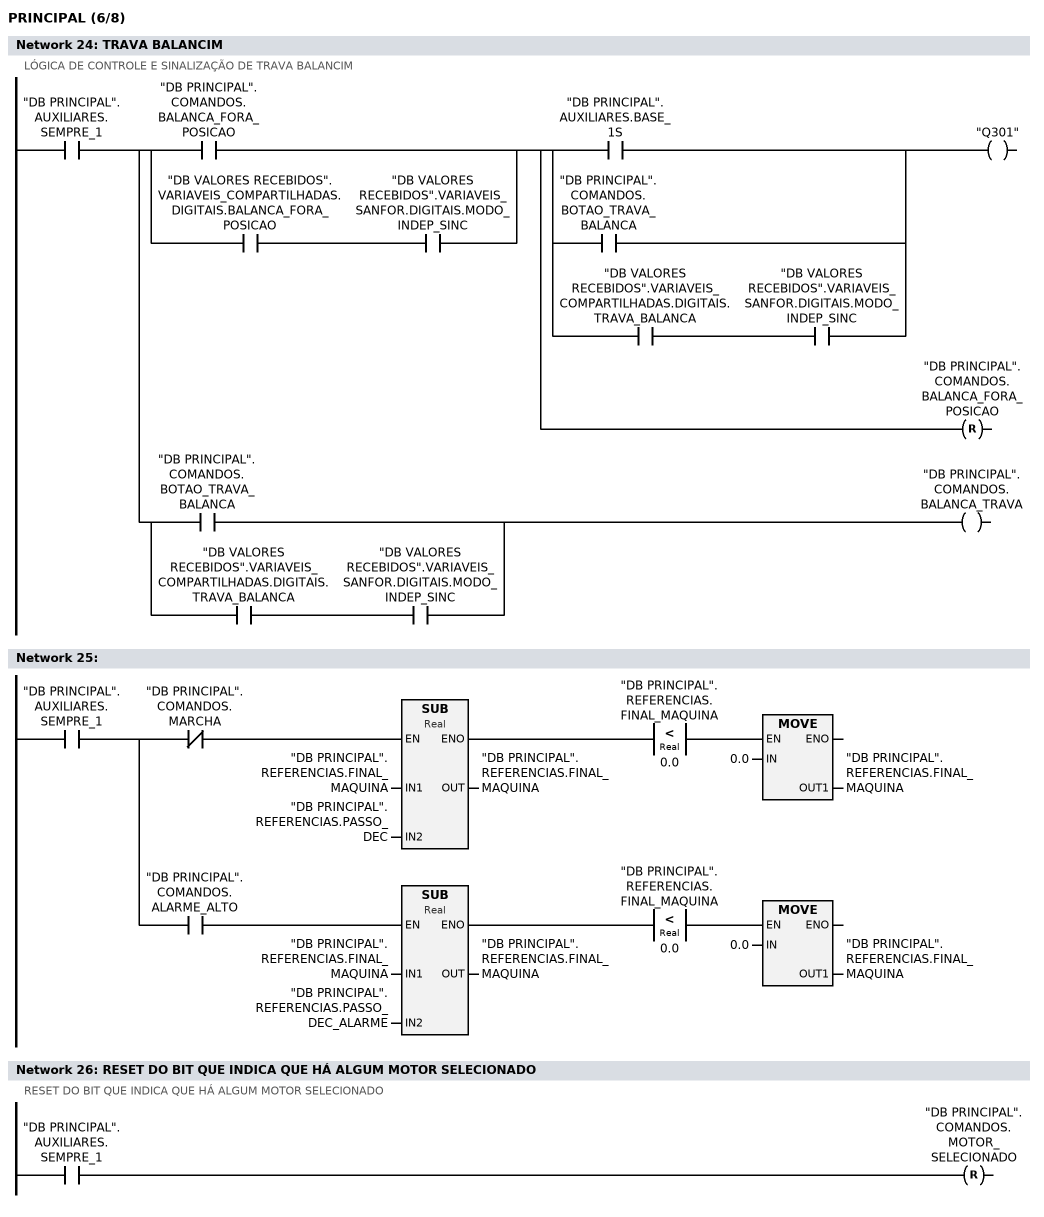
   RUNG wire#powerrail
      Contact( "DB PRINCIPAL".AUXILIARES.SEMPRE_1 )
      wire#w1
      Contact( "DB PRINCIPAL".COMANDOS.BALANCA_FORA_POSICAO )
      wire#w2
      Contact( "DB PRINCIPAL".AUXILIARES.BASE_1S )
      wire#w3
      Coil( "Q301" )
   END_RUNG
   RUNG wire#w1
      Contact( "DB VALORES RECEBIDOS".VARIAVEIS_COMPARTILHADAS.DIGITAIS.BALANCA_FORA_POSICAO )
      Contact( "DB VALORES RECEBIDOS".VARIAVEIS_SANFOR.DIGITAIS.MODO_INDEP_SINC )
   END_RUNG wire#w2
   RUNG wire#w2
      Contact( "DB PRINCIPAL".COMANDOS.BOTAO_TRAVA_BALANCA )
   END_RUNG wire#w3
   RUNG wire#w2
      Contact( "DB VALORES RECEBIDOS".VARIAVEIS_COMPARTILHADAS.DIGITAIS.TRAVA_BALANCA )
      Contact( "DB VALORES RECEBIDOS".VARIAVEIS_SANFOR.DIGITAIS.MODO_INDEP_SINC )
   END_RUNG wire#w3
   RUNG wire#w2
      R_Coil( "DB PRINCIPAL".COMANDOS.BALANCA_FORA_POSICAO )
   END_RUNG
   RUNG wire#w1
      Contact( "DB PRINCIPAL".COMANDOS.BOTAO_TRAVA_BALANCA )
      wire#w4
      Coil( "DB PRINCIPAL".COMANDOS.BALANCA_TRAVA )
   END_RUNG
   RUNG wire#w1
      Contact( "DB VALORES RECEBIDOS".VARIAVEIS_COMPARTILHADAS.DIGITAIS.TRAVA_BALANCA )
      Contact( "DB VALORES RECEBIDOS".VARIAVEIS_SANFOR.DIGITAIS.MODO_INDEP_SINC )
   END_RUNG wire#w4
   // the same network as SCL:
   #_w1 := "DB PRINCIPAL".AUXILIARES.SEMPRE_1 AND ("DB PRINCIPAL".COMANDOS.BALANCA_FORA_POSICAO OR ("DB VALORES RECEBIDOS".VARIAVEIS_COMPARTILHADAS.DIGITAIS.BALANCA_FORA_POSICAO AND "DB VALORES RECEBIDOS".VARIAVEIS_SANFOR.DIGITAIS.MODO_INDEP_SINC));
   "Q301" := #_w1 AND ("DB PRINCIPAL".AUXILIARES.BASE_1S OR "DB PRINCIPAL".COMANDOS.BOTAO_TRAVA_BALANCA OR ("DB VALORES RECEBIDOS".VARIAVEIS_COMPARTILHADAS.DIGITAIS.TRAVA_BALANCA AND "DB VALORES RECEBIDOS".VARIAVEIS_SANFOR.DIGITAIS.MODO_INDEP_SINC));
   IF #_w1 THEN "DB PRINCIPAL".COMANDOS.BALANCA_FORA_POSICAO := FALSE; END_IF;
   "DB PRINCIPAL".COMANDOS.BALANCA_TRAVA := "DB PRINCIPAL".AUXILIARES.SEMPRE_1 AND ("DB PRINCIPAL".COMANDOS.BOTAO_TRAVA_BALANCA OR ("DB VALORES RECEBIDOS".VARIAVEIS_COMPARTILHADAS.DIGITAIS.TRAVA_BALANCA AND "DB VALORES RECEBIDOS".VARIAVEIS_SANFOR.DIGITAIS.MODO_INDEP_SINC));
END_REGION

REGION Network 25
   RUNG wire#powerrail
      Contact( "DB PRINCIPAL".AUXILIARES.SEMPRE_1 )
      wire#w1
      I_Contact( "DB PRINCIPAL".COMANDOS.MARCHA )
      { S7_Templates := "SrcType := Real"; S7_GenerateENO := "TRUE" } Sub(in1 := "DB PRINCIPAL".REFERENCIAS.FINAL_MAQUINA, in2 := "DB PRINCIPAL".REFERENCIAS.PASSO_DEC, out => "DB PRINCIPAL".REFERENCIAS.FINAL_MAQUINA)
      { S7_Templates := "SrcType := Real" } LT_Contact(in1 := "DB PRINCIPAL".REFERENCIAS.FINAL_MAQUINA, in2 := 0.0)
      { S7_GenerateENO := "TRUE" } Move(in := 0.0, out1 => "DB PRINCIPAL".REFERENCIAS.FINAL_MAQUINA)
   END_RUNG
   RUNG wire#w1
      Contact( "DB PRINCIPAL".COMANDOS.ALARME_ALTO )
      { S7_Templates := "SrcType := Real"; S7_GenerateENO := "TRUE" } Sub(in1 := "DB PRINCIPAL".REFERENCIAS.FINAL_MAQUINA, in2 := "DB PRINCIPAL".REFERENCIAS.PASSO_DEC_ALARME, out => "DB PRINCIPAL".REFERENCIAS.FINAL_MAQUINA)
      { S7_Templates := "SrcType := Real" } LT_Contact(in1 := "DB PRINCIPAL".REFERENCIAS.FINAL_MAQUINA, in2 := 0.0)
      { S7_GenerateENO := "TRUE" } Move(in := 0.0, out1 => "DB PRINCIPAL".REFERENCIAS.FINAL_MAQUINA)
   END_RUNG
   // the same network as SCL:
   // ENO of a box is taken as its EN; it also drops when the box reports an error
   #_w1 := "DB PRINCIPAL".AUXILIARES.SEMPRE_1 AND NOT "DB PRINCIPAL".COMANDOS.MARCHA;
   IF #_w1 THEN
       "DB PRINCIPAL".REFERENCIAS.FINAL_MAQUINA := "DB PRINCIPAL".REFERENCIAS.FINAL_MAQUINA - "DB PRINCIPAL".REFERENCIAS.PASSO_DEC;
   END_IF;
   IF #_w1 AND ("DB PRINCIPAL".REFERENCIAS.FINAL_MAQUINA < 0.0) THEN
       "DB PRINCIPAL".REFERENCIAS.FINAL_MAQUINA := 0.0;
   END_IF;
   #_w2 := "DB PRINCIPAL".AUXILIARES.SEMPRE_1 AND "DB PRINCIPAL".COMANDOS.ALARME_ALTO;
   IF #_w2 THEN
       "DB PRINCIPAL".REFERENCIAS.FINAL_MAQUINA := "DB PRINCIPAL".REFERENCIAS.FINAL_MAQUINA - "DB PRINCIPAL".REFERENCIAS.PASSO_DEC_ALARME;
   END_IF;
   IF #_w2 AND ("DB PRINCIPAL".REFERENCIAS.FINAL_MAQUINA < 0.0) THEN
       "DB PRINCIPAL".REFERENCIAS.FINAL_MAQUINA := 0.0;
   END_IF;
END_REGION

REGION Network 26: RESET DO BIT QUE INDICA QUE HÁ ALGUM MOTOR SELECIONADO
   // RESET DO BIT QUE INDICA QUE HÁ ALGUM MOTOR SELECIONADO
   RUNG wire#powerrail
      Contact( "DB PRINCIPAL".AUXILIARES.SEMPRE_1 )
      R_Coil( "DB PRINCIPAL".COMANDOS.MOTOR_SELECIONADO )
   END_RUNG
   // the same network as SCL:
   IF "DB PRINCIPAL".AUXILIARES.SEMPRE_1 THEN "DB PRINCIPAL".COMANDOS.MOTOR_SELECIONADO := FALSE; END_IF;
END_REGION

REGION Network 27: RESET DOS ALARMES
   // RESET DOS ALARMES
   // SINALIZAÇÃO DO BOTÃO
   // QUANDO PRECIONADO O BOTÃO DE RESET
   // QUANDO DA ENERGIZAÇÃO DO P.L.C.
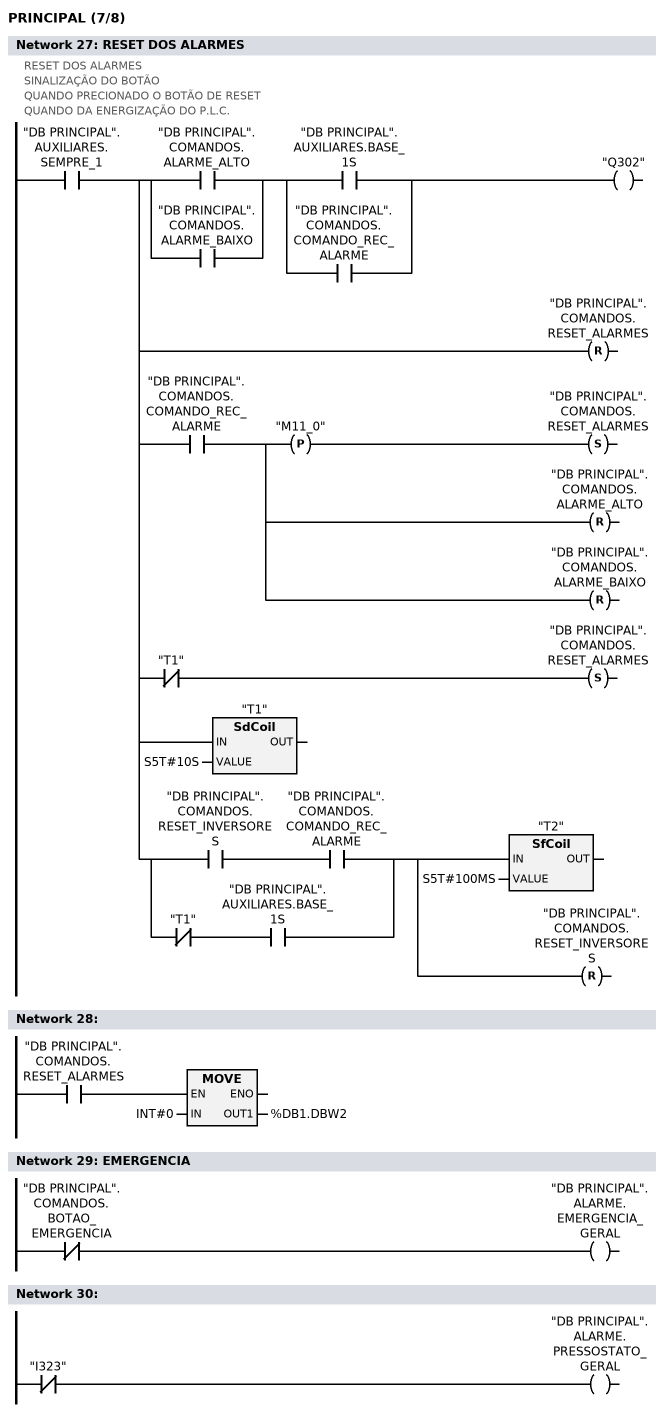
   // no SCL statement known for SdCoil, SfCoil: written as a call
   "Q302" := "DB PRINCIPAL".AUXILIARES.SEMPRE_1 AND ("DB PRINCIPAL".COMANDOS.ALARME_ALTO OR "DB PRINCIPAL".COMANDOS.ALARME_BAIXO) AND ("DB PRINCIPAL".AUXILIARES.BASE_1S OR "DB PRINCIPAL".COMANDOS.COMANDO_REC_ALARME);
   IF "DB PRINCIPAL".AUXILIARES.SEMPRE_1 THEN "DB PRINCIPAL".COMANDOS.RESET_ALARMES := FALSE; END_IF;
   #_w1 := "DB PRINCIPAL".AUXILIARES.SEMPRE_1 AND "DB PRINCIPAL".COMANDOS.COMANDO_REC_ALARME;
   #_w2 := #_w1 AND NOT "M11_0";   // rising edge
   "M11_0" := #_w1;
   IF #_w2 THEN "DB PRINCIPAL".COMANDOS.RESET_ALARMES := TRUE; END_IF;
   IF #_w1 THEN
       "DB PRINCIPAL".COMANDOS.ALARME_ALTO := FALSE;
       "DB PRINCIPAL".COMANDOS.ALARME_BAIXO := FALSE;
   END_IF;
   IF "DB PRINCIPAL".AUXILIARES.SEMPRE_1 AND NOT "T1" THEN
       "DB PRINCIPAL".COMANDOS.RESET_ALARMES := TRUE;
   END_IF;
   #_w3 := "DB PRINCIPAL".AUXILIARES.SEMPRE_1;
   SdCoil(value := S5T#10S, operand := "T1", in := "DB PRINCIPAL".AUXILIARES.SEMPRE_1);
   #_w4 := #_w3 AND (("DB PRINCIPAL".COMANDOS.RESET_INVERSORES AND "DB PRINCIPAL".COMANDOS.COMANDO_REC_ALARME) OR (NOT "T1" AND "DB PRINCIPAL".AUXILIARES.BASE_1S));
   SfCoil(in := #_w4, value := S5T#100MS, operand := "T2");
   IF #_w4 THEN "DB PRINCIPAL".COMANDOS.RESET_INVERSORES := FALSE; END_IF;
END_REGION

REGION Network 28
   RUNG wire#powerrail
      Contact( "DB PRINCIPAL".COMANDOS.RESET_ALARMES )
      { S7_GenerateENO := "TRUE" } Move(in := INT#0, out1 => %DB1.DBW2)
   END_RUNG
   // the same network as SCL:
   IF "DB PRINCIPAL".COMANDOS.RESET_ALARMES THEN %DB1.DBW2 := INT#0; END_IF;
END_REGION

REGION Network 29: EMERGENCIA
   RUNG wire#powerrail
      I_Contact( "DB PRINCIPAL".COMANDOS.BOTAO_EMERGENCIA )
      Coil( "DB PRINCIPAL".ALARME.EMERGENCIA_GERAL )
   END_RUNG
   // the same network as SCL:
   "DB PRINCIPAL".ALARME.EMERGENCIA_GERAL := NOT "DB PRINCIPAL".COMANDOS.BOTAO_EMERGENCIA;
END_REGION

REGION Network 30
   RUNG wire#powerrail
      I_Contact( "I323" )
      Coil( "DB PRINCIPAL".ALARME.PRESSOSTATO_GERAL )
   END_RUNG
   // the same network as SCL:
   "DB PRINCIPAL".ALARME.PRESSOSTATO_GERAL := NOT "I323";
END_REGION

REGION Network 31: BIT QUE INDICA QUE ALGUM ALARME DE NIVEL ALTO FOI GERADO
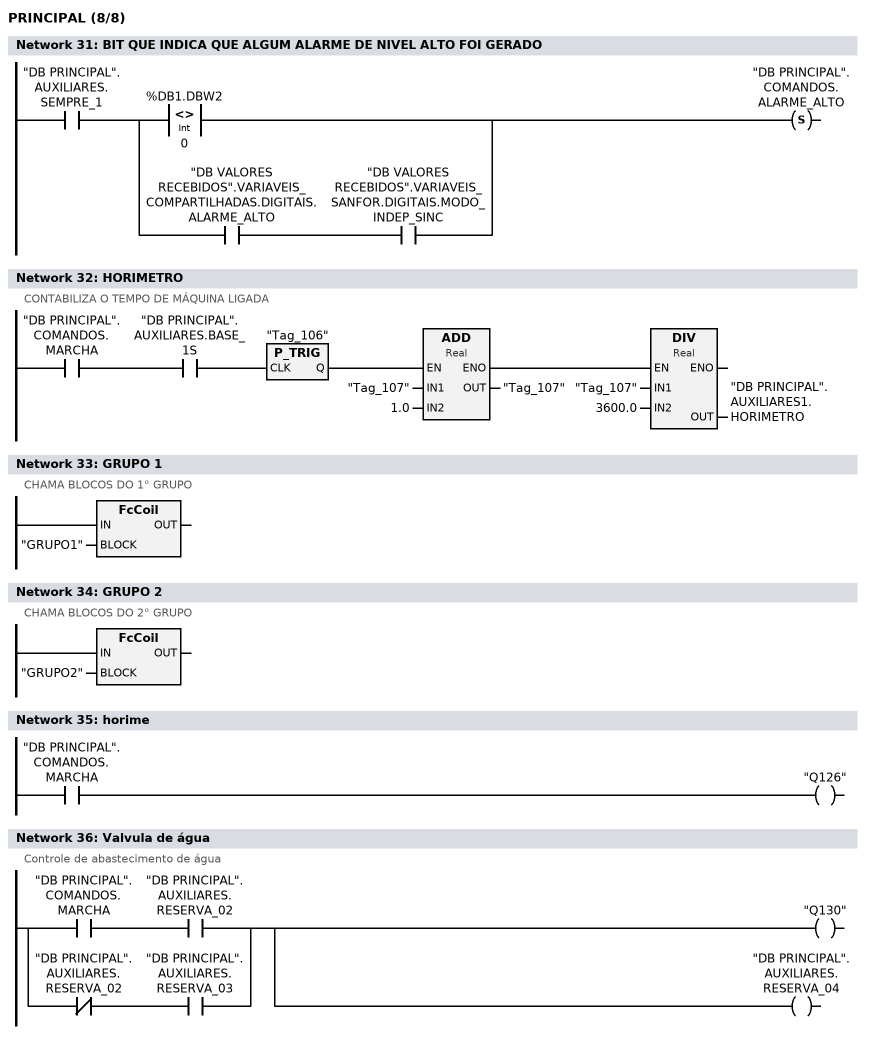
   RUNG wire#powerrail
      Contact( "DB PRINCIPAL".AUXILIARES.SEMPRE_1 )
      wire#w1
      { S7_Templates := "SrcType := Int" } NE_Contact(in1 := %DB1.DBW2, in2 := 0)
      wire#w2
      S_Coil( "DB PRINCIPAL".COMANDOS.ALARME_ALTO )
   END_RUNG
   RUNG wire#w1
      Contact( "DB VALORES RECEBIDOS".VARIAVEIS_COMPARTILHADAS.DIGITAIS.ALARME_ALTO )
      Contact( "DB VALORES RECEBIDOS".VARIAVEIS_SANFOR.DIGITAIS.MODO_INDEP_SINC )
   END_RUNG wire#w2
   // the same network as SCL:
   IF "DB PRINCIPAL".AUXILIARES.SEMPRE_1 AND ((%DB1.DBW2 <> 0) OR ("DB VALORES RECEBIDOS".VARIAVEIS_COMPARTILHADAS.DIGITAIS.ALARME_ALTO AND "DB VALORES RECEBIDOS".VARIAVEIS_SANFOR.DIGITAIS.MODO_INDEP_SINC)) THEN
       "DB PRINCIPAL".COMANDOS.ALARME_ALTO := TRUE;
   END_IF;
END_REGION

REGION Network 32: HORIMETRO
   // CONTABILIZA O TEMPO DE MÁQUINA LIGADA
   RUNG wire#powerrail
      Contact( "DB PRINCIPAL".COMANDOS.MARCHA )
      Contact( "DB PRINCIPAL".AUXILIARES.BASE_1S )
      P_Trig( "Tag_106" )
      { S7_Templates := "SrcType := Real"; S7_GenerateENO := "TRUE" } Add(in1 := "Tag_107", in2 := 1.0, out => "Tag_107")
      { S7_Templates := "SrcType := Real"; S7_GenerateENO := "TRUE" } Div(in1 := "Tag_107", in2 := 3600.0, out => "DB PRINCIPAL".AUXILIARES1.HORIMETRO)
   END_RUNG
   // the same network as SCL:
   // ENO of a box is taken as its EN; it also drops when the box reports an error
   #_w1 := "DB PRINCIPAL".COMANDOS.MARCHA AND "DB PRINCIPAL".AUXILIARES.BASE_1S;
   #_w2 := #_w1 AND NOT "Tag_106";   // rising edge
   "Tag_106" := #_w1;
   IF #_w2 THEN
       "Tag_107" := "Tag_107" + 1.0;
       "DB PRINCIPAL".AUXILIARES1.HORIMETRO := "Tag_107" / 3600.0;
   END_IF;
END_REGION

REGION Network 33: GRUPO 1
   // CHAMA BLOCOS DO 1° GRUPO
   // no SCL statement known for FcCoil: written as a call
   FcCoil(block := "GRUPO1", in := TRUE);
END_REGION

REGION Network 34: GRUPO 2
   // CHAMA BLOCOS DO 2° GRUPO
   // no SCL statement known for FcCoil: written as a call
   FcCoil(block := "GRUPO2", in := TRUE);
END_REGION

REGION Network 35: horime
   RUNG wire#powerrail
      Contact( "DB PRINCIPAL".COMANDOS.MARCHA )
      Coil( "Q126" )
   END_RUNG
   // the same network as SCL:
   "Q126" := "DB PRINCIPAL".COMANDOS.MARCHA;
END_REGION

REGION Network 36: Valvula de água
   // Controle de abastecimento de água
   RUNG wire#powerrail
      Contact( "DB PRINCIPAL".COMANDOS.MARCHA )
      Contact( "DB PRINCIPAL".AUXILIARES.RESERVA_02 )
      wire#w1
      Coil( "Q130" )
   END_RUNG
   RUNG wire#powerrail
      I_Contact( "DB PRINCIPAL".AUXILIARES.RESERVA_02 )
      Contact( "DB PRINCIPAL".AUXILIARES.RESERVA_03 )
   END_RUNG wire#w1
   RUNG wire#w1
      Coil( "DB PRINCIPAL".AUXILIARES.RESERVA_04 )
   END_RUNG
   // the same network as SCL:
   "Q130" := ("DB PRINCIPAL".COMANDOS.MARCHA AND "DB PRINCIPAL".AUXILIARES.RESERVA_02) OR (NOT "DB PRINCIPAL".AUXILIARES.RESERVA_02 AND "DB PRINCIPAL".AUXILIARES.RESERVA_03);
   "DB PRINCIPAL".AUXILIARES.RESERVA_04 := "Q130";
END_REGION
END_ORGANIZATION_BLOCK

ORGANIZATION_BLOCK "OB 100ms"   // OB35, LAD
TITLE = MÓDULO DE INTERRUPÇÃO PERIODICO
{ S7_Optimized_Access := 'FALSE' }
AUTHOR : THALLES
FAMILY : MÁQUINA
NAME : RAMOSA
VERSION : 0.1
// Automation Pack Automação Indl. e Com. Ltda.
// Cliente: Texima S/A Ind. de Máquinas
// Cliente Final: Companhia Indústrial Cataguases
// Máquina: Linha de Alvejamento - O.S.: 24.543
   VAR_TEMP
      OB35_EV_CLASS : Byte;   // Bits 0-3 = 1 (Coming event), Bits 4-7 = 1 (Event class 1)
      OB35_STRT_INF : Byte;   // 16#36 (OB 35 has started)
      OB35_PRIORITY : Byte;   // Priority of OB Execution
      OB35_OB_NUMBR : Byte;   // 35 (Organization block 35, OB35)
      OB35_RESERVED_1 : Byte;   // Reserved for system
      OB35_RESERVED_2 : Byte;   // Reserved for system
      OB35_PHASE_OFFSET : Word;   // Phase offset (msec)
      OB35_RESERVED_3 : Int;   // Reserved for system
      OB35_EXC_FREQ : Int;   // Frequency of execution (msec)
      OB35_DATE_TIME : Date_And_Time;   // Date and time OB35 started
   END_VAR
BEGIN

REGION Network 1: CHAMA MÓDULO DE CONTROLE DO SISTEMA DE AQUECIMENTO
   // CHAMA MÓDULO DE CONTROLE DO SISTEMA DE AQUECIMENTO
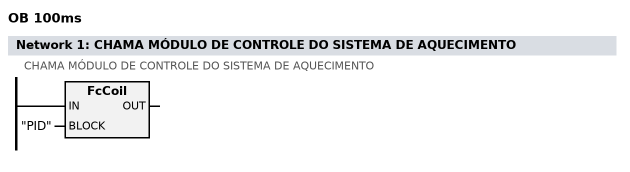
   // no SCL statement known for FcCoil: written as a call
   FcCoil(block := "PID", in := TRUE);
END_REGION
END_ORGANIZATION_BLOCK

ORGANIZATION_BLOCK "OBNL_FLT"   // OB85, LAD
TITLE = "Organization Block (OB) Not Loaded Fault"
{ S7_Optimized_Access := 'FALSE' }
VERSION : 0.1
   VAR_TEMP
      OB85_EV_CLASS : Byte;   // 16#35 Event class 3
      OB85_FLT_ID : Byte;   // 16#XX, Fault identification code
      OB85_PRIORITY : Byte;   // Priority of OB Execution
      OB85_OB_NUMBR : Byte;   // 85 (Organization block 85, OB85)
      OB85_RESERVED_1 : Byte;   // Reserved for system
      OB85_RESERVED_2 : Byte;   // Reserved for system
      OB85_RESERVED_3 : Int;   // Reserved for system
      OB85_ERR_EV_CLASS : Byte;   // Class of event causing error
      OB85_ERR_EV_NUM : Byte;   // Number of event causing error
      OB85_OB_PRIOR : Byte;   // Priority of OB causing error
      OB85_OB_NUM : Byte;   // Number of OB causing error
      OB85_DATE_TIME : Date_And_Time;   // Date and time OB85 started
   END_VAR
BEGIN
END_ORGANIZATION_BLOCK

ORGANIZATION_BLOCK "RACK_FLT"   // OB86, LAD
TITLE = "Loss Of Rack Fault"
{ S7_Optimized_Access := 'FALSE' }
VERSION : 0.1
   VAR_TEMP
      OB86_EV_CLASS : Byte;   // 16#38/39 Event class 3
      OB86_FLT_ID : Byte;   // 16#C1/C4/C5, Fault identifcation code
      OB86_PRIORITY : Byte;   // Priority of OB Execution
      OB86_OB_NUMBR : Byte;   // 86 (Organization block 86, OB86)
      OB86_RESERVED_1 : Byte;   // Reserved for system
      OB86_RESERVED_2 : Byte;   // Reserved for system
      OB86_MDL_ADDR : Word;   // Base address of IM module in rack with fault
      OB86_RACKS_FLTD : Array[0..31] of Bool;
      OB86_DATE_TIME : Date_And_Time;   // Date and time OB86 started
   END_VAR
BEGIN
END_ORGANIZATION_BLOCK

ORGANIZATION_BLOCK "COMM_FLT"   // OB87, LAD
TITLE = "Communication Fault"
{ S7_Optimized_Access := 'FALSE' }
VERSION : 0.1
   VAR_TEMP
      OB87_EV_CLASS : Byte;   // 16#39 Event class 3
      OB87_FLT_ID : Byte;   // 16#XX, Fault identifcation code
      OB87_PRIORITY : Byte;   // Priority of OB Execution
      OB87_OB_NUMBR : Byte;   // 87 (Organization block 87, OB87)
      OB87_RESERVED_1 : Byte;   // Reserved for system
      OB87_RESERVED_2 : Byte;   // Reserved for system
      OB87_RESERVED_3 : Word;   // Reserved for system
      OB87_RESERVED_4 : DWord;   // Reserved for system
      OB87_DATE_TIME : Date_And_Time;   // Date and time OB87 started
   END_VAR
BEGIN
END_ORGANIZATION_BLOCK

ORGANIZATION_BLOCK "INICIAL"   // OB100, LAD
TITLE = MÓDULO INICIAL
{ S7_Optimized_Access := 'FALSE' }
AUTHOR : THALLES
FAMILY : INICIAL
NAME : LINHA1
VERSION : 0.1
// DATA BLOCK DE CONTROLE // DB1
// Automation Pack Automação Indl. e Com. Ltda.
// Cliente: Texima S/A Ind. de Máquinas
// Cliente Final: Cia. Fiação e Tecidos Santo Antonio.
// Máquina: LINHA 1 DENIN - O.S.: 24.626
   VAR_TEMP
      OB100_EV_CLASS : Byte;   // 16#13, Event class 1, Entering event state, Event logged in diagnostic buffer
      OB100_STRTUP : Byte;   // 16#81/82/83/84 Method of startup
      OB100_PRIORITY : Byte;   // Priority of OB Execution
      OB100_OB_NUMBR : Byte;   // 100 (Organization block 100, OB100)
      OB100_RESERVED_1 : Byte;   // Reserved for system
      OB100_RESERVED_2 : Byte;   // Reserved for system
      OB100_STOP : Word;   // Event that caused CPU to stop (16#4xxx)
      OB100_STRT_INFO : DWord;   // Information on how system started
      OB100_DATE_TIME : Date_And_Time;   // Date and time OB100 started
   END_VAR
BEGIN

REGION Network 1 (STL): BIT DE USO GERAL
   // DESLIGA SEMPRE EM "0"
   // LIGA SEMPRE EM "1"
         CLR;
         =     "DB PRINCIPAL".AUXILIARES.SEMPRE_0;

         SET;
         =     "DB PRINCIPAL".AUXILIARES.SEMPRE_1;
END_REGION

REGION Network 2 (STL): BIT´S / REFERÊNCIAS PRINCIPAIS
   // DESLIGA / ZERA
         L     0.0;
         T     "DB PRINCIPAL".REFERENCIAS.BASE;
         T     "DB PRINCIPAL".REFERENCIAS.FINAL_MAQUINA;

         CLR;
         =     "DB PRINCIPAL".COMANDOS.JOG;
         =     "DB PRINCIPAL".COMANDOS.MARCHA;
END_REGION
END_ORGANIZATION_BLOCK

ORGANIZATION_BLOCK "PROG_ERR"   // OB121, LAD
TITLE = "Programming Error"
{ S7_Optimized_Access := 'FALSE' }
VERSION : 0.1
   VAR_TEMP
      OB121_EV_CLASS : Byte;   // 16#25, Event class 2, Entering event state, Internal fault event
      OB121_SW_FLT : Byte;   // 16#XX Software programming fault
      OB121_PRIORITY : Byte;   // Priority of OB Execution
      OB121_OB_NUMBR : Byte;   // 121 (Organization block 121, OB121)
      OB121_BLK_TYPE : Byte;   // 16#88/8A/8B/8C/8E Type of block fault occured in
      OB121_RESERVED_1 : Byte;   // Reserved for system
      OB121_FLT_REG : Word;   // 16#XX Specific register that caused fault
      OB121_BLK_NUM : Word;   // Number of block that programming fault occured in
      OB121_PRG_ADDR : Word;   // Address in block where programming fault occured
      OB121_DATE_TIME : Date_And_Time;   // Date and time OB121 started
   END_VAR
BEGIN
END_ORGANIZATION_BLOCK

ORGANIZATION_BLOCK "MOD_ERR"   // OB122, LAD
TITLE = "Module Access Error"
{ S7_Optimized_Access := 'FALSE' }
VERSION : 0.1
   VAR_TEMP
      OB122_EV_CLASS : Byte;   // 16#29, Event class 2, Entering event state, Internal fault event
      OB122_SW_FLT : Byte;   // 16#XX Software error code
      OB122_PRIORITY : Byte;   // Priority of OB Execution
      OB122_OB_NUMBR : Byte;   // 122 (Organization block 122, OB122)
      OB122_BLK_TYPE : Byte;   // 16#88/8C/8E Type of block fault occured in
      OB122_MEM_AREA : Byte;   // Memory area where access error occured
      OB122_MEM_ADDR : Word;   // Memory address where access error occured
      OB122_BLK_NUM : Word;   // Block number in which error occured
      OB122_PRG_ADDR : Word;   // Program address where error occured
      OB122_DATE_TIME : Date_And_Time;   // Date and time OB1 started
   END_VAR
BEGIN
END_ORGANIZATION_BLOCK